// TIA Portal V17 export
// export: Created 2025-07-01T09:58:49.6236345Z, ExportSetting WithDefaults, DisplayName Totally Integrated Automation Portal, DisplayVersion V17 Update 8, DisplayName TIA Portal Openness, DisplayVersion V17 Update 8, DisplayName TIA Portal Version Control Interface, DisplayVersion V17, DisplayName SINAMICS Startdrive Advanced, DisplayVersion V17 SP2, DisplayName SINAMICS Startdrive G110M, G120, G120C, G120D, G120P, G115D, DisplayVersion V17 SP2, DisplayName SINAMICS Startdrive G130, G150, S120, S150, SINAMICS MV, S210, DisplayVersion V17 SP2, DisplayName STEP 7 Professional, DisplayVersion V17 Update 8, DisplayName SINUMERIK ONE STEP 7 Toolbox, DisplayVersion V17 Update 12, DisplayName SINUMERIK ONE PLC Basic Program Plus, DisplayVersion V17 Update 12, DisplayName SINUMERIK 840D sl STEP 7 Toolbox, DisplayVersion V17 Update 12, DisplayName STEP 7 Safety, DisplayVersion V17 Update 6, DisplayName WinCC Advanced, DisplayVersion V17 Update 8
FUNCTION "FC1201_PART_CYCLE_UNIT_1_CLADDING" : Void   // FC1201, LAD
{ S7_Optimized_Access := 'FALSE' }
AUTHOR : ETXETAR
VERSION : 1.0
// stored: AutoNumber false, IsIECCheckEnabled false, SetENOAutomatically false, UDAEnableTagReadback false
   VAR CONSTANT
      FC_NUMBER : DInt := 1201;
   END_VAR
   VAR_TEMP   // added for the SCL form of the ladder/FBD networks
      _w1 : Bool;
      _w2 : Bool;
      _w3 : Bool;
      _w4 : Bool;
   END_VAR
BEGIN

REGION Network 1: GENERAL CONDITIONS
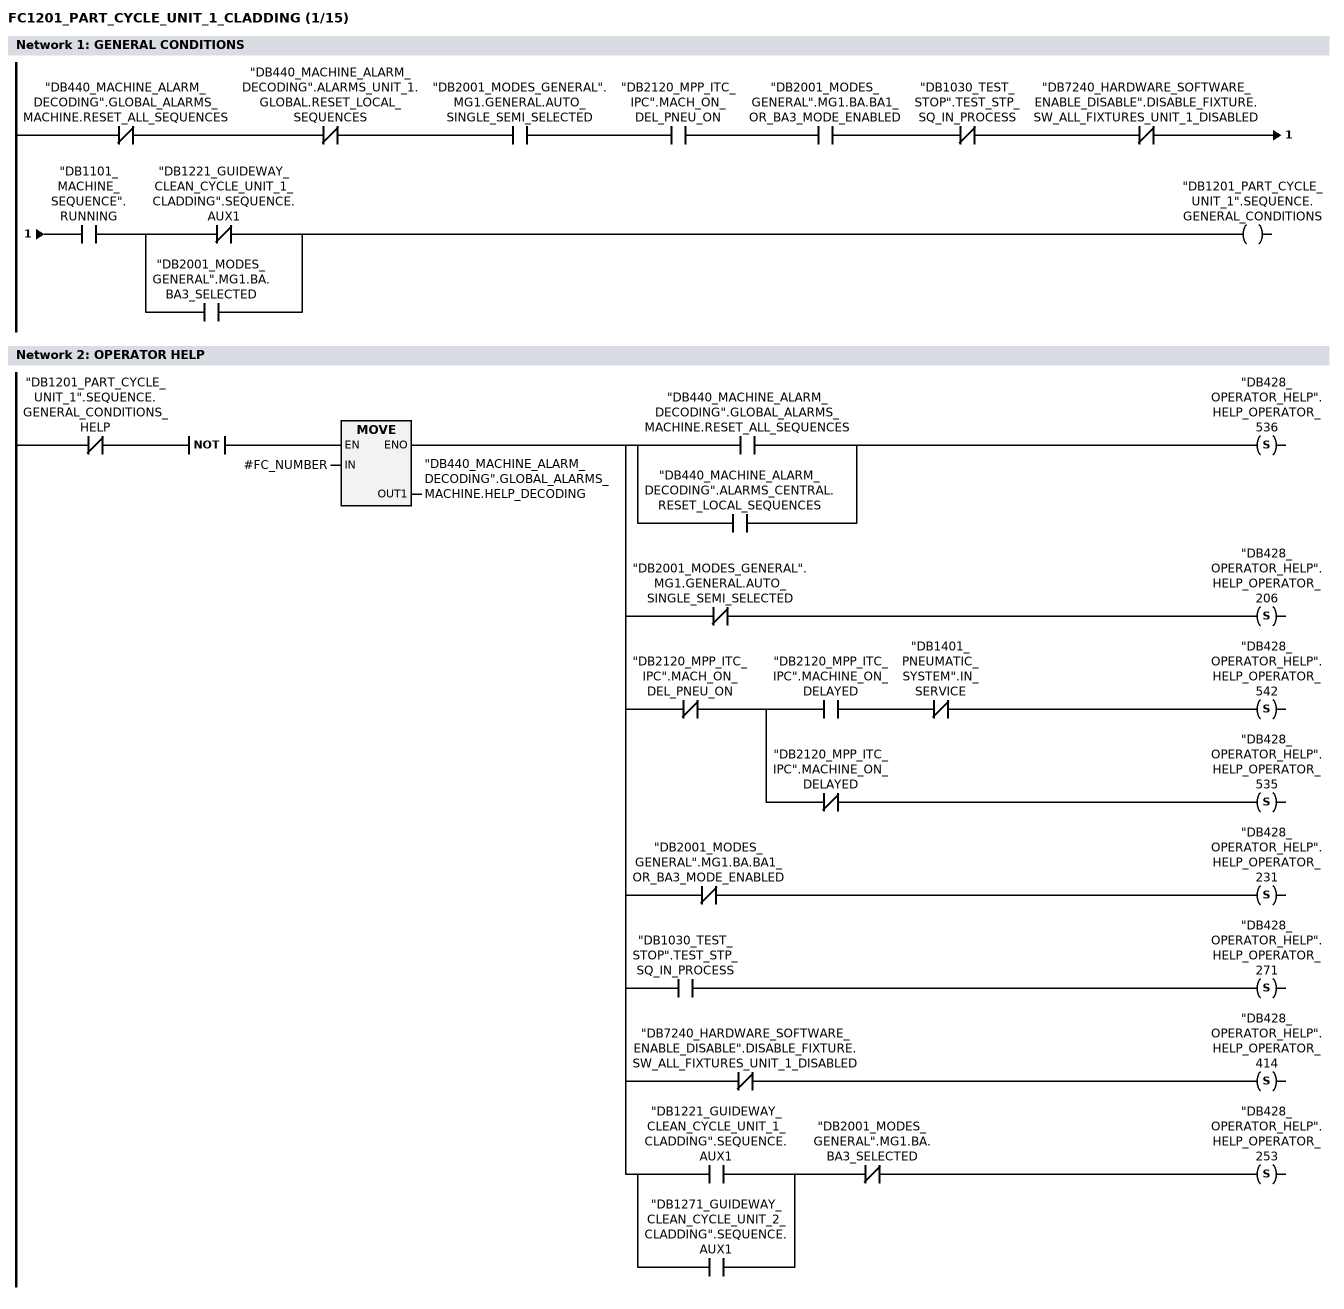
   RUNG wire#powerrail
      I_Contact( "DB440_MACHINE_ALARM_DECODING".GLOBAL_ALARMS_MACHINE.RESET_ALL_SEQUENCES )
      I_Contact( "DB440_MACHINE_ALARM_DECODING".ALARMS_UNIT_1.GLOBAL.RESET_LOCAL_SEQUENCES )
      Contact( "DB2001_MODES_GENERAL".MG1.GENERAL.AUTO_SINGLE_SEMI_SELECTED )
      Contact( "DB2120_MPP_ITC_IPC".MACH_ON_DEL_PNEU_ON )
      Contact( "DB2001_MODES_GENERAL".MG1.BA.BA1_OR_BA3_MODE_ENABLED )
      I_Contact( "DB1030_TEST_STOP".TEST_STP_SQ_IN_PROCESS )
      I_Contact( "DB7240_HARDWARE_SOFTWARE_ENABLE_DISABLE".DISABLE_FIXTURE.SW_ALL_FIXTURES_UNIT_1_DISABLED )
      Contact( "DB1101_MACHINE_SEQUENCE".RUNNING )
      wire#w1
      I_Contact( "DB1221_GUIDEWAY_CLEAN_CYCLE_UNIT_1_CLADDING".SEQUENCE.AUX1 )
      wire#w2
      Coil( "DB1201_PART_CYCLE_UNIT_1".SEQUENCE.GENERAL_CONDITIONS )
   END_RUNG
   RUNG wire#w1
      Contact( "DB2001_MODES_GENERAL".MG1.BA.BA3_SELECTED )
   END_RUNG wire#w2
   // the same network as SCL:
   "DB1201_PART_CYCLE_UNIT_1".SEQUENCE.GENERAL_CONDITIONS := NOT "DB440_MACHINE_ALARM_DECODING".GLOBAL_ALARMS_MACHINE.RESET_ALL_SEQUENCES AND NOT "DB440_MACHINE_ALARM_DECODING".ALARMS_UNIT_1.GLOBAL.RESET_LOCAL_SEQUENCES AND "DB2001_MODES_GENERAL".MG1.GENERAL.AUTO_SINGLE_SEMI_SELECTED AND "DB2120_MPP_ITC_IPC".MACH_ON_DEL_PNEU_ON AND "DB2001_MODES_GENERAL".MG1.BA.BA1_OR_BA3_MODE_ENABLED AND NOT "DB1030_TEST_STOP".TEST_STP_SQ_IN_PROCESS AND NOT "DB7240_HARDWARE_SOFTWARE_ENABLE_DISABLE".DISABLE_FIXTURE.SW_ALL_FIXTURES_UNIT_1_DISABLED AND "DB1101_MACHINE_SEQUENCE".RUNNING AND (NOT "DB1221_GUIDEWAY_CLEAN_CYCLE_UNIT_1_CLADDING".SEQUENCE.AUX1 OR "DB2001_MODES_GENERAL".MG1.BA.BA3_SELECTED);
END_REGION

REGION Network 2: OPERATOR HELP
   RUNG wire#powerrail
      I_Contact( "DB1201_PART_CYCLE_UNIT_1".SEQUENCE.GENERAL_CONDITIONS_HELP )
      Not()
      { S7_GenerateENO := "TRUE" } Move(in := #FC_NUMBER, out1 => "DB440_MACHINE_ALARM_DECODING".GLOBAL_ALARMS_MACHINE.HELP_DECODING)
      wire#w1
      Contact( "DB440_MACHINE_ALARM_DECODING".GLOBAL_ALARMS_MACHINE.RESET_ALL_SEQUENCES )
      wire#w2
      S_Coil( "DB428_OPERATOR_HELP".HELP_OPERATOR_536 )
   END_RUNG
   RUNG wire#w1
      Contact( "DB440_MACHINE_ALARM_DECODING".ALARMS_CENTRAL.RESET_LOCAL_SEQUENCES )
   END_RUNG wire#w2
   RUNG wire#w1
      I_Contact( "DB2001_MODES_GENERAL".MG1.GENERAL.AUTO_SINGLE_SEMI_SELECTED )
      S_Coil( "DB428_OPERATOR_HELP".HELP_OPERATOR_206 )
   END_RUNG
   RUNG wire#w1
      I_Contact( "DB2120_MPP_ITC_IPC".MACH_ON_DEL_PNEU_ON )
      wire#w3
      Contact( "DB2120_MPP_ITC_IPC".MACHINE_ON_DELAYED )
      I_Contact( "DB1401_PNEUMATIC_SYSTEM".IN_SERVICE )
      S_Coil( "DB428_OPERATOR_HELP".HELP_OPERATOR_542 )
   END_RUNG
   RUNG wire#w3
      I_Contact( "DB2120_MPP_ITC_IPC".MACHINE_ON_DELAYED )
      S_Coil( "DB428_OPERATOR_HELP".HELP_OPERATOR_535 )
   END_RUNG
   RUNG wire#w1
      I_Contact( "DB2001_MODES_GENERAL".MG1.BA.BA1_OR_BA3_MODE_ENABLED )
      S_Coil( "DB428_OPERATOR_HELP".HELP_OPERATOR_231 )
   END_RUNG
   RUNG wire#w1
      Contact( "DB1030_TEST_STOP".TEST_STP_SQ_IN_PROCESS )
      S_Coil( "DB428_OPERATOR_HELP".HELP_OPERATOR_271 )
   END_RUNG
   RUNG wire#w1
      I_Contact( "DB7240_HARDWARE_SOFTWARE_ENABLE_DISABLE".DISABLE_FIXTURE.SW_ALL_FIXTURES_UNIT_1_DISABLED )
      S_Coil( "DB428_OPERATOR_HELP".HELP_OPERATOR_414 )
   END_RUNG
   RUNG wire#w1
      Contact( "DB1221_GUIDEWAY_CLEAN_CYCLE_UNIT_1_CLADDING".SEQUENCE.AUX1 )
      wire#w4
      I_Contact( "DB2001_MODES_GENERAL".MG1.BA.BA3_SELECTED )
      S_Coil( "DB428_OPERATOR_HELP".HELP_OPERATOR_253 )
   END_RUNG
   RUNG wire#w1
      Contact( "DB1271_GUIDEWAY_CLEAN_CYCLE_UNIT_2_CLADDING".SEQUENCE.AUX1 )
   END_RUNG wire#w4
   // the same network as SCL:
   // ENO of a box is taken as its EN; it also drops when the box reports an error
   #_w1 := NOT (NOT "DB1201_PART_CYCLE_UNIT_1".SEQUENCE.GENERAL_CONDITIONS_HELP);
   IF #_w1 THEN "DB440_MACHINE_ALARM_DECODING".GLOBAL_ALARMS_MACHINE.HELP_DECODING := #FC_NUMBER; END_IF;
   IF #_w1 AND ("DB440_MACHINE_ALARM_DECODING".GLOBAL_ALARMS_MACHINE.RESET_ALL_SEQUENCES OR "DB440_MACHINE_ALARM_DECODING".ALARMS_CENTRAL.RESET_LOCAL_SEQUENCES) THEN
       "DB428_OPERATOR_HELP".HELP_OPERATOR_536 := TRUE;
   END_IF;
   IF #_w1 AND NOT "DB2001_MODES_GENERAL".MG1.GENERAL.AUTO_SINGLE_SEMI_SELECTED THEN
       "DB428_OPERATOR_HELP".HELP_OPERATOR_206 := TRUE;
   END_IF;
   #_w2 := #_w1 AND NOT "DB2120_MPP_ITC_IPC".MACH_ON_DEL_PNEU_ON;
   IF #_w2 AND "DB2120_MPP_ITC_IPC".MACHINE_ON_DELAYED AND NOT "DB1401_PNEUMATIC_SYSTEM".IN_SERVICE THEN
       "DB428_OPERATOR_HELP".HELP_OPERATOR_542 := TRUE;
   END_IF;
   IF #_w2 AND NOT "DB2120_MPP_ITC_IPC".MACHINE_ON_DELAYED THEN
       "DB428_OPERATOR_HELP".HELP_OPERATOR_535 := TRUE;
   END_IF;
   IF #_w1 AND NOT "DB2001_MODES_GENERAL".MG1.BA.BA1_OR_BA3_MODE_ENABLED THEN
       "DB428_OPERATOR_HELP".HELP_OPERATOR_231 := TRUE;
   END_IF;
   IF #_w1 AND "DB1030_TEST_STOP".TEST_STP_SQ_IN_PROCESS THEN
       "DB428_OPERATOR_HELP".HELP_OPERATOR_271 := TRUE;
   END_IF;
   IF #_w1 AND NOT "DB7240_HARDWARE_SOFTWARE_ENABLE_DISABLE".DISABLE_FIXTURE.SW_ALL_FIXTURES_UNIT_1_DISABLED THEN
       "DB428_OPERATOR_HELP".HELP_OPERATOR_414 := TRUE;
   END_IF;
   IF #_w1 AND ("DB1221_GUIDEWAY_CLEAN_CYCLE_UNIT_1_CLADDING".SEQUENCE.AUX1 OR "DB1271_GUIDEWAY_CLEAN_CYCLE_UNIT_2_CLADDING".SEQUENCE.AUX1) AND NOT "DB2001_MODES_GENERAL".MG1.BA.BA3_SELECTED THEN
       "DB428_OPERATOR_HELP".HELP_OPERATOR_253 := TRUE;
   END_IF;
END_REGION

REGION Network 3: INITIAL CONDITIONS
   // CAMBIAR LOS BITS DE QUALITY CUANDO ESTEN HECHOS
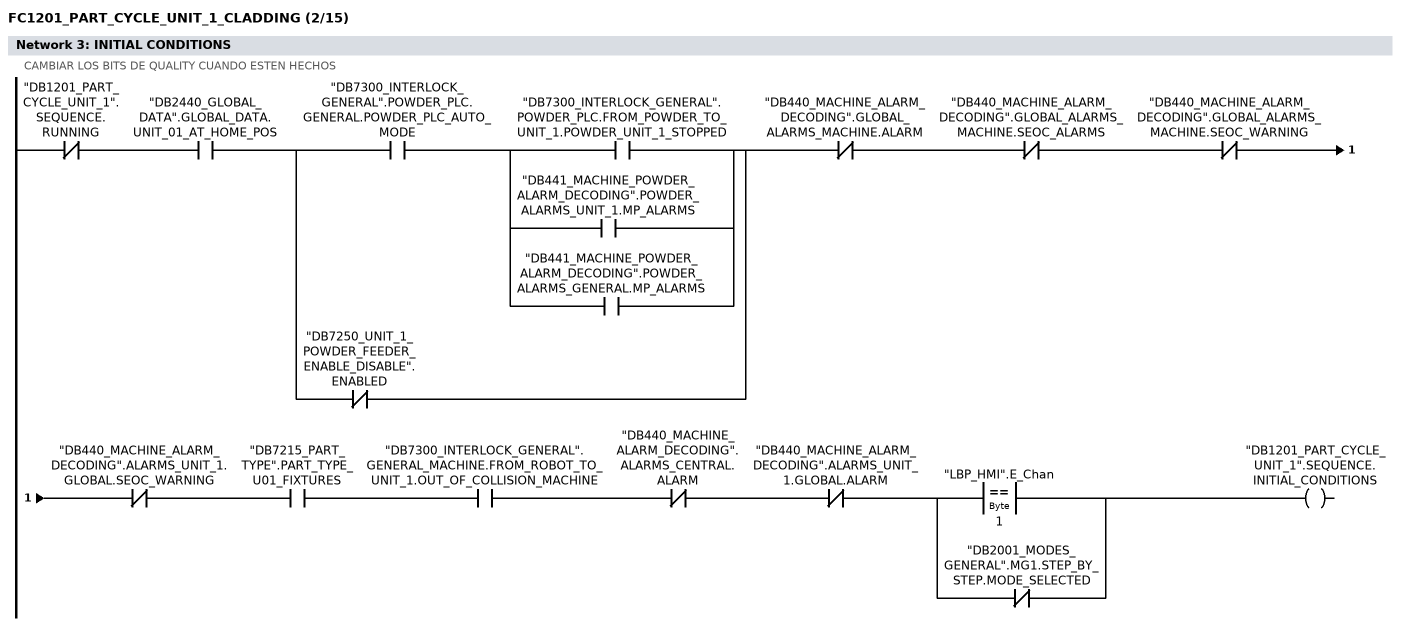
   RUNG wire#powerrail
      I_Contact( "DB1201_PART_CYCLE_UNIT_1".SEQUENCE.RUNNING )
      Contact( "DB2440_GLOBAL_DATA".GLOBAL_DATA.UNIT_01_AT_HOME_POS )
      wire#w1
      Contact( "DB7300_INTERLOCK_GENERAL".POWDER_PLC.GENERAL.POWDER_PLC_AUTO_MODE )
      wire#w2
      Contact( "DB7300_INTERLOCK_GENERAL".POWDER_PLC.FROM_POWDER_TO_UNIT_1.POWDER_UNIT_1_STOPPED )
      wire#w3
      I_Contact( "DB440_MACHINE_ALARM_DECODING".GLOBAL_ALARMS_MACHINE.ALARM )
      I_Contact( "DB440_MACHINE_ALARM_DECODING".GLOBAL_ALARMS_MACHINE.SEOC_ALARMS )
      I_Contact( "DB440_MACHINE_ALARM_DECODING".GLOBAL_ALARMS_MACHINE.SEOC_WARNING )
      I_Contact( "DB440_MACHINE_ALARM_DECODING".ALARMS_UNIT_1.GLOBAL.SEOC_WARNING )
      Contact( "DB7215_PART_TYPE".PART_TYPE_U01_FIXTURES )
      Contact( "DB7300_INTERLOCK_GENERAL".GENERAL_MACHINE.FROM_ROBOT_TO_UNIT_1.OUT_OF_COLLISION_MACHINE )
      I_Contact( "DB440_MACHINE_ALARM_DECODING".ALARMS_CENTRAL.ALARM )
      I_Contact( "DB440_MACHINE_ALARM_DECODING".ALARMS_UNIT_1.GLOBAL.ALARM )
      wire#w4
      { S7_Templates := "SrcType := Byte" } EQ_Contact(in1 := "LBP_HMI".E_Chan, in2 := 1)
      wire#w5
      Coil( "DB1201_PART_CYCLE_UNIT_1".SEQUENCE.INITIAL_CONDITIONS )
   END_RUNG
   RUNG wire#w2
      Contact( "DB441_MACHINE_POWDER_ALARM_DECODING".POWDER_ALARMS_UNIT_1.MP_ALARMS )
   END_RUNG wire#w3
   RUNG wire#w2
      Contact( "DB441_MACHINE_POWDER_ALARM_DECODING".POWDER_ALARMS_GENERAL.MP_ALARMS )
   END_RUNG wire#w3
   RUNG wire#w1
      I_Contact( "DB7250_UNIT_1_POWDER_FEEDER_ENABLE_DISABLE".ENABLED )
   END_RUNG wire#w3
   RUNG wire#w4
      I_Contact( "DB2001_MODES_GENERAL".MG1.STEP_BY_STEP.MODE_SELECTED )
   END_RUNG wire#w5
   // the same network as SCL:
   "DB1201_PART_CYCLE_UNIT_1".SEQUENCE.INITIAL_CONDITIONS := NOT "DB1201_PART_CYCLE_UNIT_1".SEQUENCE.RUNNING AND "DB2440_GLOBAL_DATA".GLOBAL_DATA.UNIT_01_AT_HOME_POS AND (("DB7300_INTERLOCK_GENERAL".POWDER_PLC.GENERAL.POWDER_PLC_AUTO_MODE AND ("DB7300_INTERLOCK_GENERAL".POWDER_PLC.FROM_POWDER_TO_UNIT_1.POWDER_UNIT_1_STOPPED OR "DB441_MACHINE_POWDER_ALARM_DECODING".POWDER_ALARMS_UNIT_1.MP_ALARMS OR "DB441_MACHINE_POWDER_ALARM_DECODING".POWDER_ALARMS_GENERAL.MP_ALARMS)) OR NOT "DB7250_UNIT_1_POWDER_FEEDER_ENABLE_DISABLE".ENABLED) AND NOT "DB440_MACHINE_ALARM_DECODING".GLOBAL_ALARMS_MACHINE.ALARM AND NOT "DB440_MACHINE_ALARM_DECODING".GLOBAL_ALARMS_MACHINE.SEOC_ALARMS AND NOT "DB440_MACHINE_ALARM_DECODING".GLOBAL_ALARMS_MACHINE.SEOC_WARNING AND NOT "DB440_MACHINE_ALARM_DECODING".ALARMS_UNIT_1.GLOBAL.SEOC_WARNING AND "DB7215_PART_TYPE".PART_TYPE_U01_FIXTURES AND "DB7300_INTERLOCK_GENERAL".GENERAL_MACHINE.FROM_ROBOT_TO_UNIT_1.OUT_OF_COLLISION_MACHINE AND NOT "DB440_MACHINE_ALARM_DECODING".ALARMS_CENTRAL.ALARM AND NOT "DB440_MACHINE_ALARM_DECODING".ALARMS_UNIT_1.GLOBAL.ALARM AND (("LBP_HMI".E_Chan = 1) OR NOT "DB2001_MODES_GENERAL".MG1.STEP_BY_STEP.MODE_SELECTED);
END_REGION

REGION Network 4: OPERATOR HELP
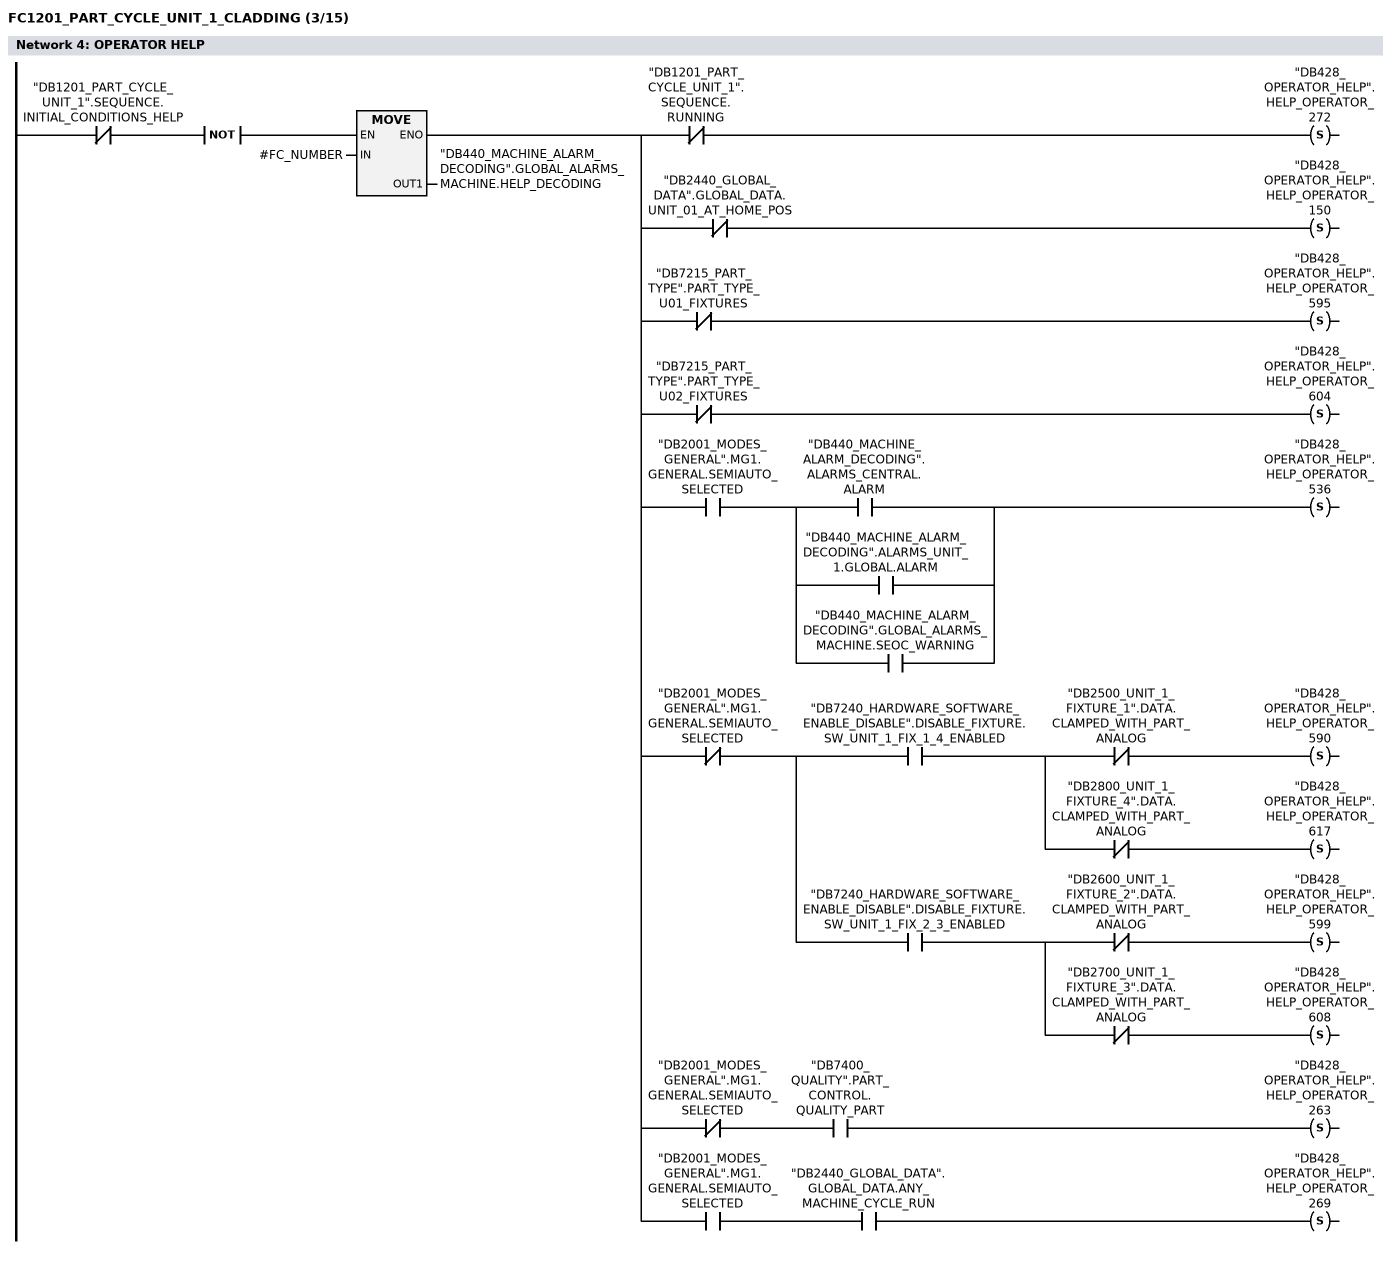
   RUNG wire#powerrail
      I_Contact( "DB1201_PART_CYCLE_UNIT_1".SEQUENCE.INITIAL_CONDITIONS_HELP )
      Not()
      { S7_GenerateENO := "TRUE" } Move(in := #FC_NUMBER, out1 => "DB440_MACHINE_ALARM_DECODING".GLOBAL_ALARMS_MACHINE.HELP_DECODING)
      wire#w1
      I_Contact( "DB1201_PART_CYCLE_UNIT_1".SEQUENCE.RUNNING )
      S_Coil( "DB428_OPERATOR_HELP".HELP_OPERATOR_272 )
   END_RUNG
   RUNG wire#w1
      I_Contact( "DB2440_GLOBAL_DATA".GLOBAL_DATA.UNIT_01_AT_HOME_POS )
      S_Coil( "DB428_OPERATOR_HELP".HELP_OPERATOR_150 )
   END_RUNG
   RUNG wire#w1
      I_Contact( "DB7215_PART_TYPE".PART_TYPE_U01_FIXTURES )
      S_Coil( "DB428_OPERATOR_HELP".HELP_OPERATOR_595 )
   END_RUNG
   RUNG wire#w1
      I_Contact( "DB7215_PART_TYPE".PART_TYPE_U02_FIXTURES )
      S_Coil( "DB428_OPERATOR_HELP".HELP_OPERATOR_604 )
   END_RUNG
   RUNG wire#w1
      Contact( "DB2001_MODES_GENERAL".MG1.GENERAL.SEMIAUTO_SELECTED )
      wire#w2
      Contact( "DB440_MACHINE_ALARM_DECODING".ALARMS_CENTRAL.ALARM )
      wire#w3
      S_Coil( "DB428_OPERATOR_HELP".HELP_OPERATOR_536 )
   END_RUNG
   RUNG wire#w2
      Contact( "DB440_MACHINE_ALARM_DECODING".ALARMS_UNIT_1.GLOBAL.ALARM )
   END_RUNG wire#w3
   RUNG wire#w2
      Contact( "DB440_MACHINE_ALARM_DECODING".GLOBAL_ALARMS_MACHINE.SEOC_WARNING )
   END_RUNG wire#w3
   RUNG wire#w1
      I_Contact( "DB2001_MODES_GENERAL".MG1.GENERAL.SEMIAUTO_SELECTED )
      wire#w4
      Contact( "DB7240_HARDWARE_SOFTWARE_ENABLE_DISABLE".DISABLE_FIXTURE.SW_UNIT_1_FIX_1_4_ENABLED )
      wire#w5
      I_Contact( "DB2500_UNIT_1_FIXTURE_1".DATA.CLAMPED_WITH_PART_ANALOG )
      S_Coil( "DB428_OPERATOR_HELP".HELP_OPERATOR_590 )
   END_RUNG
   RUNG wire#w5
      I_Contact( "DB2800_UNIT_1_FIXTURE_4".DATA.CLAMPED_WITH_PART_ANALOG )
      S_Coil( "DB428_OPERATOR_HELP".HELP_OPERATOR_617 )
   END_RUNG
   RUNG wire#w4
      Contact( "DB7240_HARDWARE_SOFTWARE_ENABLE_DISABLE".DISABLE_FIXTURE.SW_UNIT_1_FIX_2_3_ENABLED )
      wire#w6
      I_Contact( "DB2600_UNIT_1_FIXTURE_2".DATA.CLAMPED_WITH_PART_ANALOG )
      S_Coil( "DB428_OPERATOR_HELP".HELP_OPERATOR_599 )
   END_RUNG
   RUNG wire#w6
      I_Contact( "DB2700_UNIT_1_FIXTURE_3".DATA.CLAMPED_WITH_PART_ANALOG )
      S_Coil( "DB428_OPERATOR_HELP".HELP_OPERATOR_608 )
   END_RUNG
   RUNG wire#w1
      I_Contact( "DB2001_MODES_GENERAL".MG1.GENERAL.SEMIAUTO_SELECTED )
      Contact( "DB7400_QUALITY".PART_CONTROL.QUALITY_PART )
      S_Coil( "DB428_OPERATOR_HELP".HELP_OPERATOR_263 )
   END_RUNG
   RUNG wire#w1
      Contact( "DB2001_MODES_GENERAL".MG1.GENERAL.SEMIAUTO_SELECTED )
      Contact( "DB2440_GLOBAL_DATA".GLOBAL_DATA.ANY_MACHINE_CYCLE_RUN )
      S_Coil( "DB428_OPERATOR_HELP".HELP_OPERATOR_269 )
   END_RUNG
   // the same network as SCL:
   // ENO of a box is taken as its EN; it also drops when the box reports an error
   #_w1 := NOT (NOT "DB1201_PART_CYCLE_UNIT_1".SEQUENCE.INITIAL_CONDITIONS_HELP);
   IF #_w1 THEN "DB440_MACHINE_ALARM_DECODING".GLOBAL_ALARMS_MACHINE.HELP_DECODING := #FC_NUMBER; END_IF;
   IF #_w1 AND NOT "DB1201_PART_CYCLE_UNIT_1".SEQUENCE.RUNNING THEN
       "DB428_OPERATOR_HELP".HELP_OPERATOR_272 := TRUE;
   END_IF;
   IF #_w1 AND NOT "DB2440_GLOBAL_DATA".GLOBAL_DATA.UNIT_01_AT_HOME_POS THEN
       "DB428_OPERATOR_HELP".HELP_OPERATOR_150 := TRUE;
   END_IF;
   IF #_w1 AND NOT "DB7215_PART_TYPE".PART_TYPE_U01_FIXTURES THEN
       "DB428_OPERATOR_HELP".HELP_OPERATOR_595 := TRUE;
   END_IF;
   IF #_w1 AND NOT "DB7215_PART_TYPE".PART_TYPE_U02_FIXTURES THEN
       "DB428_OPERATOR_HELP".HELP_OPERATOR_604 := TRUE;
   END_IF;
   IF #_w1 AND "DB2001_MODES_GENERAL".MG1.GENERAL.SEMIAUTO_SELECTED AND ("DB440_MACHINE_ALARM_DECODING".ALARMS_CENTRAL.ALARM OR "DB440_MACHINE_ALARM_DECODING".ALARMS_UNIT_1.GLOBAL.ALARM OR "DB440_MACHINE_ALARM_DECODING".GLOBAL_ALARMS_MACHINE.SEOC_WARNING) THEN
       "DB428_OPERATOR_HELP".HELP_OPERATOR_536 := TRUE;
   END_IF;
   #_w2 := #_w1 AND NOT "DB2001_MODES_GENERAL".MG1.GENERAL.SEMIAUTO_SELECTED;
   #_w3 := #_w2 AND "DB7240_HARDWARE_SOFTWARE_ENABLE_DISABLE".DISABLE_FIXTURE.SW_UNIT_1_FIX_1_4_ENABLED;
   IF #_w3 AND NOT "DB2500_UNIT_1_FIXTURE_1".DATA.CLAMPED_WITH_PART_ANALOG THEN
       "DB428_OPERATOR_HELP".HELP_OPERATOR_590 := TRUE;
   END_IF;
   IF #_w3 AND NOT "DB2800_UNIT_1_FIXTURE_4".DATA.CLAMPED_WITH_PART_ANALOG THEN
       "DB428_OPERATOR_HELP".HELP_OPERATOR_617 := TRUE;
   END_IF;
   #_w4 := #_w2 AND "DB7240_HARDWARE_SOFTWARE_ENABLE_DISABLE".DISABLE_FIXTURE.SW_UNIT_1_FIX_2_3_ENABLED;
   IF #_w4 AND NOT "DB2600_UNIT_1_FIXTURE_2".DATA.CLAMPED_WITH_PART_ANALOG THEN
       "DB428_OPERATOR_HELP".HELP_OPERATOR_599 := TRUE;
   END_IF;
   IF #_w4 AND NOT "DB2700_UNIT_1_FIXTURE_3".DATA.CLAMPED_WITH_PART_ANALOG THEN
       "DB428_OPERATOR_HELP".HELP_OPERATOR_608 := TRUE;
   END_IF;
   IF #_w1 AND NOT "DB2001_MODES_GENERAL".MG1.GENERAL.SEMIAUTO_SELECTED AND "DB7400_QUALITY".PART_CONTROL.QUALITY_PART THEN
       "DB428_OPERATOR_HELP".HELP_OPERATOR_263 := TRUE;
   END_IF;
   IF #_w1 AND "DB2001_MODES_GENERAL".MG1.GENERAL.SEMIAUTO_SELECTED AND "DB2440_GLOBAL_DATA".GLOBAL_DATA.ANY_MACHINE_CYCLE_RUN THEN
       "DB428_OPERATOR_HELP".HELP_OPERATOR_269 := TRUE;
   END_IF;
END_REGION

REGION Network 5: SEMI AUTO REQUEST
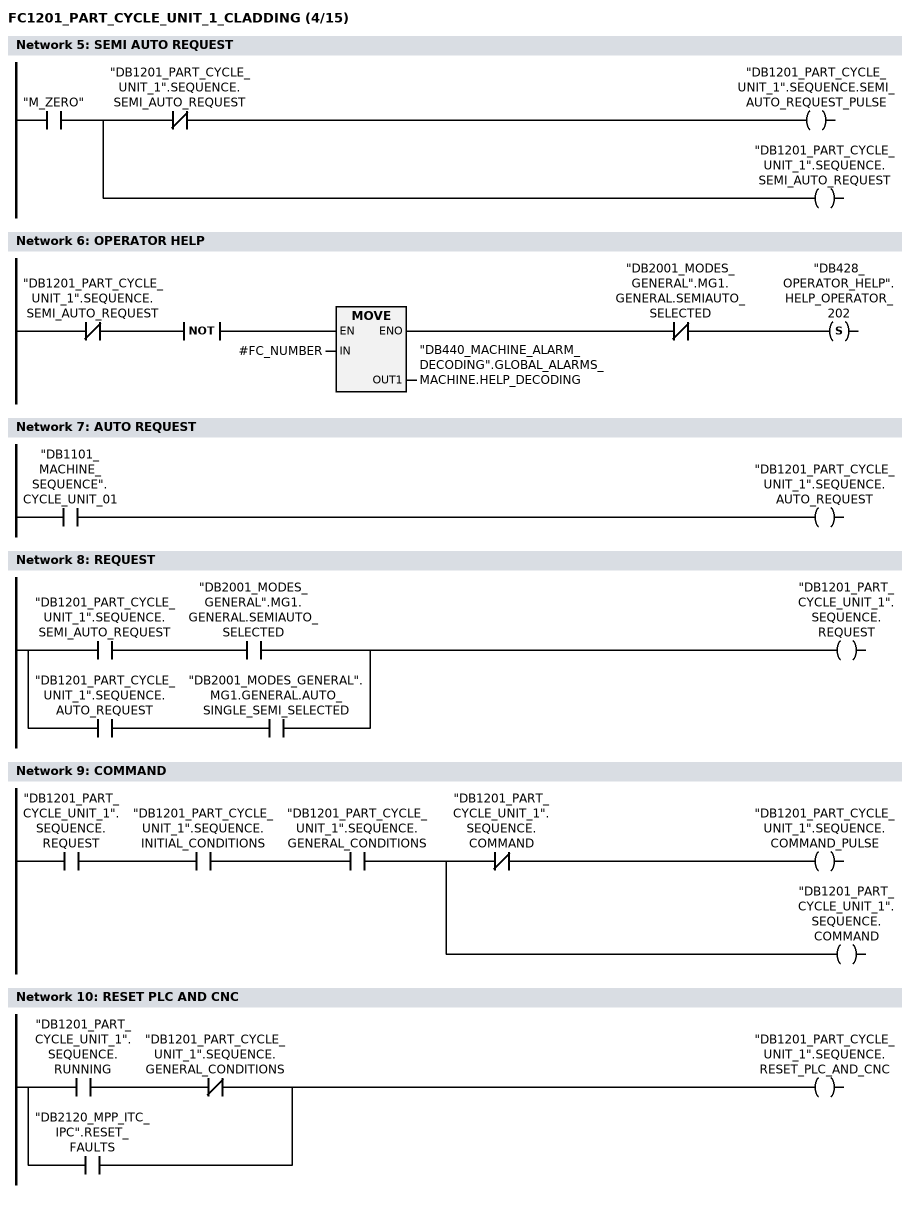
   RUNG wire#powerrail
      Contact( "M_ZERO" )
      wire#w1
      I_Contact( "DB1201_PART_CYCLE_UNIT_1".SEQUENCE.SEMI_AUTO_REQUEST )
      Coil( "DB1201_PART_CYCLE_UNIT_1".SEQUENCE.SEMI_AUTO_REQUEST_PULSE )
   END_RUNG
   RUNG wire#w1
      Coil( "DB1201_PART_CYCLE_UNIT_1".SEQUENCE.SEMI_AUTO_REQUEST )
   END_RUNG
   // the same network as SCL:
   "DB1201_PART_CYCLE_UNIT_1".SEQUENCE.SEMI_AUTO_REQUEST_PULSE := "M_ZERO" AND NOT "DB1201_PART_CYCLE_UNIT_1".SEQUENCE.SEMI_AUTO_REQUEST;
   "DB1201_PART_CYCLE_UNIT_1".SEQUENCE.SEMI_AUTO_REQUEST := "M_ZERO";
END_REGION

REGION Network 6: OPERATOR HELP
   RUNG wire#powerrail
      I_Contact( "DB1201_PART_CYCLE_UNIT_1".SEQUENCE.SEMI_AUTO_REQUEST )
      Not()
      { S7_GenerateENO := "TRUE" } Move(in := #FC_NUMBER, out1 => "DB440_MACHINE_ALARM_DECODING".GLOBAL_ALARMS_MACHINE.HELP_DECODING)
      I_Contact( "DB2001_MODES_GENERAL".MG1.GENERAL.SEMIAUTO_SELECTED )
      S_Coil( "DB428_OPERATOR_HELP".HELP_OPERATOR_202 )
   END_RUNG
   // the same network as SCL:
   // ENO of a box is taken as its EN; it also drops when the box reports an error
   #_w1 := NOT (NOT "DB1201_PART_CYCLE_UNIT_1".SEQUENCE.SEMI_AUTO_REQUEST);
   IF #_w1 THEN "DB440_MACHINE_ALARM_DECODING".GLOBAL_ALARMS_MACHINE.HELP_DECODING := #FC_NUMBER; END_IF;
   IF #_w1 AND NOT "DB2001_MODES_GENERAL".MG1.GENERAL.SEMIAUTO_SELECTED THEN
       "DB428_OPERATOR_HELP".HELP_OPERATOR_202 := TRUE;
   END_IF;
END_REGION

REGION Network 7: AUTO REQUEST
   RUNG wire#powerrail
      Contact( "DB1101_MACHINE_SEQUENCE".CYCLE_UNIT_01 )
      Coil( "DB1201_PART_CYCLE_UNIT_1".SEQUENCE.AUTO_REQUEST )
   END_RUNG
   // the same network as SCL:
   "DB1201_PART_CYCLE_UNIT_1".SEQUENCE.AUTO_REQUEST := "DB1101_MACHINE_SEQUENCE".CYCLE_UNIT_01;
END_REGION

REGION Network 8: REQUEST
   RUNG wire#powerrail
      Contact( "DB1201_PART_CYCLE_UNIT_1".SEQUENCE.SEMI_AUTO_REQUEST )
      Contact( "DB2001_MODES_GENERAL".MG1.GENERAL.SEMIAUTO_SELECTED )
      wire#w1
      Coil( "DB1201_PART_CYCLE_UNIT_1".SEQUENCE.REQUEST )
   END_RUNG
   RUNG wire#powerrail
      Contact( "DB1201_PART_CYCLE_UNIT_1".SEQUENCE.AUTO_REQUEST )
      Contact( "DB2001_MODES_GENERAL".MG1.GENERAL.AUTO_SINGLE_SEMI_SELECTED )
   END_RUNG wire#w1
   // the same network as SCL:
   "DB1201_PART_CYCLE_UNIT_1".SEQUENCE.REQUEST := ("DB1201_PART_CYCLE_UNIT_1".SEQUENCE.SEMI_AUTO_REQUEST AND "DB2001_MODES_GENERAL".MG1.GENERAL.SEMIAUTO_SELECTED) OR ("DB1201_PART_CYCLE_UNIT_1".SEQUENCE.AUTO_REQUEST AND "DB2001_MODES_GENERAL".MG1.GENERAL.AUTO_SINGLE_SEMI_SELECTED);
END_REGION

REGION Network 9: COMMAND
   RUNG wire#powerrail
      Contact( "DB1201_PART_CYCLE_UNIT_1".SEQUENCE.REQUEST )
      Contact( "DB1201_PART_CYCLE_UNIT_1".SEQUENCE.INITIAL_CONDITIONS )
      Contact( "DB1201_PART_CYCLE_UNIT_1".SEQUENCE.GENERAL_CONDITIONS )
      wire#w1
      I_Contact( "DB1201_PART_CYCLE_UNIT_1".SEQUENCE.COMMAND )
      Coil( "DB1201_PART_CYCLE_UNIT_1".SEQUENCE.COMMAND_PULSE )
   END_RUNG
   RUNG wire#w1
      Coil( "DB1201_PART_CYCLE_UNIT_1".SEQUENCE.COMMAND )
   END_RUNG
   // the same network as SCL:
   #_w1 := "DB1201_PART_CYCLE_UNIT_1".SEQUENCE.REQUEST AND "DB1201_PART_CYCLE_UNIT_1".SEQUENCE.INITIAL_CONDITIONS AND "DB1201_PART_CYCLE_UNIT_1".SEQUENCE.GENERAL_CONDITIONS;
   "DB1201_PART_CYCLE_UNIT_1".SEQUENCE.COMMAND_PULSE := #_w1 AND NOT "DB1201_PART_CYCLE_UNIT_1".SEQUENCE.COMMAND;
   "DB1201_PART_CYCLE_UNIT_1".SEQUENCE.COMMAND := #_w1;
END_REGION

REGION Network 10: RESET PLC AND CNC
   RUNG wire#powerrail
      Contact( "DB1201_PART_CYCLE_UNIT_1".SEQUENCE.RUNNING )
      I_Contact( "DB1201_PART_CYCLE_UNIT_1".SEQUENCE.GENERAL_CONDITIONS )
      wire#w1
      Coil( "DB1201_PART_CYCLE_UNIT_1".SEQUENCE.RESET_PLC_AND_CNC )
   END_RUNG
   RUNG wire#powerrail
      Contact( "DB2120_MPP_ITC_IPC".RESET_FAULTS )
   END_RUNG wire#w1
   // the same network as SCL:
   "DB1201_PART_CYCLE_UNIT_1".SEQUENCE.RESET_PLC_AND_CNC := ("DB1201_PART_CYCLE_UNIT_1".SEQUENCE.RUNNING AND NOT "DB1201_PART_CYCLE_UNIT_1".SEQUENCE.GENERAL_CONDITIONS) OR "DB2120_MPP_ITC_IPC".RESET_FAULTS;
END_REGION

REGION Network 11: RUNNING
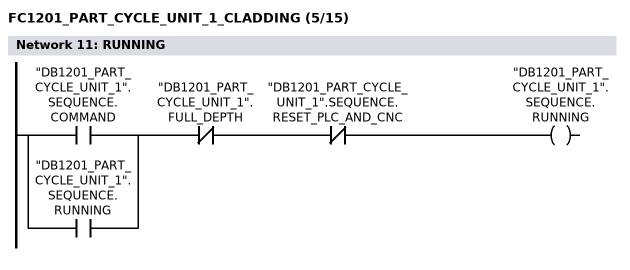
   RUNG wire#powerrail
      Contact( "DB1201_PART_CYCLE_UNIT_1".SEQUENCE.COMMAND )
      wire#w1
      I_Contact( "DB1201_PART_CYCLE_UNIT_1".FULL_DEPTH )
      I_Contact( "DB1201_PART_CYCLE_UNIT_1".SEQUENCE.RESET_PLC_AND_CNC )
      Coil( "DB1201_PART_CYCLE_UNIT_1".SEQUENCE.RUNNING )
   END_RUNG
   RUNG wire#powerrail
      Contact( "DB1201_PART_CYCLE_UNIT_1".SEQUENCE.RUNNING )
   END_RUNG wire#w1
   // the same network as SCL:
   "DB1201_PART_CYCLE_UNIT_1".SEQUENCE.RUNNING := ("DB1201_PART_CYCLE_UNIT_1".SEQUENCE.COMMAND OR "DB1201_PART_CYCLE_UNIT_1".SEQUENCE.RUNNING) AND NOT "DB1201_PART_CYCLE_UNIT_1".FULL_DEPTH AND NOT "DB1201_PART_CYCLE_UNIT_1".SEQUENCE.RESET_PLC_AND_CNC;
END_REGION

REGION Network 12: UNIT 01 STATION 1 CONDITIONS OK FOR STATION 0 CYCLE REQUEST
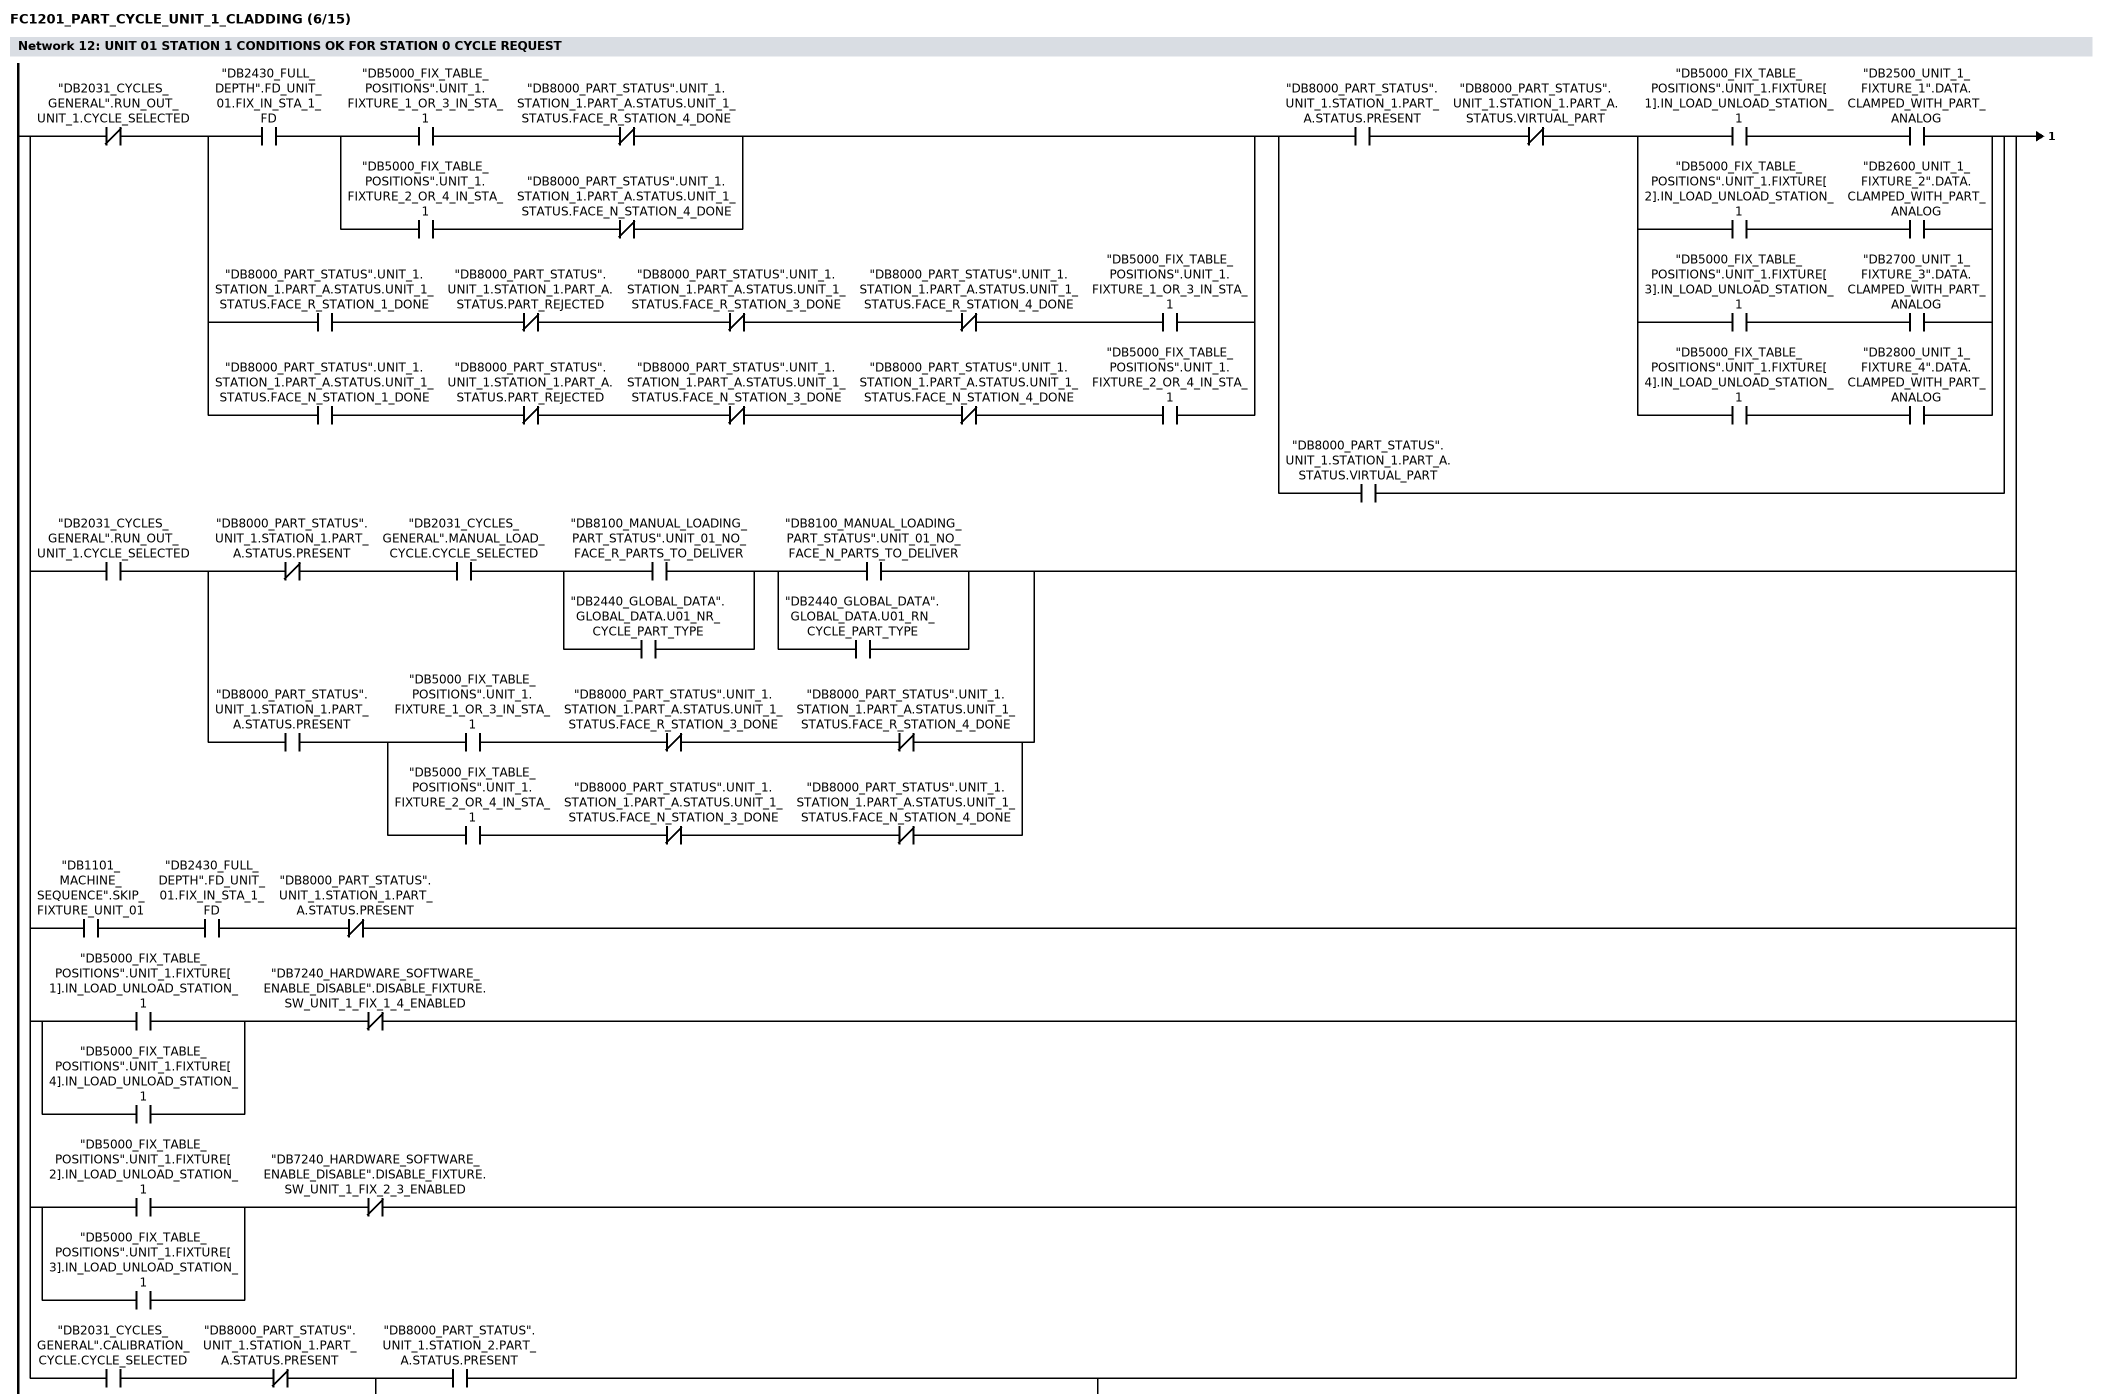
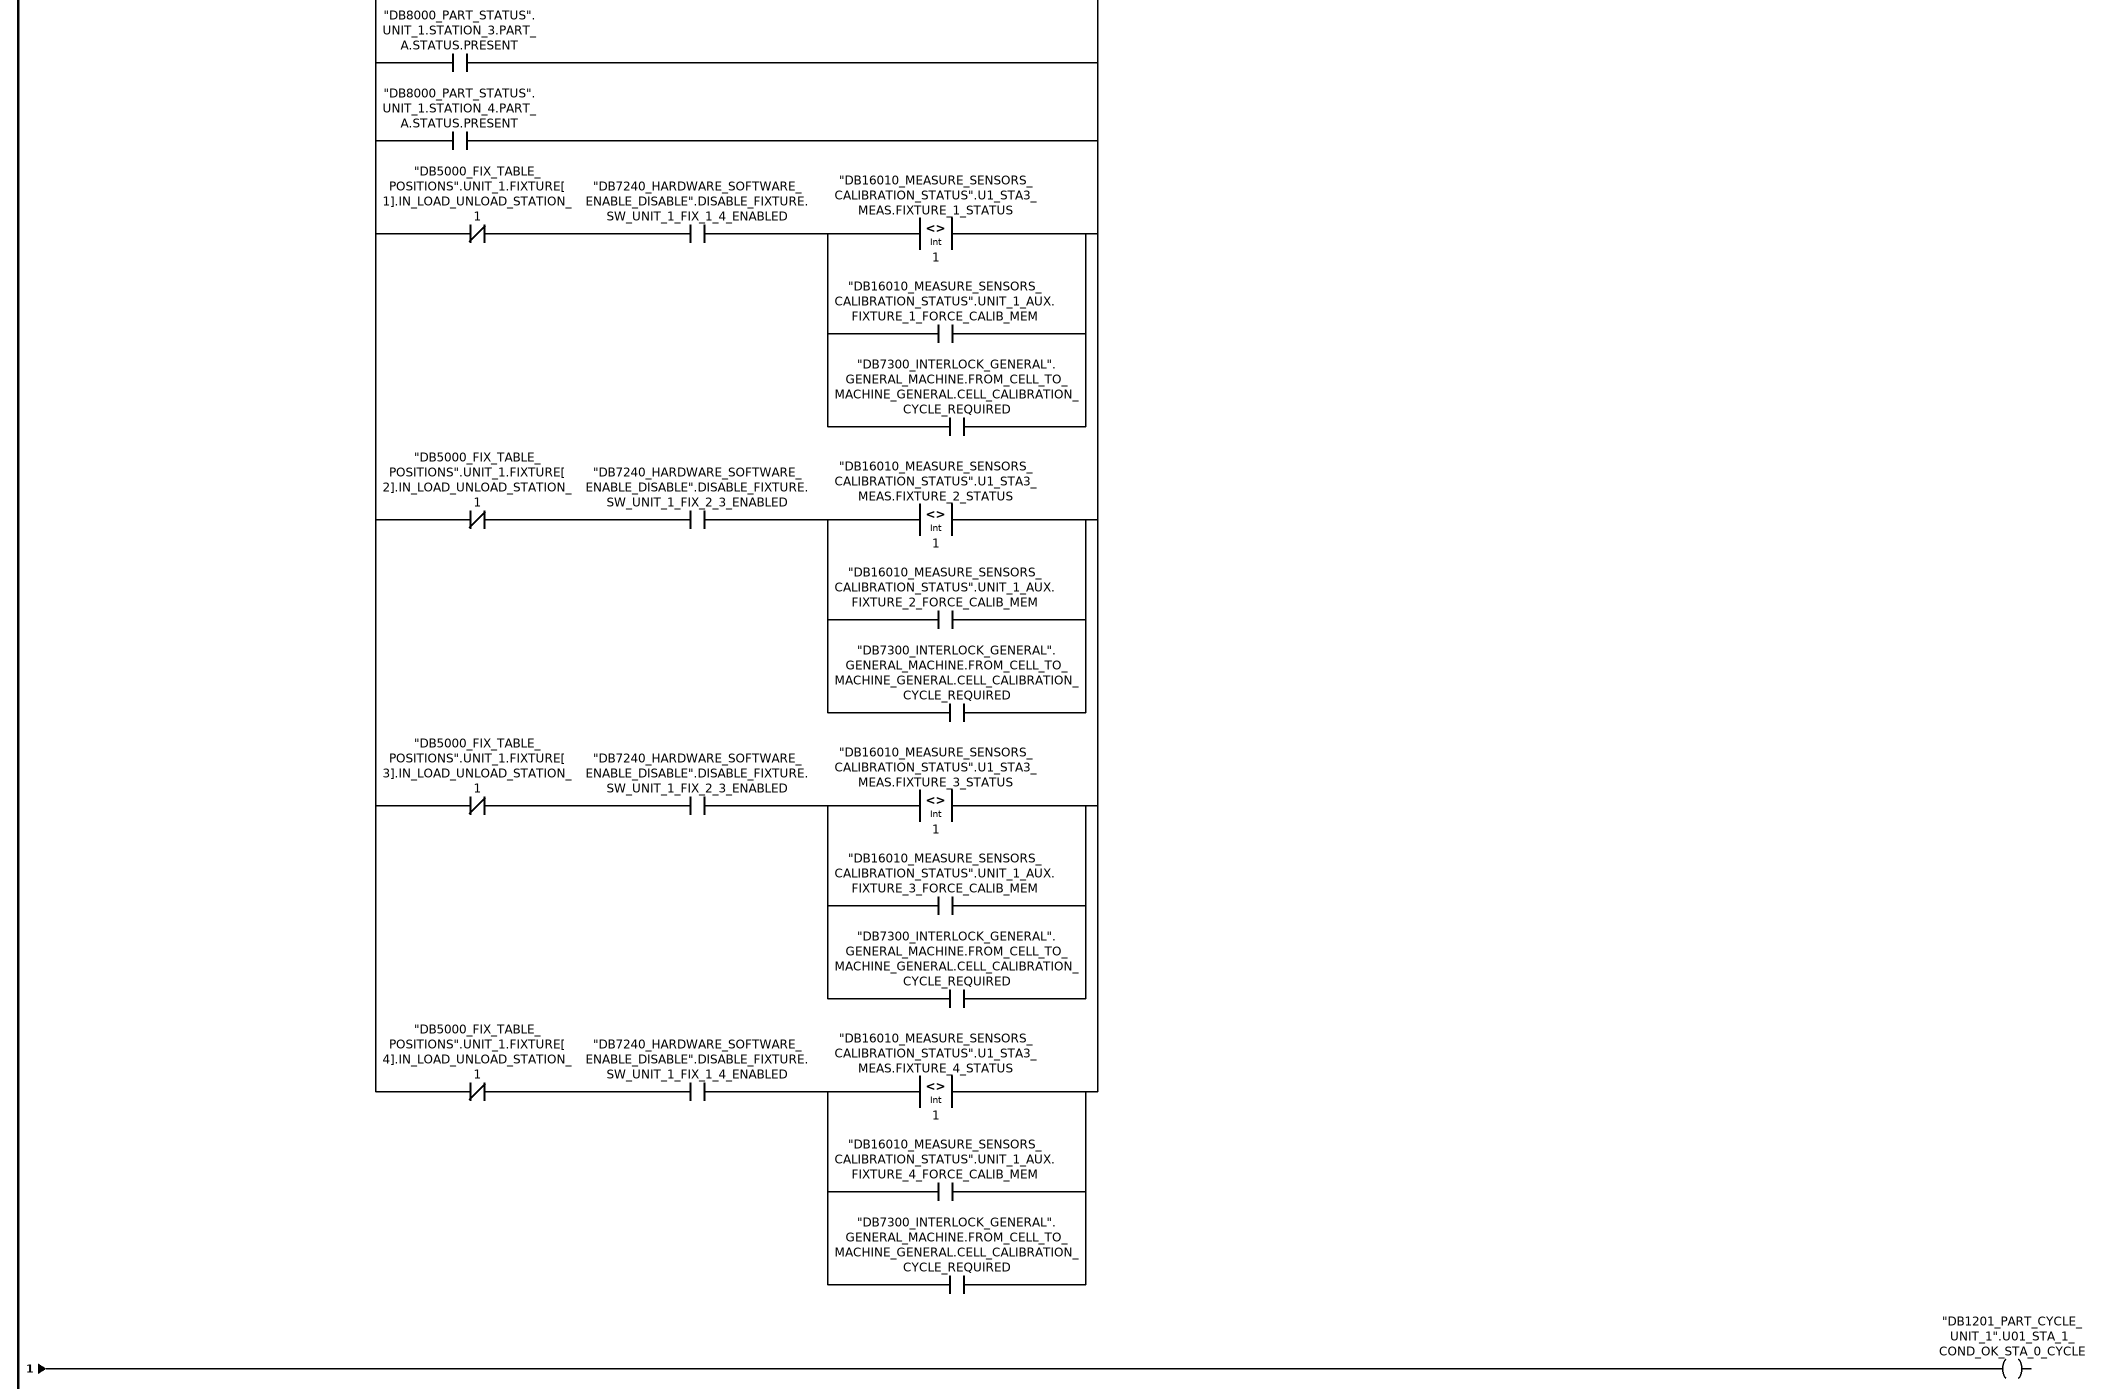
   RUNG wire#powerrail
      I_Contact( "DB2031_CYCLES_GENERAL".RUN_OUT_UNIT_1.CYCLE_SELECTED )
      wire#w1
      Contact( "DB2430_FULL_DEPTH".FD_UNIT_01.FIX_IN_STA_1_FD )
      wire#w2
      Contact( "DB5000_FIX_TABLE_POSITIONS".UNIT_1.FIXTURE_1_OR_3_IN_STA_1 )
      I_Contact( "DB8000_PART_STATUS".UNIT_1.STATION_1.PART_A.STATUS.UNIT_1_STATUS.FACE_R_STATION_4_DONE )
      wire#w3
      Contact( "DB8000_PART_STATUS".UNIT_1.STATION_1.PART_A.STATUS.PRESENT )
      I_Contact( "DB8000_PART_STATUS".UNIT_1.STATION_1.PART_A.STATUS.VIRTUAL_PART )
      wire#w4
      Contact( "DB5000_FIX_TABLE_POSITIONS".UNIT_1.FIXTURE[1].IN_LOAD_UNLOAD_STATION_1 )
      Contact( "DB2500_UNIT_1_FIXTURE_1".DATA.CLAMPED_WITH_PART_ANALOG )
      wire#w5
      Coil( "DB1201_PART_CYCLE_UNIT_1".U01_STA_1_COND_OK_STA_0_CYCLE )
   END_RUNG
   RUNG wire#w2
      Contact( "DB5000_FIX_TABLE_POSITIONS".UNIT_1.FIXTURE_2_OR_4_IN_STA_1 )
      I_Contact( "DB8000_PART_STATUS".UNIT_1.STATION_1.PART_A.STATUS.UNIT_1_STATUS.FACE_N_STATION_4_DONE )
   END_RUNG wire#w3
   RUNG wire#w1
      Contact( "DB8000_PART_STATUS".UNIT_1.STATION_1.PART_A.STATUS.UNIT_1_STATUS.FACE_R_STATION_1_DONE )
      I_Contact( "DB8000_PART_STATUS".UNIT_1.STATION_1.PART_A.STATUS.PART_REJECTED )
      I_Contact( "DB8000_PART_STATUS".UNIT_1.STATION_1.PART_A.STATUS.UNIT_1_STATUS.FACE_R_STATION_3_DONE )
      I_Contact( "DB8000_PART_STATUS".UNIT_1.STATION_1.PART_A.STATUS.UNIT_1_STATUS.FACE_R_STATION_4_DONE )
      Contact( "DB5000_FIX_TABLE_POSITIONS".UNIT_1.FIXTURE_1_OR_3_IN_STA_1 )
   END_RUNG wire#w3
   RUNG wire#w1
      Contact( "DB8000_PART_STATUS".UNIT_1.STATION_1.PART_A.STATUS.UNIT_1_STATUS.FACE_N_STATION_1_DONE )
      I_Contact( "DB8000_PART_STATUS".UNIT_1.STATION_1.PART_A.STATUS.PART_REJECTED )
      I_Contact( "DB8000_PART_STATUS".UNIT_1.STATION_1.PART_A.STATUS.UNIT_1_STATUS.FACE_N_STATION_3_DONE )
      I_Contact( "DB8000_PART_STATUS".UNIT_1.STATION_1.PART_A.STATUS.UNIT_1_STATUS.FACE_N_STATION_4_DONE )
      Contact( "DB5000_FIX_TABLE_POSITIONS".UNIT_1.FIXTURE_2_OR_4_IN_STA_1 )
   END_RUNG wire#w3
   RUNG wire#w4
      Contact( "DB5000_FIX_TABLE_POSITIONS".UNIT_1.FIXTURE[2].IN_LOAD_UNLOAD_STATION_1 )
      Contact( "DB2600_UNIT_1_FIXTURE_2".DATA.CLAMPED_WITH_PART_ANALOG )
   END_RUNG wire#w5
   RUNG wire#w4
      Contact( "DB5000_FIX_TABLE_POSITIONS".UNIT_1.FIXTURE[3].IN_LOAD_UNLOAD_STATION_1 )
      Contact( "DB2700_UNIT_1_FIXTURE_3".DATA.CLAMPED_WITH_PART_ANALOG )
   END_RUNG wire#w5
   RUNG wire#w4
      Contact( "DB5000_FIX_TABLE_POSITIONS".UNIT_1.FIXTURE[4].IN_LOAD_UNLOAD_STATION_1 )
      Contact( "DB2800_UNIT_1_FIXTURE_4".DATA.CLAMPED_WITH_PART_ANALOG )
   END_RUNG wire#w5
   RUNG wire#w3
      Contact( "DB8000_PART_STATUS".UNIT_1.STATION_1.PART_A.STATUS.VIRTUAL_PART )
   END_RUNG wire#w5
   RUNG wire#powerrail
      Contact( "DB2031_CYCLES_GENERAL".RUN_OUT_UNIT_1.CYCLE_SELECTED )
      wire#w6
      I_Contact( "DB8000_PART_STATUS".UNIT_1.STATION_1.PART_A.STATUS.PRESENT )
      Contact( "DB2031_CYCLES_GENERAL".MANUAL_LOAD_CYCLE.CYCLE_SELECTED )
      wire#w7
      Contact( "DB8100_MANUAL_LOADING_PART_STATUS".UNIT_01_NO_FACE_R_PARTS_TO_DELIVER )
      wire#w8
      Contact( "DB8100_MANUAL_LOADING_PART_STATUS".UNIT_01_NO_FACE_N_PARTS_TO_DELIVER )
   END_RUNG wire#w5
   RUNG wire#w7
      Contact( "DB2440_GLOBAL_DATA".GLOBAL_DATA.U01_NR_CYCLE_PART_TYPE )
   END_RUNG wire#w8
   RUNG wire#w8
      Contact( "DB2440_GLOBAL_DATA".GLOBAL_DATA.U01_RN_CYCLE_PART_TYPE )
   END_RUNG wire#w5
   RUNG wire#w6
      Contact( "DB8000_PART_STATUS".UNIT_1.STATION_1.PART_A.STATUS.PRESENT )
      wire#w9
      Contact( "DB5000_FIX_TABLE_POSITIONS".UNIT_1.FIXTURE_1_OR_3_IN_STA_1 )
      I_Contact( "DB8000_PART_STATUS".UNIT_1.STATION_1.PART_A.STATUS.UNIT_1_STATUS.FACE_R_STATION_3_DONE )
      I_Contact( "DB8000_PART_STATUS".UNIT_1.STATION_1.PART_A.STATUS.UNIT_1_STATUS.FACE_R_STATION_4_DONE )
   END_RUNG wire#w5
   RUNG wire#w9
      Contact( "DB5000_FIX_TABLE_POSITIONS".UNIT_1.FIXTURE_2_OR_4_IN_STA_1 )
      I_Contact( "DB8000_PART_STATUS".UNIT_1.STATION_1.PART_A.STATUS.UNIT_1_STATUS.FACE_N_STATION_3_DONE )
      I_Contact( "DB8000_PART_STATUS".UNIT_1.STATION_1.PART_A.STATUS.UNIT_1_STATUS.FACE_N_STATION_4_DONE )
   END_RUNG wire#w5
   RUNG wire#powerrail
      Contact( "DB1101_MACHINE_SEQUENCE".SKIP_FIXTURE_UNIT_01 )
      Contact( "DB2430_FULL_DEPTH".FD_UNIT_01.FIX_IN_STA_1_FD )
      I_Contact( "DB8000_PART_STATUS".UNIT_1.STATION_1.PART_A.STATUS.PRESENT )
   END_RUNG wire#w5
   RUNG wire#powerrail
      Contact( "DB5000_FIX_TABLE_POSITIONS".UNIT_1.FIXTURE[1].IN_LOAD_UNLOAD_STATION_1 )
      wire#w10
      I_Contact( "DB7240_HARDWARE_SOFTWARE_ENABLE_DISABLE".DISABLE_FIXTURE.SW_UNIT_1_FIX_1_4_ENABLED )
   END_RUNG wire#w5
   RUNG wire#powerrail
      Contact( "DB5000_FIX_TABLE_POSITIONS".UNIT_1.FIXTURE[4].IN_LOAD_UNLOAD_STATION_1 )
   END_RUNG wire#w10
   RUNG wire#powerrail
      Contact( "DB5000_FIX_TABLE_POSITIONS".UNIT_1.FIXTURE[2].IN_LOAD_UNLOAD_STATION_1 )
      wire#w11
      I_Contact( "DB7240_HARDWARE_SOFTWARE_ENABLE_DISABLE".DISABLE_FIXTURE.SW_UNIT_1_FIX_2_3_ENABLED )
   END_RUNG wire#w5
   RUNG wire#powerrail
      Contact( "DB5000_FIX_TABLE_POSITIONS".UNIT_1.FIXTURE[3].IN_LOAD_UNLOAD_STATION_1 )
   END_RUNG wire#w11
   RUNG wire#powerrail
      Contact( "DB2031_CYCLES_GENERAL".CALIBRATION_CYCLE.CYCLE_SELECTED )
      I_Contact( "DB8000_PART_STATUS".UNIT_1.STATION_1.PART_A.STATUS.PRESENT )
      wire#w12
      Contact( "DB8000_PART_STATUS".UNIT_1.STATION_2.PART_A.STATUS.PRESENT )
   END_RUNG wire#w5
   RUNG wire#w12
      Contact( "DB8000_PART_STATUS".UNIT_1.STATION_3.PART_A.STATUS.PRESENT )
   END_RUNG wire#w5
   RUNG wire#w12
      Contact( "DB8000_PART_STATUS".UNIT_1.STATION_4.PART_A.STATUS.PRESENT )
   END_RUNG wire#w5
   RUNG wire#w12
      I_Contact( "DB5000_FIX_TABLE_POSITIONS".UNIT_1.FIXTURE[1].IN_LOAD_UNLOAD_STATION_1 )
      Contact( "DB7240_HARDWARE_SOFTWARE_ENABLE_DISABLE".DISABLE_FIXTURE.SW_UNIT_1_FIX_1_4_ENABLED )
      wire#w13
      { S7_Templates := "SrcType := Int" } NE_Contact(in1 := "DB16010_MEASURE_SENSORS_CALIBRATION_STATUS".U1_STA3_MEAS.FIXTURE_1_STATUS, in2 := 1)
   END_RUNG wire#w5
   RUNG wire#w13
      Contact( "DB16010_MEASURE_SENSORS_CALIBRATION_STATUS".UNIT_1_AUX.FIXTURE_1_FORCE_CALIB_MEM )
   END_RUNG wire#w5
   RUNG wire#w13
      Contact( "DB7300_INTERLOCK_GENERAL".GENERAL_MACHINE.FROM_CELL_TO_MACHINE_GENERAL.CELL_CALIBRATION_CYCLE_REQUIRED )
   END_RUNG wire#w5
   RUNG wire#w12
      I_Contact( "DB5000_FIX_TABLE_POSITIONS".UNIT_1.FIXTURE[2].IN_LOAD_UNLOAD_STATION_1 )
      Contact( "DB7240_HARDWARE_SOFTWARE_ENABLE_DISABLE".DISABLE_FIXTURE.SW_UNIT_1_FIX_2_3_ENABLED )
      wire#w14
      { S7_Templates := "SrcType := Int" } NE_Contact(in1 := "DB16010_MEASURE_SENSORS_CALIBRATION_STATUS".U1_STA3_MEAS.FIXTURE_2_STATUS, in2 := 1)
   END_RUNG wire#w5
   RUNG wire#w14
      Contact( "DB16010_MEASURE_SENSORS_CALIBRATION_STATUS".UNIT_1_AUX.FIXTURE_2_FORCE_CALIB_MEM )
   END_RUNG wire#w5
   RUNG wire#w14
      Contact( "DB7300_INTERLOCK_GENERAL".GENERAL_MACHINE.FROM_CELL_TO_MACHINE_GENERAL.CELL_CALIBRATION_CYCLE_REQUIRED )
   END_RUNG wire#w5
   RUNG wire#w12
      I_Contact( "DB5000_FIX_TABLE_POSITIONS".UNIT_1.FIXTURE[3].IN_LOAD_UNLOAD_STATION_1 )
      Contact( "DB7240_HARDWARE_SOFTWARE_ENABLE_DISABLE".DISABLE_FIXTURE.SW_UNIT_1_FIX_2_3_ENABLED )
      wire#w15
      { S7_Templates := "SrcType := Int" } NE_Contact(in1 := "DB16010_MEASURE_SENSORS_CALIBRATION_STATUS".U1_STA3_MEAS.FIXTURE_3_STATUS, in2 := 1)
   END_RUNG wire#w5
   RUNG wire#w15
      Contact( "DB16010_MEASURE_SENSORS_CALIBRATION_STATUS".UNIT_1_AUX.FIXTURE_3_FORCE_CALIB_MEM )
   END_RUNG wire#w5
   RUNG wire#w15
      Contact( "DB7300_INTERLOCK_GENERAL".GENERAL_MACHINE.FROM_CELL_TO_MACHINE_GENERAL.CELL_CALIBRATION_CYCLE_REQUIRED )
   END_RUNG wire#w5
   RUNG wire#w12
      I_Contact( "DB5000_FIX_TABLE_POSITIONS".UNIT_1.FIXTURE[4].IN_LOAD_UNLOAD_STATION_1 )
      Contact( "DB7240_HARDWARE_SOFTWARE_ENABLE_DISABLE".DISABLE_FIXTURE.SW_UNIT_1_FIX_1_4_ENABLED )
      wire#w16
      { S7_Templates := "SrcType := Int" } NE_Contact(in1 := "DB16010_MEASURE_SENSORS_CALIBRATION_STATUS".U1_STA3_MEAS.FIXTURE_4_STATUS, in2 := 1)
   END_RUNG wire#w5
   RUNG wire#w16
      Contact( "DB16010_MEASURE_SENSORS_CALIBRATION_STATUS".UNIT_1_AUX.FIXTURE_4_FORCE_CALIB_MEM )
   END_RUNG wire#w5
   RUNG wire#w16
      Contact( "DB7300_INTERLOCK_GENERAL".GENERAL_MACHINE.FROM_CELL_TO_MACHINE_GENERAL.CELL_CALIBRATION_CYCLE_REQUIRED )
   END_RUNG wire#w5
   // the same network as SCL:
   "DB1201_PART_CYCLE_UNIT_1".U01_STA_1_COND_OK_STA_0_CYCLE := (NOT "DB2031_CYCLES_GENERAL".RUN_OUT_UNIT_1.CYCLE_SELECTED AND (("DB2430_FULL_DEPTH".FD_UNIT_01.FIX_IN_STA_1_FD AND (("DB5000_FIX_TABLE_POSITIONS".UNIT_1.FIXTURE_1_OR_3_IN_STA_1 AND NOT "DB8000_PART_STATUS".UNIT_1.STATION_1.PART_A.STATUS.UNIT_1_STATUS.FACE_R_STATION_4_DONE) OR ("DB5000_FIX_TABLE_POSITIONS".UNIT_1.FIXTURE_2_OR_4_IN_STA_1 AND NOT "DB8000_PART_STATUS".UNIT_1.STATION_1.PART_A.STATUS.UNIT_1_STATUS.FACE_N_STATION_4_DONE))) OR ("DB8000_PART_STATUS".UNIT_1.STATION_1.PART_A.STATUS.UNIT_1_STATUS.FACE_R_STATION_1_DONE AND NOT "DB8000_PART_STATUS".UNIT_1.STATION_1.PART_A.STATUS.PART_REJECTED AND NOT "DB8000_PART_STATUS".UNIT_1.STATION_1.PART_A.STATUS.UNIT_1_STATUS.FACE_R_STATION_3_DONE AND NOT "DB8000_PART_STATUS".UNIT_1.STATION_1.PART_A.STATUS.UNIT_1_STATUS.FACE_R_STATION_4_DONE AND "DB5000_FIX_TABLE_POSITIONS".UNIT_1.FIXTURE_1_OR_3_IN_STA_1) OR ("DB8000_PART_STATUS".UNIT_1.STATION_1.PART_A.STATUS.UNIT_1_STATUS.FACE_N_STATION_1_DONE AND NOT "DB8000_PART_STATUS".UNIT_1.STATION_1.PART_A.STATUS.PART_REJECTED AND NOT "DB8000_PART_STATUS".UNIT_1.STATION_1.PART_A.STATUS.UNIT_1_STATUS.FACE_N_STATION_3_DONE AND NOT "DB8000_PART_STATUS".UNIT_1.STATION_1.PART_A.STATUS.UNIT_1_STATUS.FACE_N_STATION_4_DONE AND "DB5000_FIX_TABLE_POSITIONS".UNIT_1.FIXTURE_2_OR_4_IN_STA_1)) AND (("DB8000_PART_STATUS".UNIT_1.STATION_1.PART_A.STATUS.PRESENT AND NOT "DB8000_PART_STATUS".UNIT_1.STATION_1.PART_A.STATUS.VIRTUAL_PART AND (("DB5000_FIX_TABLE_POSITIONS".UNIT_1.FIXTURE[1].IN_LOAD_UNLOAD_STATION_1 AND "DB2500_UNIT_1_FIXTURE_1".DATA.CLAMPED_WITH_PART_ANALOG) OR ("DB5000_FIX_TABLE_POSITIONS".UNIT_1.FIXTURE[2].IN_LOAD_UNLOAD_STATION_1 AND "DB2600_UNIT_1_FIXTURE_2".DATA.CLAMPED_WITH_PART_ANALOG) OR ("DB5000_FIX_TABLE_POSITIONS".UNIT_1.FIXTURE[3].IN_LOAD_UNLOAD_STATION_1 AND "DB2700_UNIT_1_FIXTURE_3".DATA.CLAMPED_WITH_PART_ANALOG) OR ("DB5000_FIX_TABLE_POSITIONS".UNIT_1.FIXTURE[4].IN_LOAD_UNLOAD_STATION_1 AND "DB2800_UNIT_1_FIXTURE_4".DATA.CLAMPED_WITH_PART_ANALOG))) OR "DB8000_PART_STATUS".UNIT_1.STATION_1.PART_A.STATUS.VIRTUAL_PART)) OR ("DB2031_CYCLES_GENERAL".RUN_OUT_UNIT_1.CYCLE_SELECTED AND ((NOT "DB8000_PART_STATUS".UNIT_1.STATION_1.PART_A.STATUS.PRESENT AND "DB2031_CYCLES_GENERAL".MANUAL_LOAD_CYCLE.CYCLE_SELECTED AND ("DB8100_MANUAL_LOADING_PART_STATUS".UNIT_01_NO_FACE_R_PARTS_TO_DELIVER OR "DB2440_GLOBAL_DATA".GLOBAL_DATA.U01_NR_CYCLE_PART_TYPE) AND ("DB8100_MANUAL_LOADING_PART_STATUS".UNIT_01_NO_FACE_N_PARTS_TO_DELIVER OR "DB2440_GLOBAL_DATA".GLOBAL_DATA.U01_RN_CYCLE_PART_TYPE)) OR ("DB8000_PART_STATUS".UNIT_1.STATION_1.PART_A.STATUS.PRESENT AND (("DB5000_FIX_TABLE_POSITIONS".UNIT_1.FIXTURE_1_OR_3_IN_STA_1 AND NOT "DB8000_PART_STATUS".UNIT_1.STATION_1.PART_A.STATUS.UNIT_1_STATUS.FACE_R_STATION_3_DONE AND NOT "DB8000_PART_STATUS".UNIT_1.STATION_1.PART_A.STATUS.UNIT_1_STATUS.FACE_R_STATION_4_DONE) OR ("DB5000_FIX_TABLE_POSITIONS".UNIT_1.FIXTURE_2_OR_4_IN_STA_1 AND NOT "DB8000_PART_STATUS".UNIT_1.STATION_1.PART_A.STATUS.UNIT_1_STATUS.FACE_N_STATION_3_DONE AND NOT "DB8000_PART_STATUS".UNIT_1.STATION_1.PART_A.STATUS.UNIT_1_STATUS.FACE_N_STATION_4_DONE))))) OR ("DB1101_MACHINE_SEQUENCE".SKIP_FIXTURE_UNIT_01 AND "DB2430_FULL_DEPTH".FD_UNIT_01.FIX_IN_STA_1_FD AND NOT "DB8000_PART_STATUS".UNIT_1.STATION_1.PART_A.STATUS.PRESENT) OR (("DB5000_FIX_TABLE_POSITIONS".UNIT_1.FIXTURE[1].IN_LOAD_UNLOAD_STATION_1 OR "DB5000_FIX_TABLE_POSITIONS".UNIT_1.FIXTURE[4].IN_LOAD_UNLOAD_STATION_1) AND NOT "DB7240_HARDWARE_SOFTWARE_ENABLE_DISABLE".DISABLE_FIXTURE.SW_UNIT_1_FIX_1_4_ENABLED) OR (("DB5000_FIX_TABLE_POSITIONS".UNIT_1.FIXTURE[2].IN_LOAD_UNLOAD_STATION_1 OR "DB5000_FIX_TABLE_POSITIONS".UNIT_1.FIXTURE[3].IN_LOAD_UNLOAD_STATION_1) AND NOT "DB7240_HARDWARE_SOFTWARE_ENABLE_DISABLE".DISABLE_FIXTURE.SW_UNIT_1_FIX_2_3_ENABLED) OR ("DB2031_CYCLES_GENERAL".CALIBRATION_CYCLE.CYCLE_SELECTED AND NOT "DB8000_PART_STATUS".UNIT_1.STATION_1.PART_A.STATUS.PRESENT AND ("DB8000_PART_STATUS".UNIT_1.STATION_2.PART_A.STATUS.PRESENT OR "DB8000_PART_STATUS".UNIT_1.STATION_3.PART_A.STATUS.PRESENT OR "DB8000_PART_STATUS".UNIT_1.STATION_4.PART_A.STATUS.PRESENT OR (NOT "DB5000_FIX_TABLE_POSITIONS".UNIT_1.FIXTURE[1].IN_LOAD_UNLOAD_STATION_1 AND "DB7240_HARDWARE_SOFTWARE_ENABLE_DISABLE".DISABLE_FIXTURE.SW_UNIT_1_FIX_1_4_ENABLED AND (("DB16010_MEASURE_SENSORS_CALIBRATION_STATUS".U1_STA3_MEAS.FIXTURE_1_STATUS <> 1) OR "DB16010_MEASURE_SENSORS_CALIBRATION_STATUS".UNIT_1_AUX.FIXTURE_1_FORCE_CALIB_MEM OR "DB7300_INTERLOCK_GENERAL".GENERAL_MACHINE.FROM_CELL_TO_MACHINE_GENERAL.CELL_CALIBRATION_CYCLE_REQUIRED)) OR (NOT "DB5000_FIX_TABLE_POSITIONS".UNIT_1.FIXTURE[2].IN_LOAD_UNLOAD_STATION_1 AND "DB7240_HARDWARE_SOFTWARE_ENABLE_DISABLE".DISABLE_FIXTURE.SW_UNIT_1_FIX_2_3_ENABLED AND (("DB16010_MEASURE_SENSORS_CALIBRATION_STATUS".U1_STA3_MEAS.FIXTURE_2_STATUS <> 1) OR "DB16010_MEASURE_SENSORS_CALIBRATION_STATUS".UNIT_1_AUX.FIXTURE_2_FORCE_CALIB_MEM OR "DB7300_INTERLOCK_GENERAL".GENERAL_MACHINE.FROM_CELL_TO_MACHINE_GENERAL.CELL_CALIBRATION_CYCLE_REQUIRED)) OR (NOT "DB5000_FIX_TABLE_POSITIONS".UNIT_1.FIXTURE[3].IN_LOAD_UNLOAD_STATION_1 AND "DB7240_HARDWARE_SOFTWARE_ENABLE_DISABLE".DISABLE_FIXTURE.SW_UNIT_1_FIX_2_3_ENABLED AND (("DB16010_MEASURE_SENSORS_CALIBRATION_STATUS".U1_STA3_MEAS.FIXTURE_3_STATUS <> 1) OR "DB16010_MEASURE_SENSORS_CALIBRATION_STATUS".UNIT_1_AUX.FIXTURE_3_FORCE_CALIB_MEM OR "DB7300_INTERLOCK_GENERAL".GENERAL_MACHINE.FROM_CELL_TO_MACHINE_GENERAL.CELL_CALIBRATION_CYCLE_REQUIRED)) OR (NOT "DB5000_FIX_TABLE_POSITIONS".UNIT_1.FIXTURE[4].IN_LOAD_UNLOAD_STATION_1 AND "DB7240_HARDWARE_SOFTWARE_ENABLE_DISABLE".DISABLE_FIXTURE.SW_UNIT_1_FIX_1_4_ENABLED AND (("DB16010_MEASURE_SENSORS_CALIBRATION_STATUS".U1_STA3_MEAS.FIXTURE_4_STATUS <> 1) OR "DB16010_MEASURE_SENSORS_CALIBRATION_STATUS".UNIT_1_AUX.FIXTURE_4_FORCE_CALIB_MEM OR "DB7300_INTERLOCK_GENERAL".GENERAL_MACHINE.FROM_CELL_TO_MACHINE_GENERAL.CELL_CALIBRATION_CYCLE_REQUIRED))));
END_REGION

REGION Network 13: UNIT 01 STATION 2 CONDITIONS OK FOR STATION 0 CYCLE REQUEST
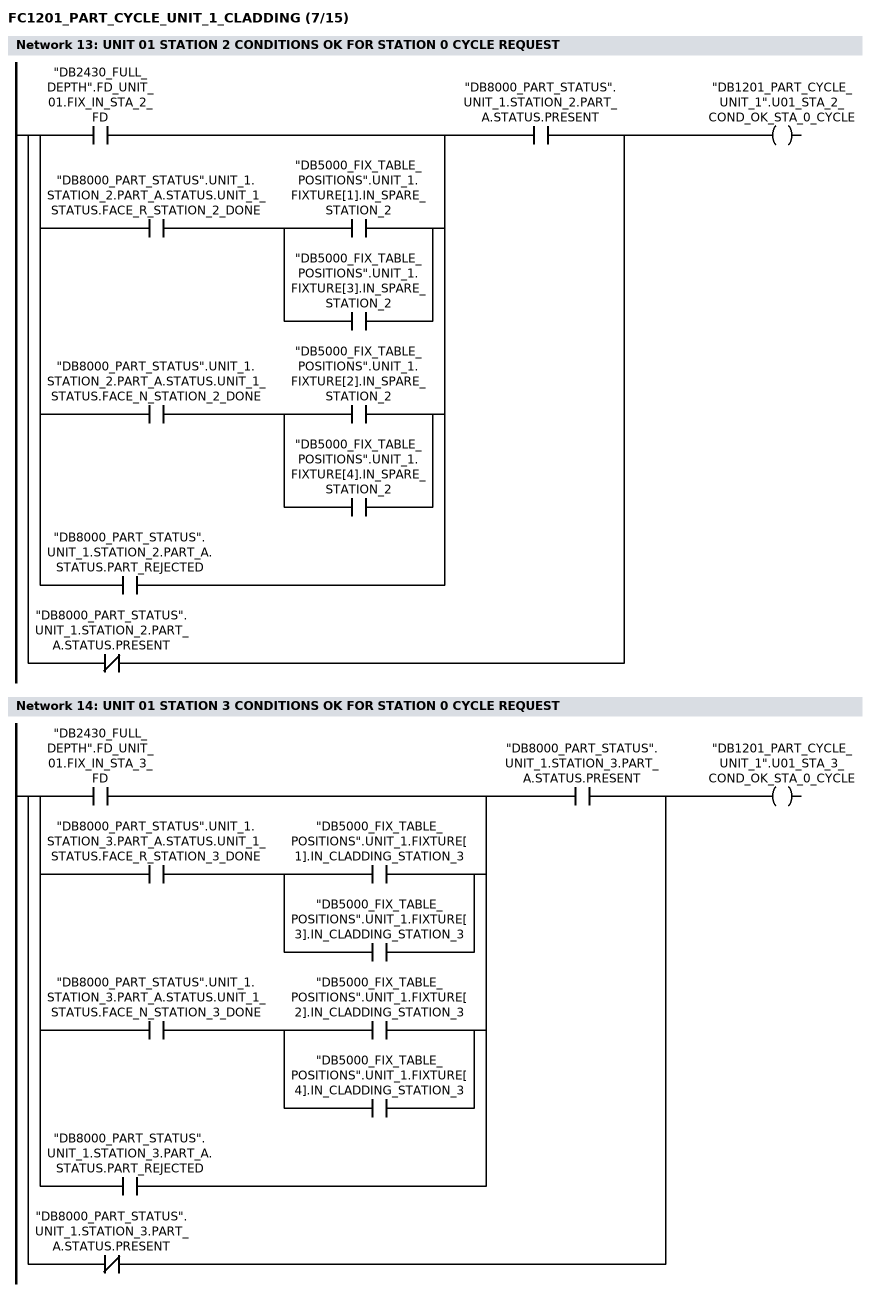
   RUNG wire#powerrail
      Contact( "DB2430_FULL_DEPTH".FD_UNIT_01.FIX_IN_STA_2_FD )
      wire#w1
      Contact( "DB8000_PART_STATUS".UNIT_1.STATION_2.PART_A.STATUS.PRESENT )
      wire#w4
      Coil( "DB1201_PART_CYCLE_UNIT_1".U01_STA_2_COND_OK_STA_0_CYCLE )
   END_RUNG
   RUNG wire#powerrail
      Contact( "DB8000_PART_STATUS".UNIT_1.STATION_2.PART_A.STATUS.UNIT_1_STATUS.FACE_R_STATION_2_DONE )
      wire#w2
      Contact( "DB5000_FIX_TABLE_POSITIONS".UNIT_1.FIXTURE[1].IN_SPARE_STATION_2 )
   END_RUNG wire#w1
   RUNG wire#w2
      Contact( "DB5000_FIX_TABLE_POSITIONS".UNIT_1.FIXTURE[3].IN_SPARE_STATION_2 )
   END_RUNG wire#w1
   RUNG wire#powerrail
      Contact( "DB8000_PART_STATUS".UNIT_1.STATION_2.PART_A.STATUS.UNIT_1_STATUS.FACE_N_STATION_2_DONE )
      wire#w3
      Contact( "DB5000_FIX_TABLE_POSITIONS".UNIT_1.FIXTURE[2].IN_SPARE_STATION_2 )
   END_RUNG wire#w1
   RUNG wire#w3
      Contact( "DB5000_FIX_TABLE_POSITIONS".UNIT_1.FIXTURE[4].IN_SPARE_STATION_2 )
   END_RUNG wire#w1
   RUNG wire#powerrail
      Contact( "DB8000_PART_STATUS".UNIT_1.STATION_2.PART_A.STATUS.PART_REJECTED )
   END_RUNG wire#w1
   RUNG wire#powerrail
      I_Contact( "DB8000_PART_STATUS".UNIT_1.STATION_2.PART_A.STATUS.PRESENT )
   END_RUNG wire#w4
   // the same network as SCL:
   "DB1201_PART_CYCLE_UNIT_1".U01_STA_2_COND_OK_STA_0_CYCLE := (("DB2430_FULL_DEPTH".FD_UNIT_01.FIX_IN_STA_2_FD OR ("DB8000_PART_STATUS".UNIT_1.STATION_2.PART_A.STATUS.UNIT_1_STATUS.FACE_R_STATION_2_DONE AND ("DB5000_FIX_TABLE_POSITIONS".UNIT_1.FIXTURE[1].IN_SPARE_STATION_2 OR "DB5000_FIX_TABLE_POSITIONS".UNIT_1.FIXTURE[3].IN_SPARE_STATION_2)) OR ("DB8000_PART_STATUS".UNIT_1.STATION_2.PART_A.STATUS.UNIT_1_STATUS.FACE_N_STATION_2_DONE AND ("DB5000_FIX_TABLE_POSITIONS".UNIT_1.FIXTURE[2].IN_SPARE_STATION_2 OR "DB5000_FIX_TABLE_POSITIONS".UNIT_1.FIXTURE[4].IN_SPARE_STATION_2)) OR "DB8000_PART_STATUS".UNIT_1.STATION_2.PART_A.STATUS.PART_REJECTED) AND "DB8000_PART_STATUS".UNIT_1.STATION_2.PART_A.STATUS.PRESENT) OR NOT "DB8000_PART_STATUS".UNIT_1.STATION_2.PART_A.STATUS.PRESENT;
END_REGION

REGION Network 14: UNIT 01 STATION 3 CONDITIONS OK FOR STATION 0 CYCLE REQUEST
   RUNG wire#powerrail
      Contact( "DB2430_FULL_DEPTH".FD_UNIT_01.FIX_IN_STA_3_FD )
      wire#w1
      Contact( "DB8000_PART_STATUS".UNIT_1.STATION_3.PART_A.STATUS.PRESENT )
      wire#w4
      Coil( "DB1201_PART_CYCLE_UNIT_1".U01_STA_3_COND_OK_STA_0_CYCLE )
   END_RUNG
   RUNG wire#powerrail
      Contact( "DB8000_PART_STATUS".UNIT_1.STATION_3.PART_A.STATUS.UNIT_1_STATUS.FACE_R_STATION_3_DONE )
      wire#w2
      Contact( "DB5000_FIX_TABLE_POSITIONS".UNIT_1.FIXTURE[1].IN_CLADDING_STATION_3 )
   END_RUNG wire#w1
   RUNG wire#w2
      Contact( "DB5000_FIX_TABLE_POSITIONS".UNIT_1.FIXTURE[3].IN_CLADDING_STATION_3 )
   END_RUNG wire#w1
   RUNG wire#powerrail
      Contact( "DB8000_PART_STATUS".UNIT_1.STATION_3.PART_A.STATUS.UNIT_1_STATUS.FACE_N_STATION_3_DONE )
      wire#w3
      Contact( "DB5000_FIX_TABLE_POSITIONS".UNIT_1.FIXTURE[2].IN_CLADDING_STATION_3 )
   END_RUNG wire#w1
   RUNG wire#w3
      Contact( "DB5000_FIX_TABLE_POSITIONS".UNIT_1.FIXTURE[4].IN_CLADDING_STATION_3 )
   END_RUNG wire#w1
   RUNG wire#powerrail
      Contact( "DB8000_PART_STATUS".UNIT_1.STATION_3.PART_A.STATUS.PART_REJECTED )
   END_RUNG wire#w1
   RUNG wire#powerrail
      I_Contact( "DB8000_PART_STATUS".UNIT_1.STATION_3.PART_A.STATUS.PRESENT )
   END_RUNG wire#w4
   // the same network as SCL:
   "DB1201_PART_CYCLE_UNIT_1".U01_STA_3_COND_OK_STA_0_CYCLE := (("DB2430_FULL_DEPTH".FD_UNIT_01.FIX_IN_STA_3_FD OR ("DB8000_PART_STATUS".UNIT_1.STATION_3.PART_A.STATUS.UNIT_1_STATUS.FACE_R_STATION_3_DONE AND ("DB5000_FIX_TABLE_POSITIONS".UNIT_1.FIXTURE[1].IN_CLADDING_STATION_3 OR "DB5000_FIX_TABLE_POSITIONS".UNIT_1.FIXTURE[3].IN_CLADDING_STATION_3)) OR ("DB8000_PART_STATUS".UNIT_1.STATION_3.PART_A.STATUS.UNIT_1_STATUS.FACE_N_STATION_3_DONE AND ("DB5000_FIX_TABLE_POSITIONS".UNIT_1.FIXTURE[2].IN_CLADDING_STATION_3 OR "DB5000_FIX_TABLE_POSITIONS".UNIT_1.FIXTURE[4].IN_CLADDING_STATION_3)) OR "DB8000_PART_STATUS".UNIT_1.STATION_3.PART_A.STATUS.PART_REJECTED) AND "DB8000_PART_STATUS".UNIT_1.STATION_3.PART_A.STATUS.PRESENT) OR NOT "DB8000_PART_STATUS".UNIT_1.STATION_3.PART_A.STATUS.PRESENT;
END_REGION

REGION Network 15: UNIT 01 STATION 4 CONDITIONS OK FOR STATION 0 CYCLE REQUEST
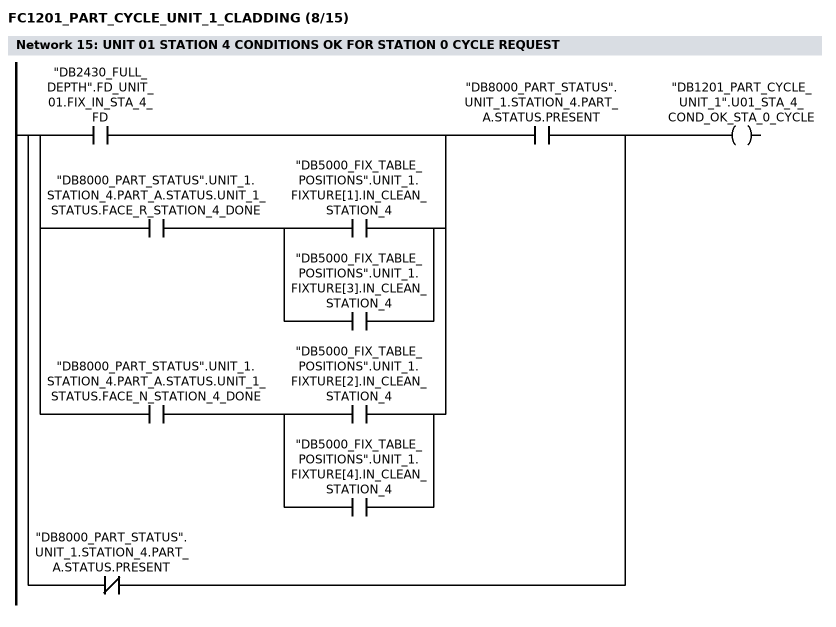
   RUNG wire#powerrail
      Contact( "DB2430_FULL_DEPTH".FD_UNIT_01.FIX_IN_STA_4_FD )
      wire#w1
      Contact( "DB8000_PART_STATUS".UNIT_1.STATION_4.PART_A.STATUS.PRESENT )
      wire#w4
      Coil( "DB1201_PART_CYCLE_UNIT_1".U01_STA_4_COND_OK_STA_0_CYCLE )
   END_RUNG
   RUNG wire#powerrail
      Contact( "DB8000_PART_STATUS".UNIT_1.STATION_4.PART_A.STATUS.UNIT_1_STATUS.FACE_R_STATION_4_DONE )
      wire#w2
      Contact( "DB5000_FIX_TABLE_POSITIONS".UNIT_1.FIXTURE[1].IN_CLEAN_STATION_4 )
   END_RUNG wire#w1
   RUNG wire#w2
      Contact( "DB5000_FIX_TABLE_POSITIONS".UNIT_1.FIXTURE[3].IN_CLEAN_STATION_4 )
   END_RUNG wire#w1
   RUNG wire#powerrail
      Contact( "DB8000_PART_STATUS".UNIT_1.STATION_4.PART_A.STATUS.UNIT_1_STATUS.FACE_N_STATION_4_DONE )
      wire#w3
      Contact( "DB5000_FIX_TABLE_POSITIONS".UNIT_1.FIXTURE[2].IN_CLEAN_STATION_4 )
   END_RUNG wire#w1
   RUNG wire#w3
      Contact( "DB5000_FIX_TABLE_POSITIONS".UNIT_1.FIXTURE[4].IN_CLEAN_STATION_4 )
   END_RUNG wire#w1
   RUNG wire#powerrail
      I_Contact( "DB8000_PART_STATUS".UNIT_1.STATION_4.PART_A.STATUS.PRESENT )
   END_RUNG wire#w4
   // the same network as SCL:
   "DB1201_PART_CYCLE_UNIT_1".U01_STA_4_COND_OK_STA_0_CYCLE := (("DB2430_FULL_DEPTH".FD_UNIT_01.FIX_IN_STA_4_FD OR ("DB8000_PART_STATUS".UNIT_1.STATION_4.PART_A.STATUS.UNIT_1_STATUS.FACE_R_STATION_4_DONE AND ("DB5000_FIX_TABLE_POSITIONS".UNIT_1.FIXTURE[1].IN_CLEAN_STATION_4 OR "DB5000_FIX_TABLE_POSITIONS".UNIT_1.FIXTURE[3].IN_CLEAN_STATION_4)) OR ("DB8000_PART_STATUS".UNIT_1.STATION_4.PART_A.STATUS.UNIT_1_STATUS.FACE_N_STATION_4_DONE AND ("DB5000_FIX_TABLE_POSITIONS".UNIT_1.FIXTURE[2].IN_CLEAN_STATION_4 OR "DB5000_FIX_TABLE_POSITIONS".UNIT_1.FIXTURE[4].IN_CLEAN_STATION_4))) AND "DB8000_PART_STATUS".UNIT_1.STATION_4.PART_A.STATUS.PRESENT) OR NOT "DB8000_PART_STATUS".UNIT_1.STATION_4.PART_A.STATUS.PRESENT;
END_REGION

REGION Network 16: UNIT 01 NEW FACE IN STATION 1
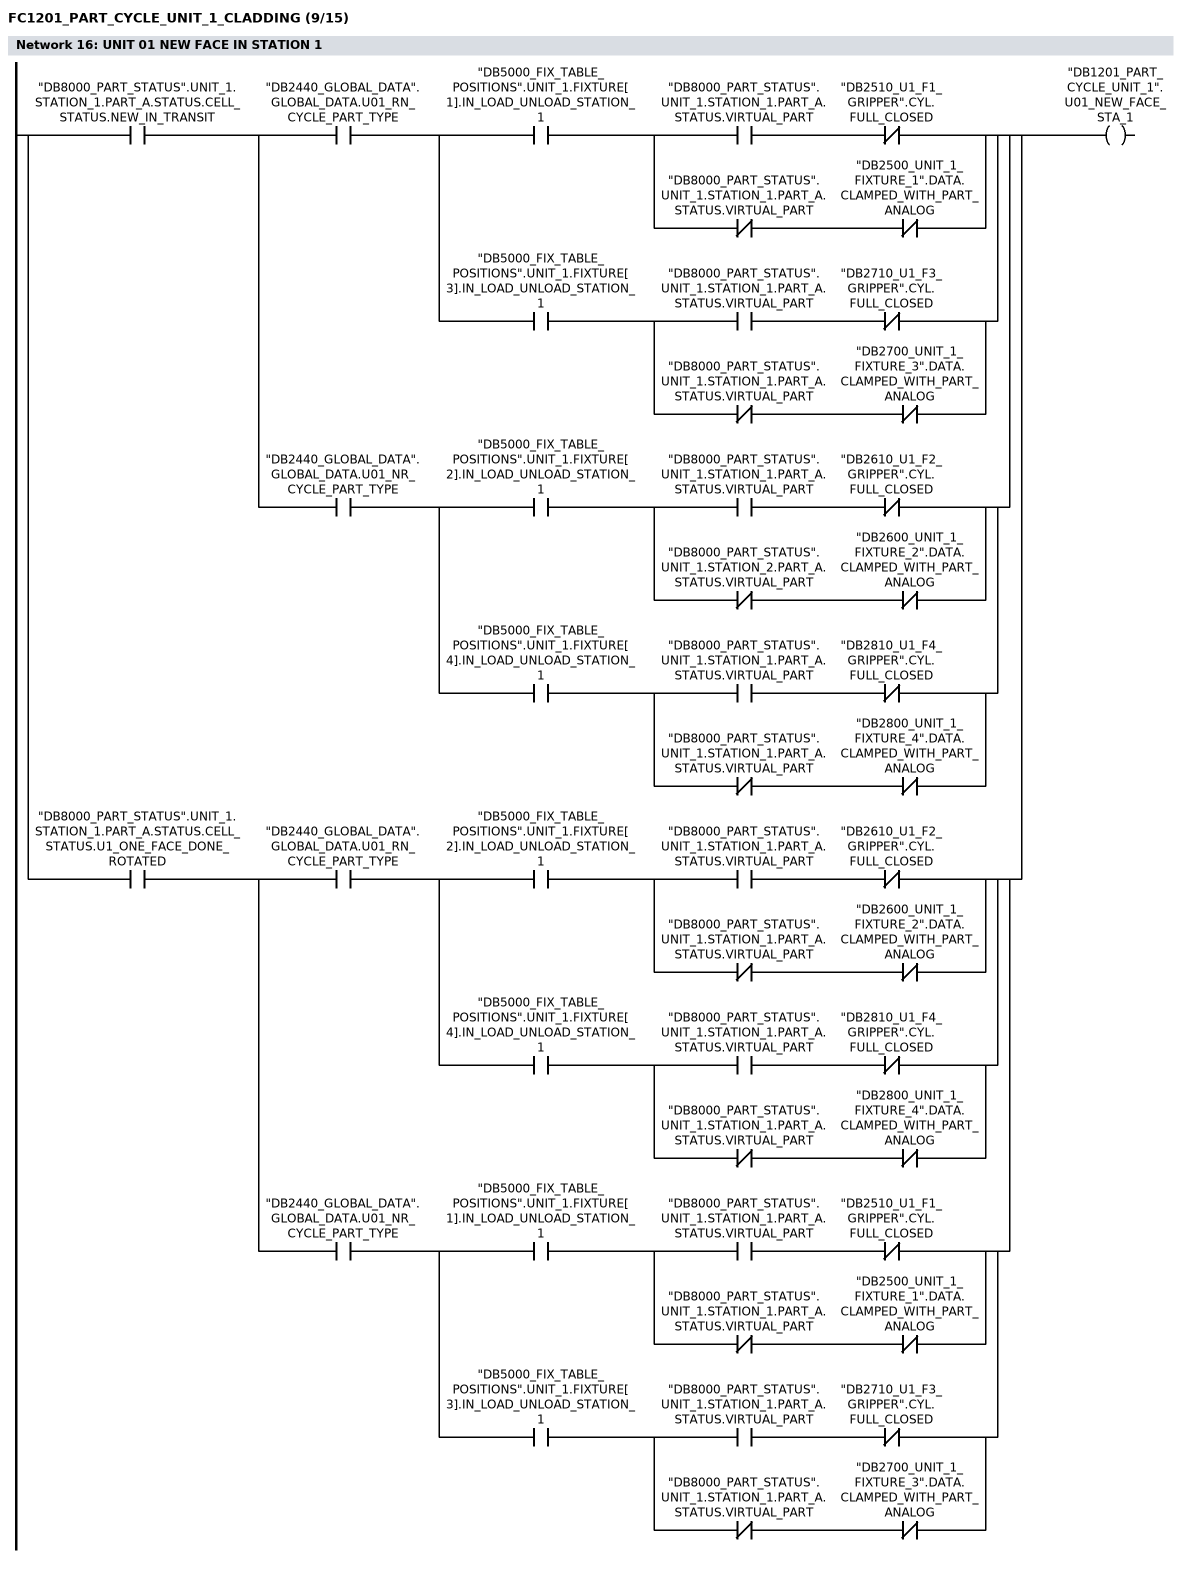
   RUNG wire#powerrail
      Contact( "DB8000_PART_STATUS".UNIT_1.STATION_1.PART_A.STATUS.CELL_STATUS.NEW_IN_TRANSIT )
      wire#w1
      Contact( "DB2440_GLOBAL_DATA".GLOBAL_DATA.U01_RN_CYCLE_PART_TYPE )
      wire#w2
      Contact( "DB5000_FIX_TABLE_POSITIONS".UNIT_1.FIXTURE[1].IN_LOAD_UNLOAD_STATION_1 )
      wire#w3
      Contact( "DB8000_PART_STATUS".UNIT_1.STATION_1.PART_A.STATUS.VIRTUAL_PART )
      I_Contact( "DB2510_U1_F1_GRIPPER".CYL.FULL_CLOSED )
      wire#w4
      Coil( "DB1201_PART_CYCLE_UNIT_1".U01_NEW_FACE_STA_1 )
   END_RUNG
   RUNG wire#w3
      I_Contact( "DB8000_PART_STATUS".UNIT_1.STATION_1.PART_A.STATUS.VIRTUAL_PART )
      I_Contact( "DB2500_UNIT_1_FIXTURE_1".DATA.CLAMPED_WITH_PART_ANALOG )
   END_RUNG wire#w4
   RUNG wire#w2
      Contact( "DB5000_FIX_TABLE_POSITIONS".UNIT_1.FIXTURE[3].IN_LOAD_UNLOAD_STATION_1 )
      wire#w5
      Contact( "DB8000_PART_STATUS".UNIT_1.STATION_1.PART_A.STATUS.VIRTUAL_PART )
      I_Contact( "DB2710_U1_F3_GRIPPER".CYL.FULL_CLOSED )
   END_RUNG wire#w4
   RUNG wire#w5
      I_Contact( "DB8000_PART_STATUS".UNIT_1.STATION_1.PART_A.STATUS.VIRTUAL_PART )
      I_Contact( "DB2700_UNIT_1_FIXTURE_3".DATA.CLAMPED_WITH_PART_ANALOG )
   END_RUNG wire#w4
   RUNG wire#w1
      Contact( "DB2440_GLOBAL_DATA".GLOBAL_DATA.U01_NR_CYCLE_PART_TYPE )
      wire#w6
      Contact( "DB5000_FIX_TABLE_POSITIONS".UNIT_1.FIXTURE[2].IN_LOAD_UNLOAD_STATION_1 )
      wire#w7
      Contact( "DB8000_PART_STATUS".UNIT_1.STATION_1.PART_A.STATUS.VIRTUAL_PART )
      I_Contact( "DB2610_U1_F2_GRIPPER".CYL.FULL_CLOSED )
   END_RUNG wire#w4
   RUNG wire#w7
      I_Contact( "DB8000_PART_STATUS".UNIT_1.STATION_2.PART_A.STATUS.VIRTUAL_PART )
      I_Contact( "DB2600_UNIT_1_FIXTURE_2".DATA.CLAMPED_WITH_PART_ANALOG )
   END_RUNG wire#w4
   RUNG wire#w6
      Contact( "DB5000_FIX_TABLE_POSITIONS".UNIT_1.FIXTURE[4].IN_LOAD_UNLOAD_STATION_1 )
      wire#w8
      Contact( "DB8000_PART_STATUS".UNIT_1.STATION_1.PART_A.STATUS.VIRTUAL_PART )
      I_Contact( "DB2810_U1_F4_GRIPPER".CYL.FULL_CLOSED )
   END_RUNG wire#w4
   RUNG wire#w8
      I_Contact( "DB8000_PART_STATUS".UNIT_1.STATION_1.PART_A.STATUS.VIRTUAL_PART )
      I_Contact( "DB2800_UNIT_1_FIXTURE_4".DATA.CLAMPED_WITH_PART_ANALOG )
   END_RUNG wire#w4
   RUNG wire#powerrail
      Contact( "DB8000_PART_STATUS".UNIT_1.STATION_1.PART_A.STATUS.CELL_STATUS.U1_ONE_FACE_DONE_ROTATED )
      wire#w9
      Contact( "DB2440_GLOBAL_DATA".GLOBAL_DATA.U01_RN_CYCLE_PART_TYPE )
      wire#w10
      Contact( "DB5000_FIX_TABLE_POSITIONS".UNIT_1.FIXTURE[2].IN_LOAD_UNLOAD_STATION_1 )
      wire#w11
      Contact( "DB8000_PART_STATUS".UNIT_1.STATION_1.PART_A.STATUS.VIRTUAL_PART )
      I_Contact( "DB2610_U1_F2_GRIPPER".CYL.FULL_CLOSED )
   END_RUNG wire#w4
   RUNG wire#w11
      I_Contact( "DB8000_PART_STATUS".UNIT_1.STATION_1.PART_A.STATUS.VIRTUAL_PART )
      I_Contact( "DB2600_UNIT_1_FIXTURE_2".DATA.CLAMPED_WITH_PART_ANALOG )
   END_RUNG wire#w4
   RUNG wire#w10
      Contact( "DB5000_FIX_TABLE_POSITIONS".UNIT_1.FIXTURE[4].IN_LOAD_UNLOAD_STATION_1 )
      wire#w12
      Contact( "DB8000_PART_STATUS".UNIT_1.STATION_1.PART_A.STATUS.VIRTUAL_PART )
      I_Contact( "DB2810_U1_F4_GRIPPER".CYL.FULL_CLOSED )
   END_RUNG wire#w4
   RUNG wire#w12
      I_Contact( "DB8000_PART_STATUS".UNIT_1.STATION_1.PART_A.STATUS.VIRTUAL_PART )
      I_Contact( "DB2800_UNIT_1_FIXTURE_4".DATA.CLAMPED_WITH_PART_ANALOG )
   END_RUNG wire#w4
   RUNG wire#w9
      Contact( "DB2440_GLOBAL_DATA".GLOBAL_DATA.U01_NR_CYCLE_PART_TYPE )
      wire#w13
      Contact( "DB5000_FIX_TABLE_POSITIONS".UNIT_1.FIXTURE[1].IN_LOAD_UNLOAD_STATION_1 )
      wire#w14
      Contact( "DB8000_PART_STATUS".UNIT_1.STATION_1.PART_A.STATUS.VIRTUAL_PART )
      I_Contact( "DB2510_U1_F1_GRIPPER".CYL.FULL_CLOSED )
   END_RUNG wire#w4
   RUNG wire#w14
      I_Contact( "DB8000_PART_STATUS".UNIT_1.STATION_1.PART_A.STATUS.VIRTUAL_PART )
      I_Contact( "DB2500_UNIT_1_FIXTURE_1".DATA.CLAMPED_WITH_PART_ANALOG )
   END_RUNG wire#w4
   RUNG wire#w13
      Contact( "DB5000_FIX_TABLE_POSITIONS".UNIT_1.FIXTURE[3].IN_LOAD_UNLOAD_STATION_1 )
      wire#w15
      Contact( "DB8000_PART_STATUS".UNIT_1.STATION_1.PART_A.STATUS.VIRTUAL_PART )
      I_Contact( "DB2710_U1_F3_GRIPPER".CYL.FULL_CLOSED )
   END_RUNG wire#w4
   RUNG wire#w15
      I_Contact( "DB8000_PART_STATUS".UNIT_1.STATION_1.PART_A.STATUS.VIRTUAL_PART )
      I_Contact( "DB2700_UNIT_1_FIXTURE_3".DATA.CLAMPED_WITH_PART_ANALOG )
   END_RUNG wire#w4
   // the same network as SCL:
   "DB1201_PART_CYCLE_UNIT_1".U01_NEW_FACE_STA_1 := ("DB8000_PART_STATUS".UNIT_1.STATION_1.PART_A.STATUS.CELL_STATUS.NEW_IN_TRANSIT AND (("DB2440_GLOBAL_DATA".GLOBAL_DATA.U01_RN_CYCLE_PART_TYPE AND (("DB5000_FIX_TABLE_POSITIONS".UNIT_1.FIXTURE[1].IN_LOAD_UNLOAD_STATION_1 AND (("DB8000_PART_STATUS".UNIT_1.STATION_1.PART_A.STATUS.VIRTUAL_PART AND NOT "DB2510_U1_F1_GRIPPER".CYL.FULL_CLOSED) OR (NOT "DB8000_PART_STATUS".UNIT_1.STATION_1.PART_A.STATUS.VIRTUAL_PART AND NOT "DB2500_UNIT_1_FIXTURE_1".DATA.CLAMPED_WITH_PART_ANALOG))) OR ("DB5000_FIX_TABLE_POSITIONS".UNIT_1.FIXTURE[3].IN_LOAD_UNLOAD_STATION_1 AND (("DB8000_PART_STATUS".UNIT_1.STATION_1.PART_A.STATUS.VIRTUAL_PART AND NOT "DB2710_U1_F3_GRIPPER".CYL.FULL_CLOSED) OR (NOT "DB8000_PART_STATUS".UNIT_1.STATION_1.PART_A.STATUS.VIRTUAL_PART AND NOT "DB2700_UNIT_1_FIXTURE_3".DATA.CLAMPED_WITH_PART_ANALOG))))) OR ("DB2440_GLOBAL_DATA".GLOBAL_DATA.U01_NR_CYCLE_PART_TYPE AND (("DB5000_FIX_TABLE_POSITIONS".UNIT_1.FIXTURE[2].IN_LOAD_UNLOAD_STATION_1 AND (("DB8000_PART_STATUS".UNIT_1.STATION_1.PART_A.STATUS.VIRTUAL_PART AND NOT "DB2610_U1_F2_GRIPPER".CYL.FULL_CLOSED) OR (NOT "DB8000_PART_STATUS".UNIT_1.STATION_2.PART_A.STATUS.VIRTUAL_PART AND NOT "DB2600_UNIT_1_FIXTURE_2".DATA.CLAMPED_WITH_PART_ANALOG))) OR ("DB5000_FIX_TABLE_POSITIONS".UNIT_1.FIXTURE[4].IN_LOAD_UNLOAD_STATION_1 AND (("DB8000_PART_STATUS".UNIT_1.STATION_1.PART_A.STATUS.VIRTUAL_PART AND NOT "DB2810_U1_F4_GRIPPER".CYL.FULL_CLOSED) OR (NOT "DB8000_PART_STATUS".UNIT_1.STATION_1.PART_A.STATUS.VIRTUAL_PART AND NOT "DB2800_UNIT_1_FIXTURE_4".DATA.CLAMPED_WITH_PART_ANALOG))))))) OR ("DB8000_PART_STATUS".UNIT_1.STATION_1.PART_A.STATUS.CELL_STATUS.U1_ONE_FACE_DONE_ROTATED AND (("DB2440_GLOBAL_DATA".GLOBAL_DATA.U01_RN_CYCLE_PART_TYPE AND (("DB5000_FIX_TABLE_POSITIONS".UNIT_1.FIXTURE[2].IN_LOAD_UNLOAD_STATION_1 AND (("DB8000_PART_STATUS".UNIT_1.STATION_1.PART_A.STATUS.VIRTUAL_PART AND NOT "DB2610_U1_F2_GRIPPER".CYL.FULL_CLOSED) OR (NOT "DB8000_PART_STATUS".UNIT_1.STATION_1.PART_A.STATUS.VIRTUAL_PART AND NOT "DB2600_UNIT_1_FIXTURE_2".DATA.CLAMPED_WITH_PART_ANALOG))) OR ("DB5000_FIX_TABLE_POSITIONS".UNIT_1.FIXTURE[4].IN_LOAD_UNLOAD_STATION_1 AND (("DB8000_PART_STATUS".UNIT_1.STATION_1.PART_A.STATUS.VIRTUAL_PART AND NOT "DB2810_U1_F4_GRIPPER".CYL.FULL_CLOSED) OR (NOT "DB8000_PART_STATUS".UNIT_1.STATION_1.PART_A.STATUS.VIRTUAL_PART AND NOT "DB2800_UNIT_1_FIXTURE_4".DATA.CLAMPED_WITH_PART_ANALOG))))) OR ("DB2440_GLOBAL_DATA".GLOBAL_DATA.U01_NR_CYCLE_PART_TYPE AND (("DB5000_FIX_TABLE_POSITIONS".UNIT_1.FIXTURE[1].IN_LOAD_UNLOAD_STATION_1 AND (("DB8000_PART_STATUS".UNIT_1.STATION_1.PART_A.STATUS.VIRTUAL_PART AND NOT "DB2510_U1_F1_GRIPPER".CYL.FULL_CLOSED) OR (NOT "DB8000_PART_STATUS".UNIT_1.STATION_1.PART_A.STATUS.VIRTUAL_PART AND NOT "DB2500_UNIT_1_FIXTURE_1".DATA.CLAMPED_WITH_PART_ANALOG))) OR ("DB5000_FIX_TABLE_POSITIONS".UNIT_1.FIXTURE[3].IN_LOAD_UNLOAD_STATION_1 AND (("DB8000_PART_STATUS".UNIT_1.STATION_1.PART_A.STATUS.VIRTUAL_PART AND NOT "DB2710_U1_F3_GRIPPER".CYL.FULL_CLOSED) OR (NOT "DB8000_PART_STATUS".UNIT_1.STATION_1.PART_A.STATUS.VIRTUAL_PART AND NOT "DB2700_UNIT_1_FIXTURE_3".DATA.CLAMPED_WITH_PART_ANALOG)))))));
END_REGION

REGION Network 17: UNIT 01 FACE DONE IN STATION 1
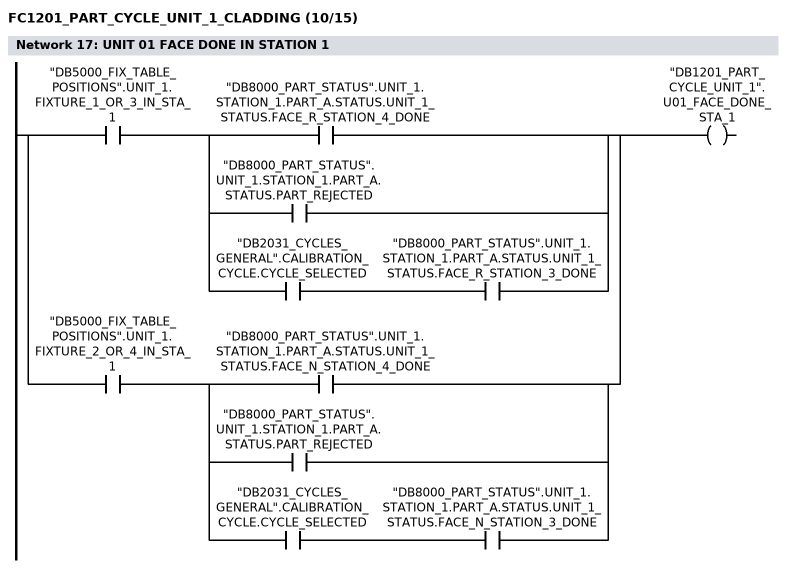
   RUNG wire#powerrail
      Contact( "DB5000_FIX_TABLE_POSITIONS".UNIT_1.FIXTURE_1_OR_3_IN_STA_1 )
      wire#w1
      Contact( "DB8000_PART_STATUS".UNIT_1.STATION_1.PART_A.STATUS.UNIT_1_STATUS.FACE_R_STATION_4_DONE )
      wire#w2
      Coil( "DB1201_PART_CYCLE_UNIT_1".U01_FACE_DONE_STA_1 )
   END_RUNG
   RUNG wire#w1
      Contact( "DB8000_PART_STATUS".UNIT_1.STATION_1.PART_A.STATUS.PART_REJECTED )
   END_RUNG wire#w2
   RUNG wire#w1
      Contact( "DB2031_CYCLES_GENERAL".CALIBRATION_CYCLE.CYCLE_SELECTED )
      Contact( "DB8000_PART_STATUS".UNIT_1.STATION_1.PART_A.STATUS.UNIT_1_STATUS.FACE_R_STATION_3_DONE )
   END_RUNG wire#w2
   RUNG wire#powerrail
      Contact( "DB5000_FIX_TABLE_POSITIONS".UNIT_1.FIXTURE_2_OR_4_IN_STA_1 )
      wire#w3
      Contact( "DB8000_PART_STATUS".UNIT_1.STATION_1.PART_A.STATUS.UNIT_1_STATUS.FACE_N_STATION_4_DONE )
   END_RUNG wire#w2
   RUNG wire#w3
      Contact( "DB8000_PART_STATUS".UNIT_1.STATION_1.PART_A.STATUS.PART_REJECTED )
   END_RUNG wire#w2
   RUNG wire#w3
      Contact( "DB2031_CYCLES_GENERAL".CALIBRATION_CYCLE.CYCLE_SELECTED )
      Contact( "DB8000_PART_STATUS".UNIT_1.STATION_1.PART_A.STATUS.UNIT_1_STATUS.FACE_N_STATION_3_DONE )
   END_RUNG wire#w2
   // the same network as SCL:
   "DB1201_PART_CYCLE_UNIT_1".U01_FACE_DONE_STA_1 := ("DB5000_FIX_TABLE_POSITIONS".UNIT_1.FIXTURE_1_OR_3_IN_STA_1 AND ("DB8000_PART_STATUS".UNIT_1.STATION_1.PART_A.STATUS.UNIT_1_STATUS.FACE_R_STATION_4_DONE OR "DB8000_PART_STATUS".UNIT_1.STATION_1.PART_A.STATUS.PART_REJECTED OR ("DB2031_CYCLES_GENERAL".CALIBRATION_CYCLE.CYCLE_SELECTED AND "DB8000_PART_STATUS".UNIT_1.STATION_1.PART_A.STATUS.UNIT_1_STATUS.FACE_R_STATION_3_DONE))) OR ("DB5000_FIX_TABLE_POSITIONS".UNIT_1.FIXTURE_2_OR_4_IN_STA_1 AND ("DB8000_PART_STATUS".UNIT_1.STATION_1.PART_A.STATUS.UNIT_1_STATUS.FACE_N_STATION_4_DONE OR "DB8000_PART_STATUS".UNIT_1.STATION_1.PART_A.STATUS.PART_REJECTED OR ("DB2031_CYCLES_GENERAL".CALIBRATION_CYCLE.CYCLE_SELECTED AND "DB8000_PART_STATUS".UNIT_1.STATION_1.PART_A.STATUS.UNIT_1_STATUS.FACE_N_STATION_3_DONE)));
END_REGION

REGION Network 18: CYCLE UNIT 01 STATION 0
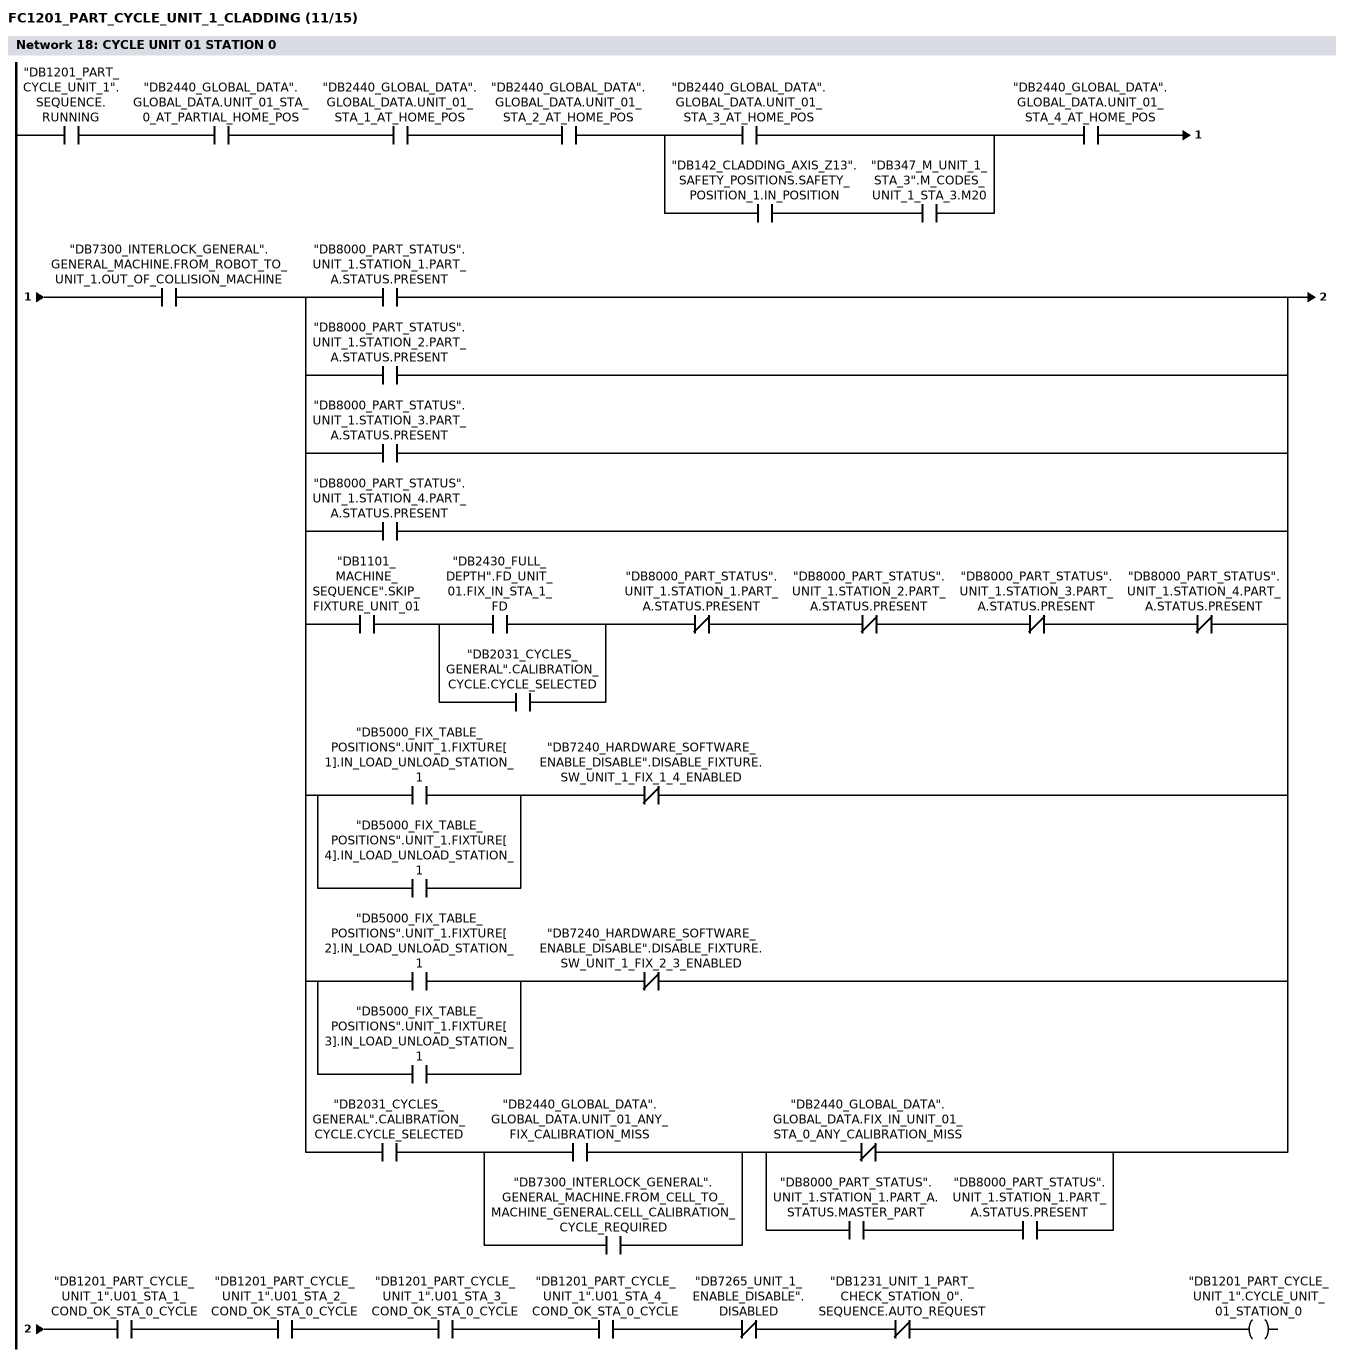
   RUNG wire#powerrail
      Contact( "DB1201_PART_CYCLE_UNIT_1".SEQUENCE.RUNNING )
      Contact( "DB2440_GLOBAL_DATA".GLOBAL_DATA.UNIT_01_STA_0_AT_PARTIAL_HOME_POS )
      Contact( "DB2440_GLOBAL_DATA".GLOBAL_DATA.UNIT_01_STA_1_AT_HOME_POS )
      Contact( "DB2440_GLOBAL_DATA".GLOBAL_DATA.UNIT_01_STA_2_AT_HOME_POS )
      wire#w1
      Contact( "DB2440_GLOBAL_DATA".GLOBAL_DATA.UNIT_01_STA_3_AT_HOME_POS )
      wire#w2
      Contact( "DB2440_GLOBAL_DATA".GLOBAL_DATA.UNIT_01_STA_4_AT_HOME_POS )
      Contact( "DB7300_INTERLOCK_GENERAL".GENERAL_MACHINE.FROM_ROBOT_TO_UNIT_1.OUT_OF_COLLISION_MACHINE )
      wire#w3
      Contact( "DB8000_PART_STATUS".UNIT_1.STATION_1.PART_A.STATUS.PRESENT )
      wire#w4
      Contact( "DB1201_PART_CYCLE_UNIT_1".U01_STA_1_COND_OK_STA_0_CYCLE )
      Contact( "DB1201_PART_CYCLE_UNIT_1".U01_STA_2_COND_OK_STA_0_CYCLE )
      Contact( "DB1201_PART_CYCLE_UNIT_1".U01_STA_3_COND_OK_STA_0_CYCLE )
      Contact( "DB1201_PART_CYCLE_UNIT_1".U01_STA_4_COND_OK_STA_0_CYCLE )
      I_Contact( "DB7265_UNIT_1_ENABLE_DISABLE".DISABLED )
      I_Contact( "DB1231_UNIT_1_PART_CHECK_STATION_0".SEQUENCE.AUTO_REQUEST )
      Coil( "DB1201_PART_CYCLE_UNIT_1".CYCLE_UNIT_01_STATION_0 )
   END_RUNG
   RUNG wire#w1
      Contact( "DB142_CLADDING_AXIS_Z13".SAFETY_POSITIONS.SAFETY_POSITION_1.IN_POSITION )
      Contact( "DB347_M_UNIT_1_STA_3".M_CODES_UNIT_1_STA_3.M20 )
   END_RUNG wire#w2
   RUNG wire#w3
      Contact( "DB8000_PART_STATUS".UNIT_1.STATION_2.PART_A.STATUS.PRESENT )
   END_RUNG wire#w4
   RUNG wire#w3
      Contact( "DB8000_PART_STATUS".UNIT_1.STATION_3.PART_A.STATUS.PRESENT )
   END_RUNG wire#w4
   RUNG wire#w3
      Contact( "DB8000_PART_STATUS".UNIT_1.STATION_4.PART_A.STATUS.PRESENT )
   END_RUNG wire#w4
   RUNG wire#w3
      Contact( "DB1101_MACHINE_SEQUENCE".SKIP_FIXTURE_UNIT_01 )
      wire#w5
      Contact( "DB2430_FULL_DEPTH".FD_UNIT_01.FIX_IN_STA_1_FD )
      wire#w6
      I_Contact( "DB8000_PART_STATUS".UNIT_1.STATION_1.PART_A.STATUS.PRESENT )
      I_Contact( "DB8000_PART_STATUS".UNIT_1.STATION_2.PART_A.STATUS.PRESENT )
      I_Contact( "DB8000_PART_STATUS".UNIT_1.STATION_3.PART_A.STATUS.PRESENT )
      I_Contact( "DB8000_PART_STATUS".UNIT_1.STATION_4.PART_A.STATUS.PRESENT )
   END_RUNG wire#w4
   RUNG wire#w5
      Contact( "DB2031_CYCLES_GENERAL".CALIBRATION_CYCLE.CYCLE_SELECTED )
   END_RUNG wire#w6
   RUNG wire#w3
      Contact( "DB5000_FIX_TABLE_POSITIONS".UNIT_1.FIXTURE[1].IN_LOAD_UNLOAD_STATION_1 )
      wire#w7
      I_Contact( "DB7240_HARDWARE_SOFTWARE_ENABLE_DISABLE".DISABLE_FIXTURE.SW_UNIT_1_FIX_1_4_ENABLED )
   END_RUNG wire#w4
   RUNG wire#w3
      Contact( "DB5000_FIX_TABLE_POSITIONS".UNIT_1.FIXTURE[4].IN_LOAD_UNLOAD_STATION_1 )
   END_RUNG wire#w7
   RUNG wire#w3
      Contact( "DB5000_FIX_TABLE_POSITIONS".UNIT_1.FIXTURE[2].IN_LOAD_UNLOAD_STATION_1 )
      wire#w8
      I_Contact( "DB7240_HARDWARE_SOFTWARE_ENABLE_DISABLE".DISABLE_FIXTURE.SW_UNIT_1_FIX_2_3_ENABLED )
   END_RUNG wire#w4
   RUNG wire#w3
      Contact( "DB5000_FIX_TABLE_POSITIONS".UNIT_1.FIXTURE[3].IN_LOAD_UNLOAD_STATION_1 )
   END_RUNG wire#w8
   RUNG wire#w3
      Contact( "DB2031_CYCLES_GENERAL".CALIBRATION_CYCLE.CYCLE_SELECTED )
      wire#w9
      Contact( "DB2440_GLOBAL_DATA".GLOBAL_DATA.UNIT_01_ANY_FIX_CALIBRATION_MISS )
      wire#w10
      I_Contact( "DB2440_GLOBAL_DATA".GLOBAL_DATA.FIX_IN_UNIT_01_STA_0_ANY_CALIBRATION_MISS )
   END_RUNG wire#w4
   RUNG wire#w9
      Contact( "DB7300_INTERLOCK_GENERAL".GENERAL_MACHINE.FROM_CELL_TO_MACHINE_GENERAL.CELL_CALIBRATION_CYCLE_REQUIRED )
   END_RUNG wire#w10
   RUNG wire#w10
      Contact( "DB8000_PART_STATUS".UNIT_1.STATION_1.PART_A.STATUS.MASTER_PART )
      Contact( "DB8000_PART_STATUS".UNIT_1.STATION_1.PART_A.STATUS.PRESENT )
   END_RUNG wire#w4
   // the same network as SCL:
   "DB1201_PART_CYCLE_UNIT_1".CYCLE_UNIT_01_STATION_0 := "DB1201_PART_CYCLE_UNIT_1".SEQUENCE.RUNNING AND "DB2440_GLOBAL_DATA".GLOBAL_DATA.UNIT_01_STA_0_AT_PARTIAL_HOME_POS AND "DB2440_GLOBAL_DATA".GLOBAL_DATA.UNIT_01_STA_1_AT_HOME_POS AND "DB2440_GLOBAL_DATA".GLOBAL_DATA.UNIT_01_STA_2_AT_HOME_POS AND ("DB2440_GLOBAL_DATA".GLOBAL_DATA.UNIT_01_STA_3_AT_HOME_POS OR ("DB142_CLADDING_AXIS_Z13".SAFETY_POSITIONS.SAFETY_POSITION_1.IN_POSITION AND "DB347_M_UNIT_1_STA_3".M_CODES_UNIT_1_STA_3.M20)) AND "DB2440_GLOBAL_DATA".GLOBAL_DATA.UNIT_01_STA_4_AT_HOME_POS AND "DB7300_INTERLOCK_GENERAL".GENERAL_MACHINE.FROM_ROBOT_TO_UNIT_1.OUT_OF_COLLISION_MACHINE AND ("DB8000_PART_STATUS".UNIT_1.STATION_1.PART_A.STATUS.PRESENT OR "DB8000_PART_STATUS".UNIT_1.STATION_2.PART_A.STATUS.PRESENT OR "DB8000_PART_STATUS".UNIT_1.STATION_3.PART_A.STATUS.PRESENT OR "DB8000_PART_STATUS".UNIT_1.STATION_4.PART_A.STATUS.PRESENT OR ("DB1101_MACHINE_SEQUENCE".SKIP_FIXTURE_UNIT_01 AND ("DB2430_FULL_DEPTH".FD_UNIT_01.FIX_IN_STA_1_FD OR "DB2031_CYCLES_GENERAL".CALIBRATION_CYCLE.CYCLE_SELECTED) AND NOT "DB8000_PART_STATUS".UNIT_1.STATION_1.PART_A.STATUS.PRESENT AND NOT "DB8000_PART_STATUS".UNIT_1.STATION_2.PART_A.STATUS.PRESENT AND NOT "DB8000_PART_STATUS".UNIT_1.STATION_3.PART_A.STATUS.PRESENT AND NOT "DB8000_PART_STATUS".UNIT_1.STATION_4.PART_A.STATUS.PRESENT) OR (("DB5000_FIX_TABLE_POSITIONS".UNIT_1.FIXTURE[1].IN_LOAD_UNLOAD_STATION_1 OR "DB5000_FIX_TABLE_POSITIONS".UNIT_1.FIXTURE[4].IN_LOAD_UNLOAD_STATION_1) AND NOT "DB7240_HARDWARE_SOFTWARE_ENABLE_DISABLE".DISABLE_FIXTURE.SW_UNIT_1_FIX_1_4_ENABLED) OR (("DB5000_FIX_TABLE_POSITIONS".UNIT_1.FIXTURE[2].IN_LOAD_UNLOAD_STATION_1 OR "DB5000_FIX_TABLE_POSITIONS".UNIT_1.FIXTURE[3].IN_LOAD_UNLOAD_STATION_1) AND NOT "DB7240_HARDWARE_SOFTWARE_ENABLE_DISABLE".DISABLE_FIXTURE.SW_UNIT_1_FIX_2_3_ENABLED) OR ("DB2031_CYCLES_GENERAL".CALIBRATION_CYCLE.CYCLE_SELECTED AND ("DB2440_GLOBAL_DATA".GLOBAL_DATA.UNIT_01_ANY_FIX_CALIBRATION_MISS OR "DB7300_INTERLOCK_GENERAL".GENERAL_MACHINE.FROM_CELL_TO_MACHINE_GENERAL.CELL_CALIBRATION_CYCLE_REQUIRED) AND (NOT "DB2440_GLOBAL_DATA".GLOBAL_DATA.FIX_IN_UNIT_01_STA_0_ANY_CALIBRATION_MISS OR ("DB8000_PART_STATUS".UNIT_1.STATION_1.PART_A.STATUS.MASTER_PART AND "DB8000_PART_STATUS".UNIT_1.STATION_1.PART_A.STATUS.PRESENT)))) AND "DB1201_PART_CYCLE_UNIT_1".U01_STA_1_COND_OK_STA_0_CYCLE AND "DB1201_PART_CYCLE_UNIT_1".U01_STA_2_COND_OK_STA_0_CYCLE AND "DB1201_PART_CYCLE_UNIT_1".U01_STA_3_COND_OK_STA_0_CYCLE AND "DB1201_PART_CYCLE_UNIT_1".U01_STA_4_COND_OK_STA_0_CYCLE AND NOT "DB7265_UNIT_1_ENABLE_DISABLE".DISABLED AND NOT "DB1231_UNIT_1_PART_CHECK_STATION_0".SEQUENCE.AUTO_REQUEST;
END_REGION

REGION Network 19: CYCLE UNIT 01 STATION 1
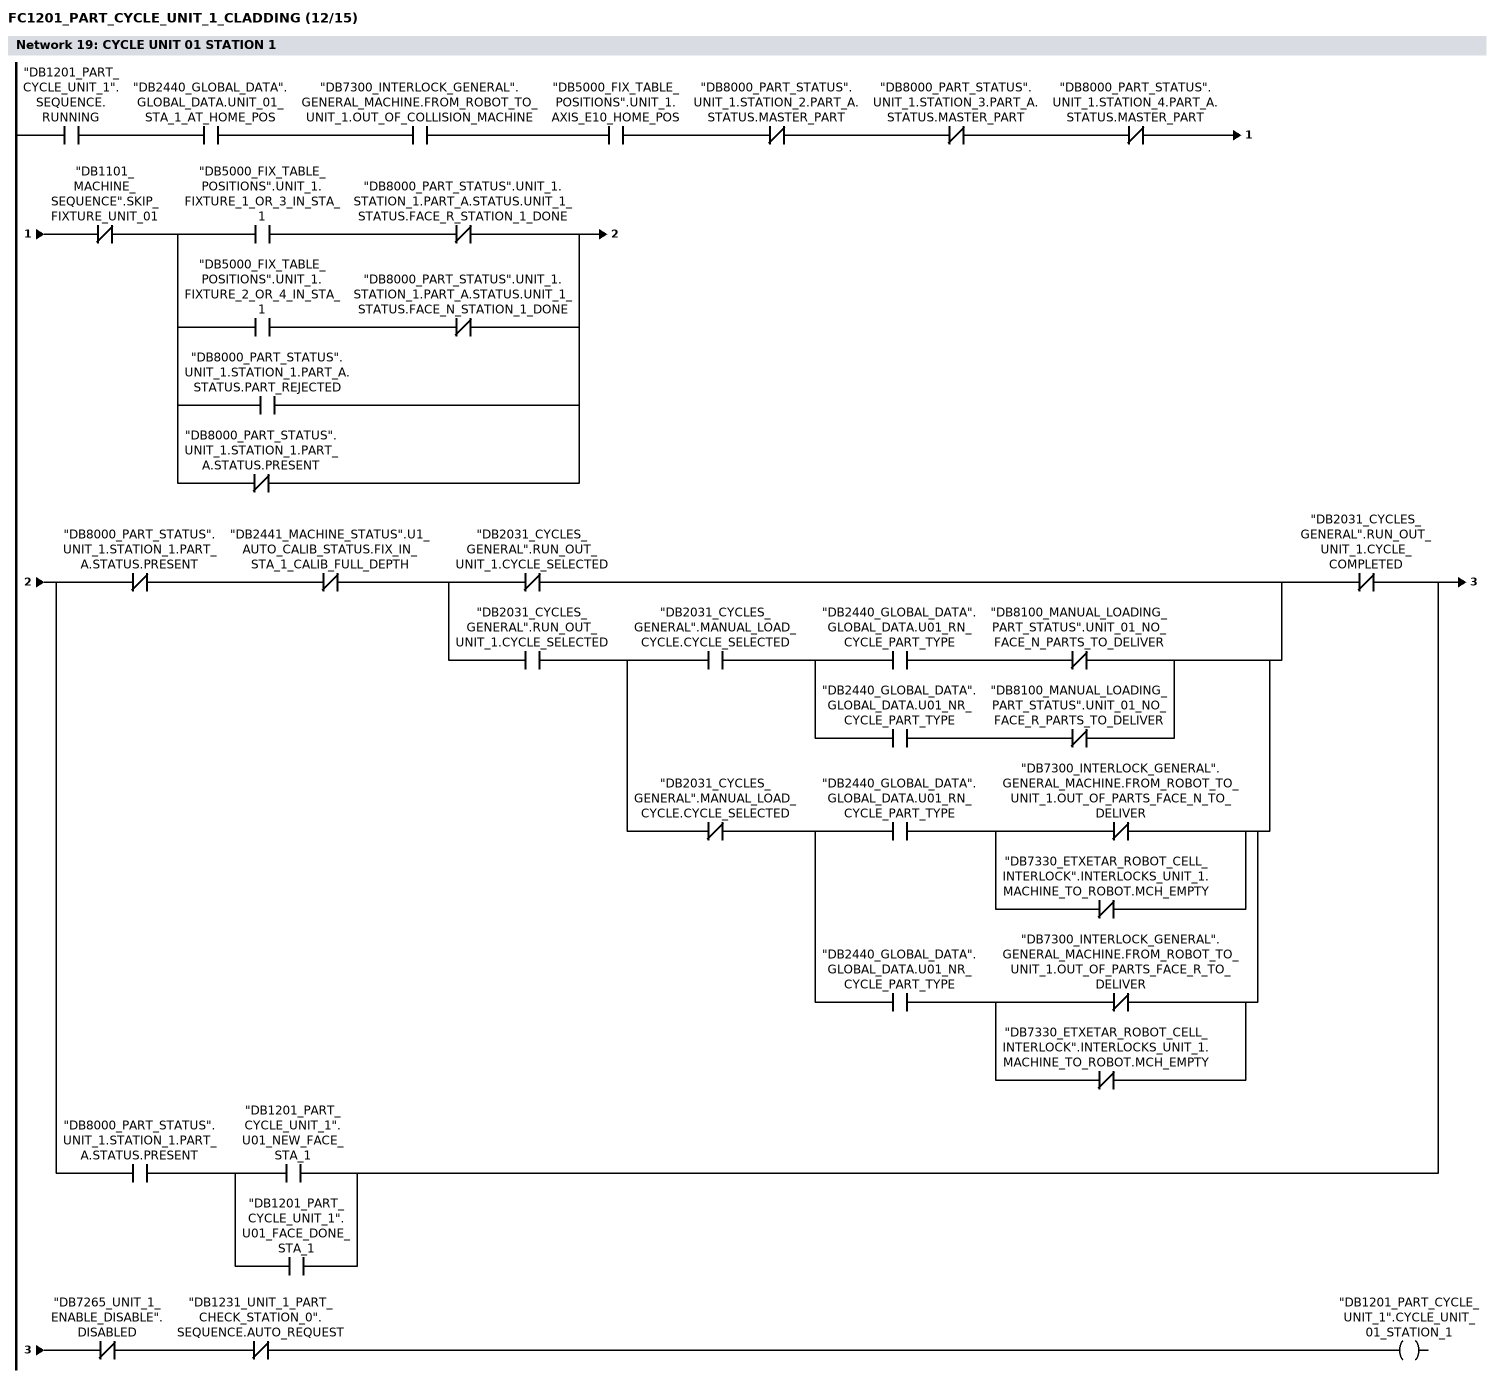
   RUNG wire#powerrail
      Contact( "DB1201_PART_CYCLE_UNIT_1".SEQUENCE.RUNNING )
      Contact( "DB2440_GLOBAL_DATA".GLOBAL_DATA.UNIT_01_STA_1_AT_HOME_POS )
      Contact( "DB7300_INTERLOCK_GENERAL".GENERAL_MACHINE.FROM_ROBOT_TO_UNIT_1.OUT_OF_COLLISION_MACHINE )
      Contact( "DB5000_FIX_TABLE_POSITIONS".UNIT_1.AXIS_E10_HOME_POS )
      I_Contact( "DB8000_PART_STATUS".UNIT_1.STATION_2.PART_A.STATUS.MASTER_PART )
      I_Contact( "DB8000_PART_STATUS".UNIT_1.STATION_3.PART_A.STATUS.MASTER_PART )
      I_Contact( "DB8000_PART_STATUS".UNIT_1.STATION_4.PART_A.STATUS.MASTER_PART )
      I_Contact( "DB1101_MACHINE_SEQUENCE".SKIP_FIXTURE_UNIT_01 )
      wire#w1
      Contact( "DB5000_FIX_TABLE_POSITIONS".UNIT_1.FIXTURE_1_OR_3_IN_STA_1 )
      I_Contact( "DB8000_PART_STATUS".UNIT_1.STATION_1.PART_A.STATUS.UNIT_1_STATUS.FACE_R_STATION_1_DONE )
      wire#w2
      I_Contact( "DB8000_PART_STATUS".UNIT_1.STATION_1.PART_A.STATUS.PRESENT )
      I_Contact( "DB2441_MACHINE_STATUS".U1_AUTO_CALIB_STATUS.FIX_IN_STA_1_CALIB_FULL_DEPTH )
      wire#w3
      I_Contact( "DB2031_CYCLES_GENERAL".RUN_OUT_UNIT_1.CYCLE_SELECTED )
      wire#w4
      I_Contact( "DB2031_CYCLES_GENERAL".RUN_OUT_UNIT_1.CYCLE_COMPLETED )
      wire#w10
      I_Contact( "DB7265_UNIT_1_ENABLE_DISABLE".DISABLED )
      I_Contact( "DB1231_UNIT_1_PART_CHECK_STATION_0".SEQUENCE.AUTO_REQUEST )
      Coil( "DB1201_PART_CYCLE_UNIT_1".CYCLE_UNIT_01_STATION_1 )
   END_RUNG
   RUNG wire#w1
      Contact( "DB5000_FIX_TABLE_POSITIONS".UNIT_1.FIXTURE_2_OR_4_IN_STA_1 )
      I_Contact( "DB8000_PART_STATUS".UNIT_1.STATION_1.PART_A.STATUS.UNIT_1_STATUS.FACE_N_STATION_1_DONE )
   END_RUNG wire#w2
   RUNG wire#w1
      Contact( "DB8000_PART_STATUS".UNIT_1.STATION_1.PART_A.STATUS.PART_REJECTED )
   END_RUNG wire#w2
   RUNG wire#w1
      I_Contact( "DB8000_PART_STATUS".UNIT_1.STATION_1.PART_A.STATUS.PRESENT )
   END_RUNG wire#w2
   RUNG wire#w3
      Contact( "DB2031_CYCLES_GENERAL".RUN_OUT_UNIT_1.CYCLE_SELECTED )
      wire#w5
      Contact( "DB2031_CYCLES_GENERAL".MANUAL_LOAD_CYCLE.CYCLE_SELECTED )
      wire#w6
      Contact( "DB2440_GLOBAL_DATA".GLOBAL_DATA.U01_RN_CYCLE_PART_TYPE )
      I_Contact( "DB8100_MANUAL_LOADING_PART_STATUS".UNIT_01_NO_FACE_N_PARTS_TO_DELIVER )
   END_RUNG wire#w4
   RUNG wire#w6
      Contact( "DB2440_GLOBAL_DATA".GLOBAL_DATA.U01_NR_CYCLE_PART_TYPE )
      I_Contact( "DB8100_MANUAL_LOADING_PART_STATUS".UNIT_01_NO_FACE_R_PARTS_TO_DELIVER )
   END_RUNG wire#w4
   RUNG wire#w5
      I_Contact( "DB2031_CYCLES_GENERAL".MANUAL_LOAD_CYCLE.CYCLE_SELECTED )
      wire#w7
      Contact( "DB2440_GLOBAL_DATA".GLOBAL_DATA.U01_RN_CYCLE_PART_TYPE )
      wire#w8
      I_Contact( "DB7300_INTERLOCK_GENERAL".GENERAL_MACHINE.FROM_ROBOT_TO_UNIT_1.OUT_OF_PARTS_FACE_N_TO_DELIVER )
   END_RUNG wire#w4
   RUNG wire#w8
      I_Contact( "DB7330_ETXETAR_ROBOT_CELL_INTERLOCK".INTERLOCKS_UNIT_1.MACHINE_TO_ROBOT.MCH_EMPTY )
   END_RUNG wire#w4
   RUNG wire#w7
      Contact( "DB2440_GLOBAL_DATA".GLOBAL_DATA.U01_NR_CYCLE_PART_TYPE )
      wire#w9
      I_Contact( "DB7300_INTERLOCK_GENERAL".GENERAL_MACHINE.FROM_ROBOT_TO_UNIT_1.OUT_OF_PARTS_FACE_R_TO_DELIVER )
   END_RUNG wire#w4
   RUNG wire#w9
      I_Contact( "DB7330_ETXETAR_ROBOT_CELL_INTERLOCK".INTERLOCKS_UNIT_1.MACHINE_TO_ROBOT.MCH_EMPTY )
   END_RUNG wire#w4
   RUNG wire#w2
      Contact( "DB8000_PART_STATUS".UNIT_1.STATION_1.PART_A.STATUS.PRESENT )
      wire#w11
      Contact( "DB1201_PART_CYCLE_UNIT_1".U01_NEW_FACE_STA_1 )
   END_RUNG wire#w10
   RUNG wire#w11
      Contact( "DB1201_PART_CYCLE_UNIT_1".U01_FACE_DONE_STA_1 )
   END_RUNG wire#w10
   // the same network as SCL:
   "DB1201_PART_CYCLE_UNIT_1".CYCLE_UNIT_01_STATION_1 := "DB1201_PART_CYCLE_UNIT_1".SEQUENCE.RUNNING AND "DB2440_GLOBAL_DATA".GLOBAL_DATA.UNIT_01_STA_1_AT_HOME_POS AND "DB7300_INTERLOCK_GENERAL".GENERAL_MACHINE.FROM_ROBOT_TO_UNIT_1.OUT_OF_COLLISION_MACHINE AND "DB5000_FIX_TABLE_POSITIONS".UNIT_1.AXIS_E10_HOME_POS AND NOT "DB8000_PART_STATUS".UNIT_1.STATION_2.PART_A.STATUS.MASTER_PART AND NOT "DB8000_PART_STATUS".UNIT_1.STATION_3.PART_A.STATUS.MASTER_PART AND NOT "DB8000_PART_STATUS".UNIT_1.STATION_4.PART_A.STATUS.MASTER_PART AND NOT "DB1101_MACHINE_SEQUENCE".SKIP_FIXTURE_UNIT_01 AND (("DB5000_FIX_TABLE_POSITIONS".UNIT_1.FIXTURE_1_OR_3_IN_STA_1 AND NOT "DB8000_PART_STATUS".UNIT_1.STATION_1.PART_A.STATUS.UNIT_1_STATUS.FACE_R_STATION_1_DONE) OR ("DB5000_FIX_TABLE_POSITIONS".UNIT_1.FIXTURE_2_OR_4_IN_STA_1 AND NOT "DB8000_PART_STATUS".UNIT_1.STATION_1.PART_A.STATUS.UNIT_1_STATUS.FACE_N_STATION_1_DONE) OR "DB8000_PART_STATUS".UNIT_1.STATION_1.PART_A.STATUS.PART_REJECTED OR NOT "DB8000_PART_STATUS".UNIT_1.STATION_1.PART_A.STATUS.PRESENT) AND ((NOT "DB8000_PART_STATUS".UNIT_1.STATION_1.PART_A.STATUS.PRESENT AND NOT "DB2441_MACHINE_STATUS".U1_AUTO_CALIB_STATUS.FIX_IN_STA_1_CALIB_FULL_DEPTH AND (NOT "DB2031_CYCLES_GENERAL".RUN_OUT_UNIT_1.CYCLE_SELECTED OR ("DB2031_CYCLES_GENERAL".RUN_OUT_UNIT_1.CYCLE_SELECTED AND (("DB2031_CYCLES_GENERAL".MANUAL_LOAD_CYCLE.CYCLE_SELECTED AND (("DB2440_GLOBAL_DATA".GLOBAL_DATA.U01_RN_CYCLE_PART_TYPE AND NOT "DB8100_MANUAL_LOADING_PART_STATUS".UNIT_01_NO_FACE_N_PARTS_TO_DELIVER) OR ("DB2440_GLOBAL_DATA".GLOBAL_DATA.U01_NR_CYCLE_PART_TYPE AND NOT "DB8100_MANUAL_LOADING_PART_STATUS".UNIT_01_NO_FACE_R_PARTS_TO_DELIVER))) OR (NOT "DB2031_CYCLES_GENERAL".MANUAL_LOAD_CYCLE.CYCLE_SELECTED AND (("DB2440_GLOBAL_DATA".GLOBAL_DATA.U01_RN_CYCLE_PART_TYPE AND (NOT "DB7300_INTERLOCK_GENERAL".GENERAL_MACHINE.FROM_ROBOT_TO_UNIT_1.OUT_OF_PARTS_FACE_N_TO_DELIVER OR NOT "DB7330_ETXETAR_ROBOT_CELL_INTERLOCK".INTERLOCKS_UNIT_1.MACHINE_TO_ROBOT.MCH_EMPTY)) OR ("DB2440_GLOBAL_DATA".GLOBAL_DATA.U01_NR_CYCLE_PART_TYPE AND (NOT "DB7300_INTERLOCK_GENERAL".GENERAL_MACHINE.FROM_ROBOT_TO_UNIT_1.OUT_OF_PARTS_FACE_R_TO_DELIVER OR NOT "DB7330_ETXETAR_ROBOT_CELL_INTERLOCK".INTERLOCKS_UNIT_1.MACHINE_TO_ROBOT.MCH_EMPTY))))))) AND NOT "DB2031_CYCLES_GENERAL".RUN_OUT_UNIT_1.CYCLE_COMPLETED) OR ("DB8000_PART_STATUS".UNIT_1.STATION_1.PART_A.STATUS.PRESENT AND ("DB1201_PART_CYCLE_UNIT_1".U01_NEW_FACE_STA_1 OR "DB1201_PART_CYCLE_UNIT_1".U01_FACE_DONE_STA_1))) AND NOT "DB7265_UNIT_1_ENABLE_DISABLE".DISABLED AND NOT "DB1231_UNIT_1_PART_CHECK_STATION_0".SEQUENCE.AUTO_REQUEST;
END_REGION

REGION Network 20: CYCLE UNIT 01 STATION 2
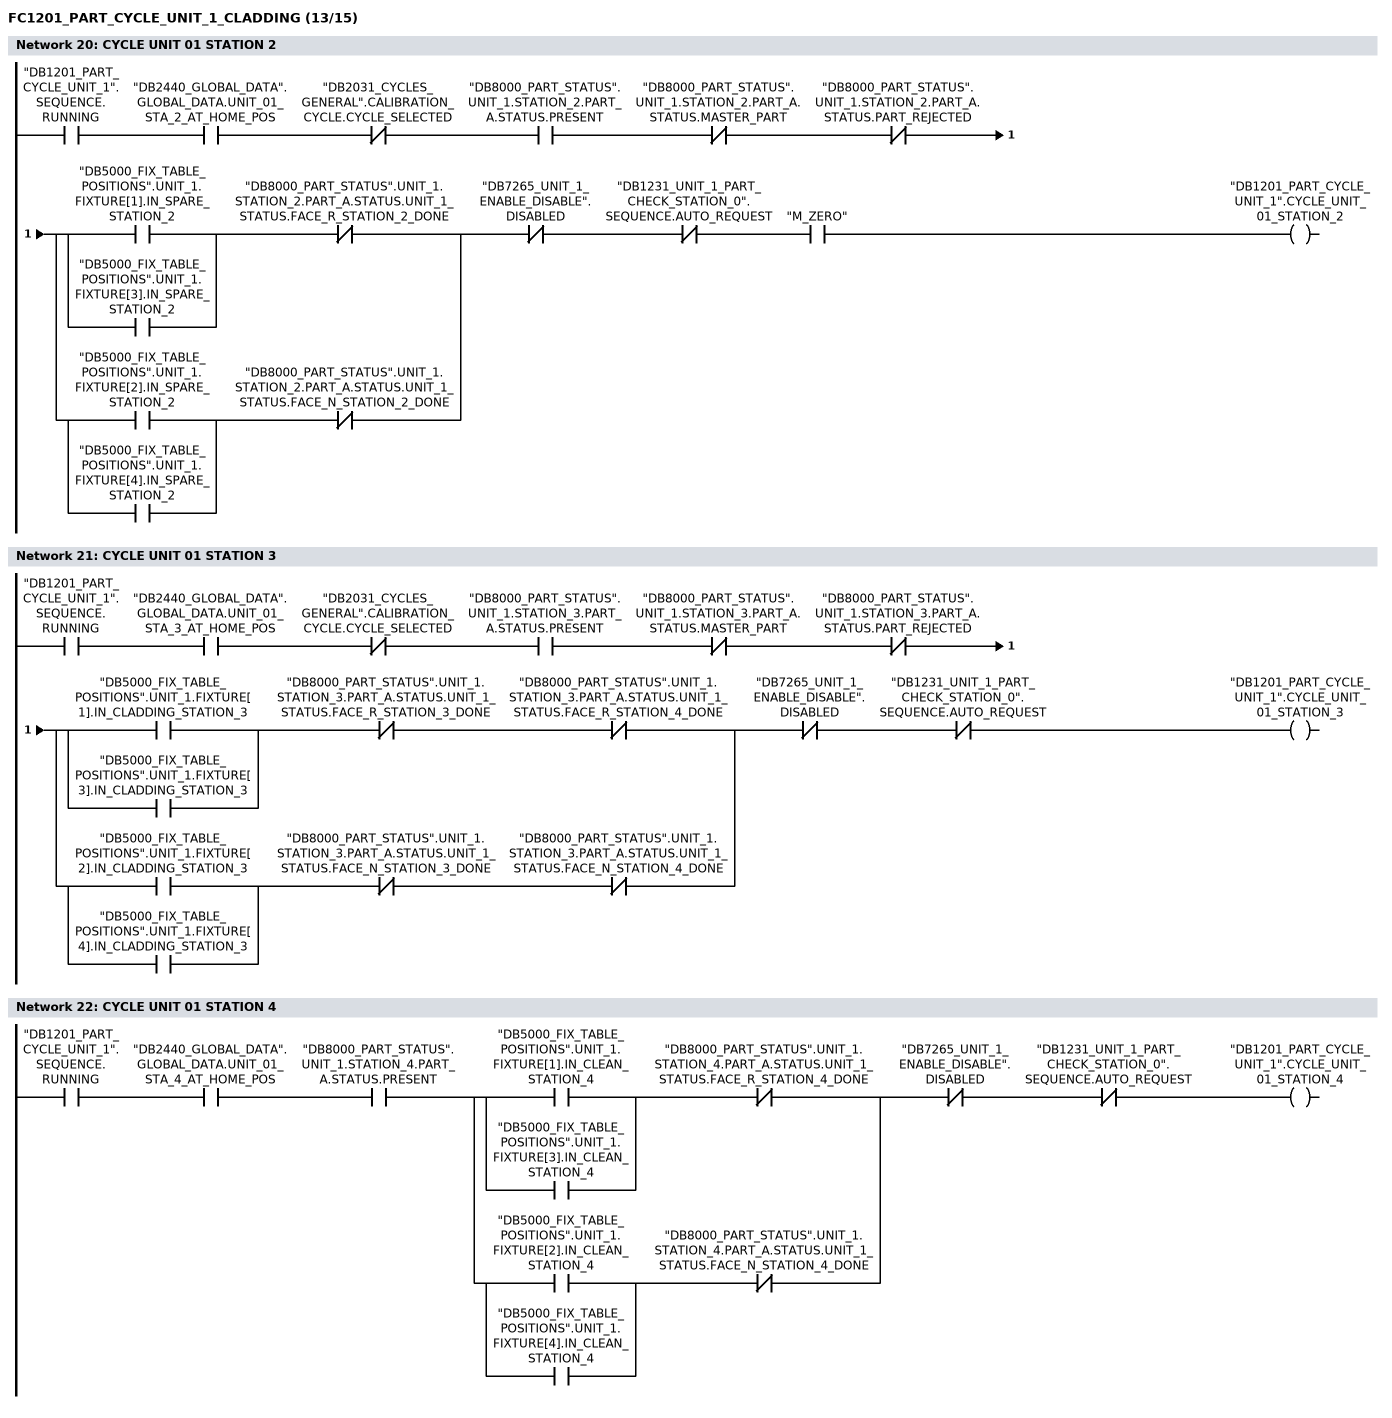
   RUNG wire#powerrail
      Contact( "DB1201_PART_CYCLE_UNIT_1".SEQUENCE.RUNNING )
      Contact( "DB2440_GLOBAL_DATA".GLOBAL_DATA.UNIT_01_STA_2_AT_HOME_POS )
      I_Contact( "DB2031_CYCLES_GENERAL".CALIBRATION_CYCLE.CYCLE_SELECTED )
      Contact( "DB8000_PART_STATUS".UNIT_1.STATION_2.PART_A.STATUS.PRESENT )
      I_Contact( "DB8000_PART_STATUS".UNIT_1.STATION_2.PART_A.STATUS.MASTER_PART )
      I_Contact( "DB8000_PART_STATUS".UNIT_1.STATION_2.PART_A.STATUS.PART_REJECTED )
      wire#w1
      Contact( "DB5000_FIX_TABLE_POSITIONS".UNIT_1.FIXTURE[1].IN_SPARE_STATION_2 )
      wire#w2
      I_Contact( "DB8000_PART_STATUS".UNIT_1.STATION_2.PART_A.STATUS.UNIT_1_STATUS.FACE_R_STATION_2_DONE )
      wire#w3
      I_Contact( "DB7265_UNIT_1_ENABLE_DISABLE".DISABLED )
      I_Contact( "DB1231_UNIT_1_PART_CHECK_STATION_0".SEQUENCE.AUTO_REQUEST )
      Contact( "M_ZERO" )
      Coil( "DB1201_PART_CYCLE_UNIT_1".CYCLE_UNIT_01_STATION_2 )
   END_RUNG
   RUNG wire#w1
      Contact( "DB5000_FIX_TABLE_POSITIONS".UNIT_1.FIXTURE[3].IN_SPARE_STATION_2 )
   END_RUNG wire#w2
   RUNG wire#w1
      Contact( "DB5000_FIX_TABLE_POSITIONS".UNIT_1.FIXTURE[2].IN_SPARE_STATION_2 )
      wire#w4
      I_Contact( "DB8000_PART_STATUS".UNIT_1.STATION_2.PART_A.STATUS.UNIT_1_STATUS.FACE_N_STATION_2_DONE )
   END_RUNG wire#w3
   RUNG wire#w1
      Contact( "DB5000_FIX_TABLE_POSITIONS".UNIT_1.FIXTURE[4].IN_SPARE_STATION_2 )
   END_RUNG wire#w4
   // the same network as SCL:
   "DB1201_PART_CYCLE_UNIT_1".CYCLE_UNIT_01_STATION_2 := "DB1201_PART_CYCLE_UNIT_1".SEQUENCE.RUNNING AND "DB2440_GLOBAL_DATA".GLOBAL_DATA.UNIT_01_STA_2_AT_HOME_POS AND NOT "DB2031_CYCLES_GENERAL".CALIBRATION_CYCLE.CYCLE_SELECTED AND "DB8000_PART_STATUS".UNIT_1.STATION_2.PART_A.STATUS.PRESENT AND NOT "DB8000_PART_STATUS".UNIT_1.STATION_2.PART_A.STATUS.MASTER_PART AND NOT "DB8000_PART_STATUS".UNIT_1.STATION_2.PART_A.STATUS.PART_REJECTED AND ((("DB5000_FIX_TABLE_POSITIONS".UNIT_1.FIXTURE[1].IN_SPARE_STATION_2 OR "DB5000_FIX_TABLE_POSITIONS".UNIT_1.FIXTURE[3].IN_SPARE_STATION_2) AND NOT "DB8000_PART_STATUS".UNIT_1.STATION_2.PART_A.STATUS.UNIT_1_STATUS.FACE_R_STATION_2_DONE) OR (("DB5000_FIX_TABLE_POSITIONS".UNIT_1.FIXTURE[2].IN_SPARE_STATION_2 OR "DB5000_FIX_TABLE_POSITIONS".UNIT_1.FIXTURE[4].IN_SPARE_STATION_2) AND NOT "DB8000_PART_STATUS".UNIT_1.STATION_2.PART_A.STATUS.UNIT_1_STATUS.FACE_N_STATION_2_DONE)) AND NOT "DB7265_UNIT_1_ENABLE_DISABLE".DISABLED AND NOT "DB1231_UNIT_1_PART_CHECK_STATION_0".SEQUENCE.AUTO_REQUEST AND "M_ZERO";
END_REGION

REGION Network 21: CYCLE UNIT 01 STATION 3
   RUNG wire#powerrail
      Contact( "DB1201_PART_CYCLE_UNIT_1".SEQUENCE.RUNNING )
      Contact( "DB2440_GLOBAL_DATA".GLOBAL_DATA.UNIT_01_STA_3_AT_HOME_POS )
      I_Contact( "DB2031_CYCLES_GENERAL".CALIBRATION_CYCLE.CYCLE_SELECTED )
      Contact( "DB8000_PART_STATUS".UNIT_1.STATION_3.PART_A.STATUS.PRESENT )
      I_Contact( "DB8000_PART_STATUS".UNIT_1.STATION_3.PART_A.STATUS.MASTER_PART )
      I_Contact( "DB8000_PART_STATUS".UNIT_1.STATION_3.PART_A.STATUS.PART_REJECTED )
      wire#w1
      Contact( "DB5000_FIX_TABLE_POSITIONS".UNIT_1.FIXTURE[1].IN_CLADDING_STATION_3 )
      wire#w2
      I_Contact( "DB8000_PART_STATUS".UNIT_1.STATION_3.PART_A.STATUS.UNIT_1_STATUS.FACE_R_STATION_3_DONE )
      I_Contact( "DB8000_PART_STATUS".UNIT_1.STATION_3.PART_A.STATUS.UNIT_1_STATUS.FACE_R_STATION_4_DONE )
      wire#w3
      I_Contact( "DB7265_UNIT_1_ENABLE_DISABLE".DISABLED )
      I_Contact( "DB1231_UNIT_1_PART_CHECK_STATION_0".SEQUENCE.AUTO_REQUEST )
      Coil( "DB1201_PART_CYCLE_UNIT_1".CYCLE_UNIT_01_STATION_3 )
   END_RUNG
   RUNG wire#w1
      Contact( "DB5000_FIX_TABLE_POSITIONS".UNIT_1.FIXTURE[3].IN_CLADDING_STATION_3 )
   END_RUNG wire#w2
   RUNG wire#w1
      Contact( "DB5000_FIX_TABLE_POSITIONS".UNIT_1.FIXTURE[2].IN_CLADDING_STATION_3 )
      wire#w4
      I_Contact( "DB8000_PART_STATUS".UNIT_1.STATION_3.PART_A.STATUS.UNIT_1_STATUS.FACE_N_STATION_3_DONE )
      I_Contact( "DB8000_PART_STATUS".UNIT_1.STATION_3.PART_A.STATUS.UNIT_1_STATUS.FACE_N_STATION_4_DONE )
   END_RUNG wire#w3
   RUNG wire#w1
      Contact( "DB5000_FIX_TABLE_POSITIONS".UNIT_1.FIXTURE[4].IN_CLADDING_STATION_3 )
   END_RUNG wire#w4
   // the same network as SCL:
   "DB1201_PART_CYCLE_UNIT_1".CYCLE_UNIT_01_STATION_3 := "DB1201_PART_CYCLE_UNIT_1".SEQUENCE.RUNNING AND "DB2440_GLOBAL_DATA".GLOBAL_DATA.UNIT_01_STA_3_AT_HOME_POS AND NOT "DB2031_CYCLES_GENERAL".CALIBRATION_CYCLE.CYCLE_SELECTED AND "DB8000_PART_STATUS".UNIT_1.STATION_3.PART_A.STATUS.PRESENT AND NOT "DB8000_PART_STATUS".UNIT_1.STATION_3.PART_A.STATUS.MASTER_PART AND NOT "DB8000_PART_STATUS".UNIT_1.STATION_3.PART_A.STATUS.PART_REJECTED AND ((("DB5000_FIX_TABLE_POSITIONS".UNIT_1.FIXTURE[1].IN_CLADDING_STATION_3 OR "DB5000_FIX_TABLE_POSITIONS".UNIT_1.FIXTURE[3].IN_CLADDING_STATION_3) AND NOT "DB8000_PART_STATUS".UNIT_1.STATION_3.PART_A.STATUS.UNIT_1_STATUS.FACE_R_STATION_3_DONE AND NOT "DB8000_PART_STATUS".UNIT_1.STATION_3.PART_A.STATUS.UNIT_1_STATUS.FACE_R_STATION_4_DONE) OR (("DB5000_FIX_TABLE_POSITIONS".UNIT_1.FIXTURE[2].IN_CLADDING_STATION_3 OR "DB5000_FIX_TABLE_POSITIONS".UNIT_1.FIXTURE[4].IN_CLADDING_STATION_3) AND NOT "DB8000_PART_STATUS".UNIT_1.STATION_3.PART_A.STATUS.UNIT_1_STATUS.FACE_N_STATION_3_DONE AND NOT "DB8000_PART_STATUS".UNIT_1.STATION_3.PART_A.STATUS.UNIT_1_STATUS.FACE_N_STATION_4_DONE)) AND NOT "DB7265_UNIT_1_ENABLE_DISABLE".DISABLED AND NOT "DB1231_UNIT_1_PART_CHECK_STATION_0".SEQUENCE.AUTO_REQUEST;
END_REGION

REGION Network 22: CYCLE UNIT 01 STATION 4
   RUNG wire#powerrail
      Contact( "DB1201_PART_CYCLE_UNIT_1".SEQUENCE.RUNNING )
      Contact( "DB2440_GLOBAL_DATA".GLOBAL_DATA.UNIT_01_STA_4_AT_HOME_POS )
      Contact( "DB8000_PART_STATUS".UNIT_1.STATION_4.PART_A.STATUS.PRESENT )
      wire#w1
      Contact( "DB5000_FIX_TABLE_POSITIONS".UNIT_1.FIXTURE[1].IN_CLEAN_STATION_4 )
      wire#w2
      I_Contact( "DB8000_PART_STATUS".UNIT_1.STATION_4.PART_A.STATUS.UNIT_1_STATUS.FACE_R_STATION_4_DONE )
      wire#w3
      I_Contact( "DB7265_UNIT_1_ENABLE_DISABLE".DISABLED )
      I_Contact( "DB1231_UNIT_1_PART_CHECK_STATION_0".SEQUENCE.AUTO_REQUEST )
      Coil( "DB1201_PART_CYCLE_UNIT_1".CYCLE_UNIT_01_STATION_4 )
   END_RUNG
   RUNG wire#w1
      Contact( "DB5000_FIX_TABLE_POSITIONS".UNIT_1.FIXTURE[3].IN_CLEAN_STATION_4 )
   END_RUNG wire#w2
   RUNG wire#w1
      Contact( "DB5000_FIX_TABLE_POSITIONS".UNIT_1.FIXTURE[2].IN_CLEAN_STATION_4 )
      wire#w4
      I_Contact( "DB8000_PART_STATUS".UNIT_1.STATION_4.PART_A.STATUS.UNIT_1_STATUS.FACE_N_STATION_4_DONE )
   END_RUNG wire#w3
   RUNG wire#w1
      Contact( "DB5000_FIX_TABLE_POSITIONS".UNIT_1.FIXTURE[4].IN_CLEAN_STATION_4 )
   END_RUNG wire#w4
   // the same network as SCL:
   "DB1201_PART_CYCLE_UNIT_1".CYCLE_UNIT_01_STATION_4 := "DB1201_PART_CYCLE_UNIT_1".SEQUENCE.RUNNING AND "DB2440_GLOBAL_DATA".GLOBAL_DATA.UNIT_01_STA_4_AT_HOME_POS AND "DB8000_PART_STATUS".UNIT_1.STATION_4.PART_A.STATUS.PRESENT AND ((("DB5000_FIX_TABLE_POSITIONS".UNIT_1.FIXTURE[1].IN_CLEAN_STATION_4 OR "DB5000_FIX_TABLE_POSITIONS".UNIT_1.FIXTURE[3].IN_CLEAN_STATION_4) AND NOT "DB8000_PART_STATUS".UNIT_1.STATION_4.PART_A.STATUS.UNIT_1_STATUS.FACE_R_STATION_4_DONE) OR (("DB5000_FIX_TABLE_POSITIONS".UNIT_1.FIXTURE[2].IN_CLEAN_STATION_4 OR "DB5000_FIX_TABLE_POSITIONS".UNIT_1.FIXTURE[4].IN_CLEAN_STATION_4) AND NOT "DB8000_PART_STATUS".UNIT_1.STATION_4.PART_A.STATUS.UNIT_1_STATUS.FACE_N_STATION_4_DONE)) AND NOT "DB7265_UNIT_1_ENABLE_DISABLE".DISABLED AND NOT "DB1231_UNIT_1_PART_CHECK_STATION_0".SEQUENCE.AUTO_REQUEST;
END_REGION

REGION Network 23: UNIT 01 STATION 3 CALIBRATION
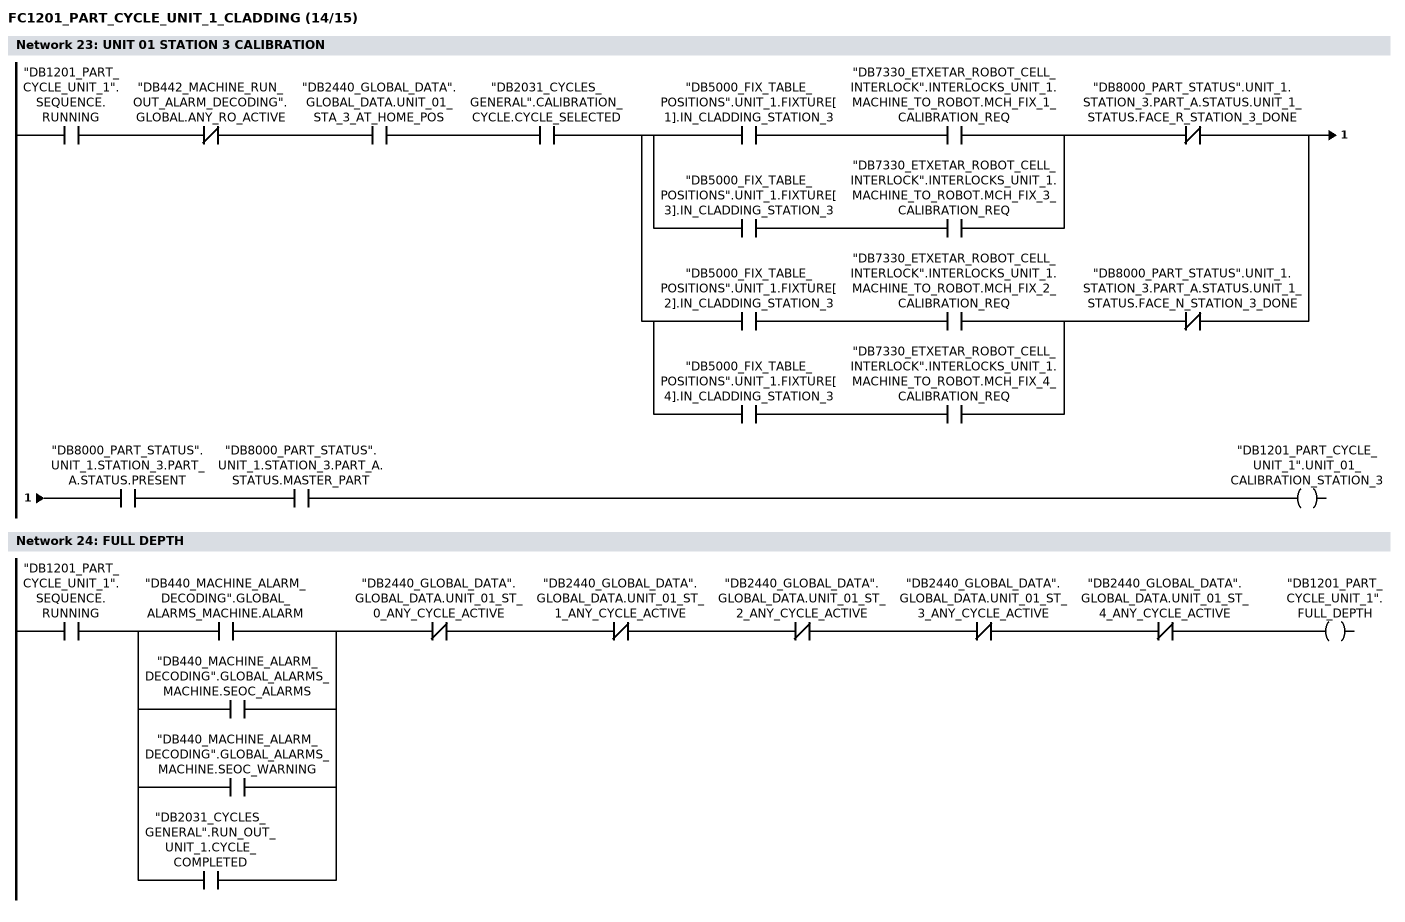
   RUNG wire#powerrail
      Contact( "DB1201_PART_CYCLE_UNIT_1".SEQUENCE.RUNNING )
      I_Contact( "DB442_MACHINE_RUN_OUT_ALARM_DECODING".GLOBAL.ANY_RO_ACTIVE )
      Contact( "DB2440_GLOBAL_DATA".GLOBAL_DATA.UNIT_01_STA_3_AT_HOME_POS )
      Contact( "DB2031_CYCLES_GENERAL".CALIBRATION_CYCLE.CYCLE_SELECTED )
      wire#w1
      Contact( "DB5000_FIX_TABLE_POSITIONS".UNIT_1.FIXTURE[1].IN_CLADDING_STATION_3 )
      Contact( "DB7330_ETXETAR_ROBOT_CELL_INTERLOCK".INTERLOCKS_UNIT_1.MACHINE_TO_ROBOT.MCH_FIX_1_CALIBRATION_REQ )
      wire#w2
      I_Contact( "DB8000_PART_STATUS".UNIT_1.STATION_3.PART_A.STATUS.UNIT_1_STATUS.FACE_R_STATION_3_DONE )
      wire#w3
      Contact( "DB8000_PART_STATUS".UNIT_1.STATION_3.PART_A.STATUS.PRESENT )
      Contact( "DB8000_PART_STATUS".UNIT_1.STATION_3.PART_A.STATUS.MASTER_PART )
      Coil( "DB1201_PART_CYCLE_UNIT_1".UNIT_01_CALIBRATION_STATION_3 )
   END_RUNG
   RUNG wire#w1
      Contact( "DB5000_FIX_TABLE_POSITIONS".UNIT_1.FIXTURE[3].IN_CLADDING_STATION_3 )
      Contact( "DB7330_ETXETAR_ROBOT_CELL_INTERLOCK".INTERLOCKS_UNIT_1.MACHINE_TO_ROBOT.MCH_FIX_3_CALIBRATION_REQ )
   END_RUNG wire#w2
   RUNG wire#w1
      Contact( "DB5000_FIX_TABLE_POSITIONS".UNIT_1.FIXTURE[2].IN_CLADDING_STATION_3 )
      Contact( "DB7330_ETXETAR_ROBOT_CELL_INTERLOCK".INTERLOCKS_UNIT_1.MACHINE_TO_ROBOT.MCH_FIX_2_CALIBRATION_REQ )
      wire#w4
      I_Contact( "DB8000_PART_STATUS".UNIT_1.STATION_3.PART_A.STATUS.UNIT_1_STATUS.FACE_N_STATION_3_DONE )
   END_RUNG wire#w3
   RUNG wire#w1
      Contact( "DB5000_FIX_TABLE_POSITIONS".UNIT_1.FIXTURE[4].IN_CLADDING_STATION_3 )
      Contact( "DB7330_ETXETAR_ROBOT_CELL_INTERLOCK".INTERLOCKS_UNIT_1.MACHINE_TO_ROBOT.MCH_FIX_4_CALIBRATION_REQ )
   END_RUNG wire#w4
   // the same network as SCL:
   "DB1201_PART_CYCLE_UNIT_1".UNIT_01_CALIBRATION_STATION_3 := "DB1201_PART_CYCLE_UNIT_1".SEQUENCE.RUNNING AND NOT "DB442_MACHINE_RUN_OUT_ALARM_DECODING".GLOBAL.ANY_RO_ACTIVE AND "DB2440_GLOBAL_DATA".GLOBAL_DATA.UNIT_01_STA_3_AT_HOME_POS AND "DB2031_CYCLES_GENERAL".CALIBRATION_CYCLE.CYCLE_SELECTED AND (((("DB5000_FIX_TABLE_POSITIONS".UNIT_1.FIXTURE[1].IN_CLADDING_STATION_3 AND "DB7330_ETXETAR_ROBOT_CELL_INTERLOCK".INTERLOCKS_UNIT_1.MACHINE_TO_ROBOT.MCH_FIX_1_CALIBRATION_REQ) OR ("DB5000_FIX_TABLE_POSITIONS".UNIT_1.FIXTURE[3].IN_CLADDING_STATION_3 AND "DB7330_ETXETAR_ROBOT_CELL_INTERLOCK".INTERLOCKS_UNIT_1.MACHINE_TO_ROBOT.MCH_FIX_3_CALIBRATION_REQ)) AND NOT "DB8000_PART_STATUS".UNIT_1.STATION_3.PART_A.STATUS.UNIT_1_STATUS.FACE_R_STATION_3_DONE) OR ((("DB5000_FIX_TABLE_POSITIONS".UNIT_1.FIXTURE[2].IN_CLADDING_STATION_3 AND "DB7330_ETXETAR_ROBOT_CELL_INTERLOCK".INTERLOCKS_UNIT_1.MACHINE_TO_ROBOT.MCH_FIX_2_CALIBRATION_REQ) OR ("DB5000_FIX_TABLE_POSITIONS".UNIT_1.FIXTURE[4].IN_CLADDING_STATION_3 AND "DB7330_ETXETAR_ROBOT_CELL_INTERLOCK".INTERLOCKS_UNIT_1.MACHINE_TO_ROBOT.MCH_FIX_4_CALIBRATION_REQ)) AND NOT "DB8000_PART_STATUS".UNIT_1.STATION_3.PART_A.STATUS.UNIT_1_STATUS.FACE_N_STATION_3_DONE)) AND "DB8000_PART_STATUS".UNIT_1.STATION_3.PART_A.STATUS.PRESENT AND "DB8000_PART_STATUS".UNIT_1.STATION_3.PART_A.STATUS.MASTER_PART;
END_REGION

REGION Network 24: FULL DEPTH
   RUNG wire#powerrail
      Contact( "DB1201_PART_CYCLE_UNIT_1".SEQUENCE.RUNNING )
      wire#w1
      Contact( "DB440_MACHINE_ALARM_DECODING".GLOBAL_ALARMS_MACHINE.ALARM )
      wire#w2
      I_Contact( "DB2440_GLOBAL_DATA".GLOBAL_DATA.UNIT_01_ST_0_ANY_CYCLE_ACTIVE )
      I_Contact( "DB2440_GLOBAL_DATA".GLOBAL_DATA.UNIT_01_ST_1_ANY_CYCLE_ACTIVE )
      I_Contact( "DB2440_GLOBAL_DATA".GLOBAL_DATA.UNIT_01_ST_2_ANY_CYCLE_ACTIVE )
      I_Contact( "DB2440_GLOBAL_DATA".GLOBAL_DATA.UNIT_01_ST_3_ANY_CYCLE_ACTIVE )
      I_Contact( "DB2440_GLOBAL_DATA".GLOBAL_DATA.UNIT_01_ST_4_ANY_CYCLE_ACTIVE )
      Coil( "DB1201_PART_CYCLE_UNIT_1".FULL_DEPTH )
   END_RUNG
   RUNG wire#w1
      Contact( "DB440_MACHINE_ALARM_DECODING".GLOBAL_ALARMS_MACHINE.SEOC_ALARMS )
   END_RUNG wire#w2
   RUNG wire#w1
      Contact( "DB440_MACHINE_ALARM_DECODING".GLOBAL_ALARMS_MACHINE.SEOC_WARNING )
   END_RUNG wire#w2
   RUNG wire#w1
      Contact( "DB2031_CYCLES_GENERAL".RUN_OUT_UNIT_1.CYCLE_COMPLETED )
   END_RUNG wire#w2
   // the same network as SCL:
   "DB1201_PART_CYCLE_UNIT_1".FULL_DEPTH := "DB1201_PART_CYCLE_UNIT_1".SEQUENCE.RUNNING AND ("DB440_MACHINE_ALARM_DECODING".GLOBAL_ALARMS_MACHINE.ALARM OR "DB440_MACHINE_ALARM_DECODING".GLOBAL_ALARMS_MACHINE.SEOC_ALARMS OR "DB440_MACHINE_ALARM_DECODING".GLOBAL_ALARMS_MACHINE.SEOC_WARNING OR "DB2031_CYCLES_GENERAL".RUN_OUT_UNIT_1.CYCLE_COMPLETED) AND NOT "DB2440_GLOBAL_DATA".GLOBAL_DATA.UNIT_01_ST_0_ANY_CYCLE_ACTIVE AND NOT "DB2440_GLOBAL_DATA".GLOBAL_DATA.UNIT_01_ST_1_ANY_CYCLE_ACTIVE AND NOT "DB2440_GLOBAL_DATA".GLOBAL_DATA.UNIT_01_ST_2_ANY_CYCLE_ACTIVE AND NOT "DB2440_GLOBAL_DATA".GLOBAL_DATA.UNIT_01_ST_3_ANY_CYCLE_ACTIVE AND NOT "DB2440_GLOBAL_DATA".GLOBAL_DATA.UNIT_01_ST_4_ANY_CYCLE_ACTIVE;
END_REGION

REGION Network 25: TIME EXCEEDED ALARM
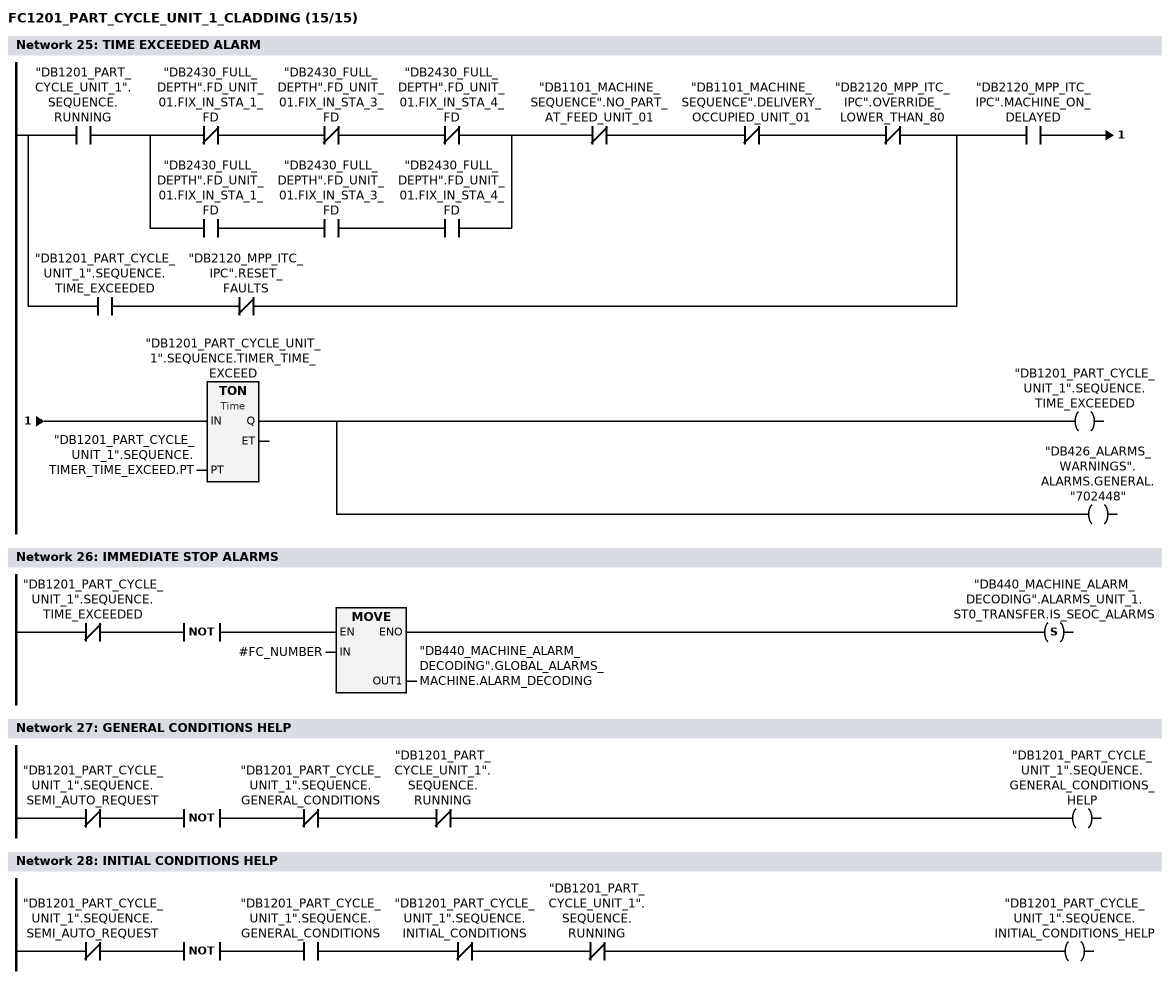
   RUNG wire#powerrail
      Contact( "DB1201_PART_CYCLE_UNIT_1".SEQUENCE.RUNNING )
      wire#w1
      I_Contact( "DB2430_FULL_DEPTH".FD_UNIT_01.FIX_IN_STA_1_FD )
      I_Contact( "DB2430_FULL_DEPTH".FD_UNIT_01.FIX_IN_STA_3_FD )
      I_Contact( "DB2430_FULL_DEPTH".FD_UNIT_01.FIX_IN_STA_4_FD )
      wire#w2
      I_Contact( "DB1101_MACHINE_SEQUENCE".NO_PART_AT_FEED_UNIT_01 )
      I_Contact( "DB1101_MACHINE_SEQUENCE".DELIVERY_OCCUPIED_UNIT_01 )
      I_Contact( "DB2120_MPP_ITC_IPC".OVERRIDE_LOWER_THAN_80 )
      wire#w3
      Contact( "DB2120_MPP_ITC_IPC".MACHINE_ON_DELAYED )
      { S7_Templates := "time_type := Time" } "DB1201_PART_CYCLE_UNIT_1".SEQUENCE.TIMER_TIME_EXCEED.TON(pt := "DB1201_PART_CYCLE_UNIT_1".SEQUENCE.TIMER_TIME_EXCEED.PT, et =>)
      wire#w4
      Coil( "DB1201_PART_CYCLE_UNIT_1".SEQUENCE.TIME_EXCEEDED )
   END_RUNG
   RUNG wire#w1
      Contact( "DB2430_FULL_DEPTH".FD_UNIT_01.FIX_IN_STA_1_FD )
      Contact( "DB2430_FULL_DEPTH".FD_UNIT_01.FIX_IN_STA_3_FD )
      Contact( "DB2430_FULL_DEPTH".FD_UNIT_01.FIX_IN_STA_4_FD )
   END_RUNG wire#w2
   RUNG wire#powerrail
      Contact( "DB1201_PART_CYCLE_UNIT_1".SEQUENCE.TIME_EXCEEDED )
      I_Contact( "DB2120_MPP_ITC_IPC".RESET_FAULTS )
   END_RUNG wire#w3
   RUNG wire#w4
      Coil( "DB426_ALARMS_WARNINGS".ALARMS.GENERAL."702448" )
   END_RUNG
   // the same network as SCL:
   "DB1201_PART_CYCLE_UNIT_1".SEQUENCE.TIMER_TIME_EXCEED.TON(IN := (("DB1201_PART_CYCLE_UNIT_1".SEQUENCE.RUNNING AND ((NOT "DB2430_FULL_DEPTH".FD_UNIT_01.FIX_IN_STA_1_FD AND NOT "DB2430_FULL_DEPTH".FD_UNIT_01.FIX_IN_STA_3_FD AND NOT "DB2430_FULL_DEPTH".FD_UNIT_01.FIX_IN_STA_4_FD) OR ("DB2430_FULL_DEPTH".FD_UNIT_01.FIX_IN_STA_1_FD AND "DB2430_FULL_DEPTH".FD_UNIT_01.FIX_IN_STA_3_FD AND "DB2430_FULL_DEPTH".FD_UNIT_01.FIX_IN_STA_4_FD)) AND NOT "DB1101_MACHINE_SEQUENCE".NO_PART_AT_FEED_UNIT_01 AND NOT "DB1101_MACHINE_SEQUENCE".DELIVERY_OCCUPIED_UNIT_01 AND NOT "DB2120_MPP_ITC_IPC".OVERRIDE_LOWER_THAN_80) OR ("DB1201_PART_CYCLE_UNIT_1".SEQUENCE.TIME_EXCEEDED AND NOT "DB2120_MPP_ITC_IPC".RESET_FAULTS)) AND "DB2120_MPP_ITC_IPC".MACHINE_ON_DELAYED,
                           PT := "DB1201_PART_CYCLE_UNIT_1".SEQUENCE.TIMER_TIME_EXCEED.PT);
   "DB1201_PART_CYCLE_UNIT_1".SEQUENCE.TIME_EXCEEDED := "DB1201_PART_CYCLE_UNIT_1".SEQUENCE.TIMER_TIME_EXCEED.Q;
   "DB426_ALARMS_WARNINGS".ALARMS.GENERAL."702448" := "DB1201_PART_CYCLE_UNIT_1".SEQUENCE.TIMER_TIME_EXCEED.Q;
END_REGION

REGION Network 26: IMMEDIATE STOP ALARMS
   RUNG wire#powerrail
      I_Contact( "DB1201_PART_CYCLE_UNIT_1".SEQUENCE.TIME_EXCEEDED )
      Not()
      { S7_GenerateENO := "TRUE" } Move(in := #FC_NUMBER, out1 => "DB440_MACHINE_ALARM_DECODING".GLOBAL_ALARMS_MACHINE.ALARM_DECODING)
      S_Coil( "DB440_MACHINE_ALARM_DECODING".ALARMS_UNIT_1.ST0_TRANSFER.IS_SEOC_ALARMS )
   END_RUNG
   // the same network as SCL:
   // ENO of a box is taken as its EN; it also drops when the box reports an error
   IF NOT (NOT "DB1201_PART_CYCLE_UNIT_1".SEQUENCE.TIME_EXCEEDED) THEN
       "DB440_MACHINE_ALARM_DECODING".GLOBAL_ALARMS_MACHINE.ALARM_DECODING := #FC_NUMBER;
       "DB440_MACHINE_ALARM_DECODING".ALARMS_UNIT_1.ST0_TRANSFER.IS_SEOC_ALARMS := TRUE;
   END_IF;
END_REGION

REGION Network 27: GENERAL CONDITIONS HELP
   RUNG wire#powerrail
      I_Contact( "DB1201_PART_CYCLE_UNIT_1".SEQUENCE.SEMI_AUTO_REQUEST )
      Not()
      I_Contact( "DB1201_PART_CYCLE_UNIT_1".SEQUENCE.GENERAL_CONDITIONS )
      I_Contact( "DB1201_PART_CYCLE_UNIT_1".SEQUENCE.RUNNING )
      Coil( "DB1201_PART_CYCLE_UNIT_1".SEQUENCE.GENERAL_CONDITIONS_HELP )
   END_RUNG
   // the same network as SCL:
   "DB1201_PART_CYCLE_UNIT_1".SEQUENCE.GENERAL_CONDITIONS_HELP := NOT (NOT "DB1201_PART_CYCLE_UNIT_1".SEQUENCE.SEMI_AUTO_REQUEST) AND NOT "DB1201_PART_CYCLE_UNIT_1".SEQUENCE.GENERAL_CONDITIONS AND NOT "DB1201_PART_CYCLE_UNIT_1".SEQUENCE.RUNNING;
END_REGION

REGION Network 28: INITIAL CONDITIONS HELP
   RUNG wire#powerrail
      I_Contact( "DB1201_PART_CYCLE_UNIT_1".SEQUENCE.SEMI_AUTO_REQUEST )
      Not()
      Contact( "DB1201_PART_CYCLE_UNIT_1".SEQUENCE.GENERAL_CONDITIONS )
      I_Contact( "DB1201_PART_CYCLE_UNIT_1".SEQUENCE.INITIAL_CONDITIONS )
      I_Contact( "DB1201_PART_CYCLE_UNIT_1".SEQUENCE.RUNNING )
      Coil( "DB1201_PART_CYCLE_UNIT_1".SEQUENCE.INITIAL_CONDITIONS_HELP )
   END_RUNG
   // the same network as SCL:
   "DB1201_PART_CYCLE_UNIT_1".SEQUENCE.INITIAL_CONDITIONS_HELP := NOT (NOT "DB1201_PART_CYCLE_UNIT_1".SEQUENCE.SEMI_AUTO_REQUEST) AND "DB1201_PART_CYCLE_UNIT_1".SEQUENCE.GENERAL_CONDITIONS AND NOT "DB1201_PART_CYCLE_UNIT_1".SEQUENCE.INITIAL_CONDITIONS AND NOT "DB1201_PART_CYCLE_UNIT_1".SEQUENCE.RUNNING;
END_REGION
END_FUNCTION
